REGION Network 27: STIRRER SPEED LINE 1 LIMITS CALCULATION ALARM
   RUNG wire#powerrail
      Add(in1 := #oPLC_Aux.o_rStirrerSpeedNominal_Line1, in2 := #"iHMI_Offsets Alarms and Warnings".StirrerSpeedNominalLine1_Max_Alarm, out => #oPLC_Aux.o_rHHlimitStirrerSpeedNominal_Line1)
      "FC21020_FEEDER_SCALING"(DINT_INPUT_VALUE := 0, REAL_INPUT_VALUE := #oPLC_Aux.o_rHHlimitStirrerSpeedNominal_Line1, DINT_TO_REAL := false, REAL_TRANSFORM_FOR_FEEDER := true, OUTPUT_VALUE_PLC => #Retval_Fill_R, OUTPUT_VALUE_FEEDER => #ioPowder_Feeder_Unit_In_Out.Outputs."PF Setpoints, Warnings and Alarms".o_rHHlimitStirrerSpeedNominal_Line1)
      Sub(in1 := #oPLC_Aux.o_rStirrerSpeedNominal_Line1, in2 := #"iHMI_Offsets Alarms and Warnings".StirrerSpeedNominalLine1_Min_Alarm, out => #oPLC_Aux.o_rLLlimitStirrerSpeedNominal_Line1)
      "FC21020_FEEDER_SCALING"(DINT_INPUT_VALUE := 0, REAL_INPUT_VALUE := #oPLC_Aux.o_rLLlimitStirrerSpeedNominal_Line1, DINT_TO_REAL := false, REAL_TRANSFORM_FOR_FEEDER := true, OUTPUT_VALUE_PLC => #Retval_Fill_R, OUTPUT_VALUE_FEEDER => #ioPowder_Feeder_Unit_In_Out.Outputs."PF Setpoints, Warnings and Alarms".o_rLLlimitStirrerSpeedNominal_Line1)
   END_RUNG
   // the same network as SCL:
   #oPLC_Aux.o_rHHlimitStirrerSpeedNominal_Line1 := #oPLC_Aux.o_rStirrerSpeedNominal_Line1 + #"iHMI_Offsets Alarms and Warnings".StirrerSpeedNominalLine1_Max_Alarm;
   "FC21020_FEEDER_SCALING"(DINT_INPUT_VALUE := 0,
                           REAL_INPUT_VALUE := #oPLC_Aux.o_rHHlimitStirrerSpeedNominal_Line1,
                           DINT_TO_REAL := false,
                           REAL_TRANSFORM_FOR_FEEDER := true,
                           OUTPUT_VALUE_PLC => #Retval_Fill_R,
                           OUTPUT_VALUE_FEEDER => #ioPowder_Feeder_Unit_In_Out.Outputs."PF Setpoints, Warnings and Alarms".o_rHHlimitStirrerSpeedNominal_Line1,
                           ENO => #_w1);
   IF #_w1 THEN
       #oPLC_Aux.o_rLLlimitStirrerSpeedNominal_Line1 := #oPLC_Aux.o_rStirrerSpeedNominal_Line1 - #"iHMI_Offsets Alarms and Warnings".StirrerSpeedNominalLine1_Min_Alarm;
       "FC21020_FEEDER_SCALING"(DINT_INPUT_VALUE := 0,
                               REAL_INPUT_VALUE := #oPLC_Aux.o_rLLlimitStirrerSpeedNominal_Line1,
                               DINT_TO_REAL := false,
                               REAL_TRANSFORM_FOR_FEEDER := true,
                               OUTPUT_VALUE_PLC => #Retval_Fill_R,
                               OUTPUT_VALUE_FEEDER => #ioPowder_Feeder_Unit_In_Out.Outputs."PF Setpoints, Warnings and Alarms".o_rLLlimitStirrerSpeedNominal_Line1);
   END_IF;
END_REGION

REGION Network 28: STIRRER SPEED LINE 2 LIMITS CALCULATION ALARM
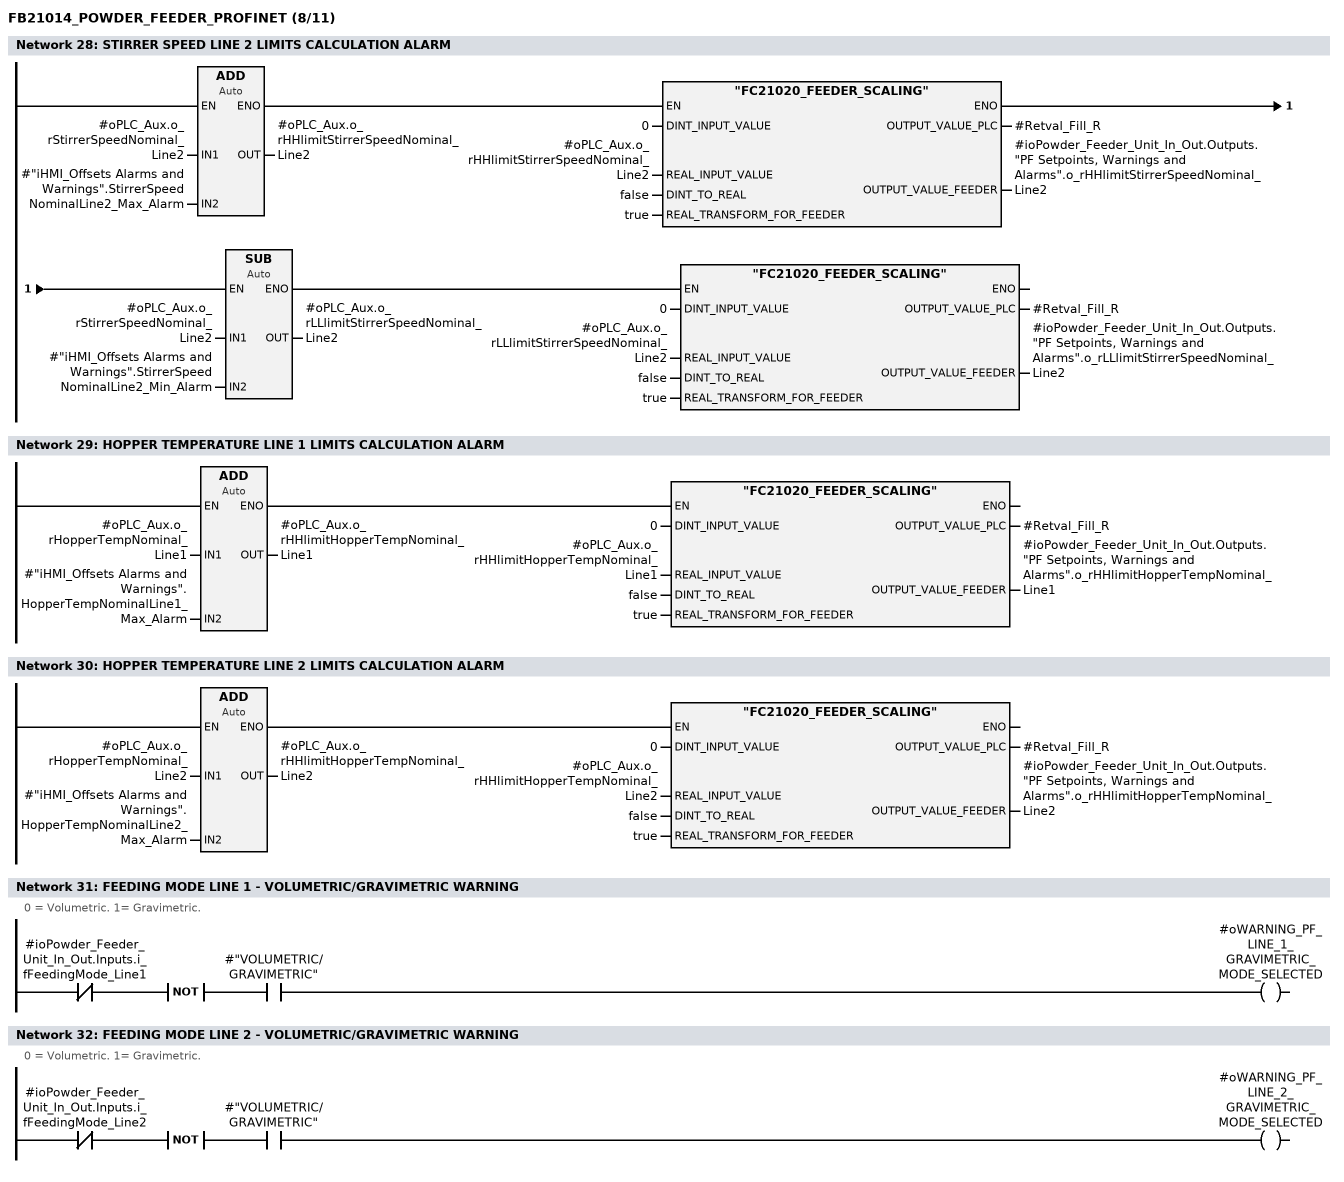
   RUNG wire#powerrail
      Add(in1 := #oPLC_Aux.o_rStirrerSpeedNominal_Line2, in2 := #"iHMI_Offsets Alarms and Warnings".StirrerSpeedNominalLine2_Max_Alarm, out => #oPLC_Aux.o_rHHlimitStirrerSpeedNominal_Line2)
      "FC21020_FEEDER_SCALING"(DINT_INPUT_VALUE := 0, REAL_INPUT_VALUE := #oPLC_Aux.o_rHHlimitStirrerSpeedNominal_Line2, DINT_TO_REAL := false, REAL_TRANSFORM_FOR_FEEDER := true, OUTPUT_VALUE_PLC => #Retval_Fill_R, OUTPUT_VALUE_FEEDER => #ioPowder_Feeder_Unit_In_Out.Outputs."PF Setpoints, Warnings and Alarms".o_rHHlimitStirrerSpeedNominal_Line2)
      Sub(in1 := #oPLC_Aux.o_rStirrerSpeedNominal_Line2, in2 := #"iHMI_Offsets Alarms and Warnings".StirrerSpeedNominalLine2_Min_Alarm, out => #oPLC_Aux.o_rLLlimitStirrerSpeedNominal_Line2)
      "FC21020_FEEDER_SCALING"(DINT_INPUT_VALUE := 0, REAL_INPUT_VALUE := #oPLC_Aux.o_rLLlimitStirrerSpeedNominal_Line2, DINT_TO_REAL := false, REAL_TRANSFORM_FOR_FEEDER := true, OUTPUT_VALUE_PLC => #Retval_Fill_R, OUTPUT_VALUE_FEEDER => #ioPowder_Feeder_Unit_In_Out.Outputs."PF Setpoints, Warnings and Alarms".o_rLLlimitStirrerSpeedNominal_Line2)
   END_RUNG
   // the same network as SCL:
   #oPLC_Aux.o_rHHlimitStirrerSpeedNominal_Line2 := #oPLC_Aux.o_rStirrerSpeedNominal_Line2 + #"iHMI_Offsets Alarms and Warnings".StirrerSpeedNominalLine2_Max_Alarm;
   "FC21020_FEEDER_SCALING"(DINT_INPUT_VALUE := 0,
                           REAL_INPUT_VALUE := #oPLC_Aux.o_rHHlimitStirrerSpeedNominal_Line2,
                           DINT_TO_REAL := false,
                           REAL_TRANSFORM_FOR_FEEDER := true,
                           OUTPUT_VALUE_PLC => #Retval_Fill_R,
                           OUTPUT_VALUE_FEEDER => #ioPowder_Feeder_Unit_In_Out.Outputs."PF Setpoints, Warnings and Alarms".o_rHHlimitStirrerSpeedNominal_Line2,
                           ENO => #_w1);
   IF #_w1 THEN
       #oPLC_Aux.o_rLLlimitStirrerSpeedNominal_Line2 := #oPLC_Aux.o_rStirrerSpeedNominal_Line2 - #"iHMI_Offsets Alarms and Warnings".StirrerSpeedNominalLine2_Min_Alarm;
       "FC21020_FEEDER_SCALING"(DINT_INPUT_VALUE := 0,
                               REAL_INPUT_VALUE := #oPLC_Aux.o_rLLlimitStirrerSpeedNominal_Line2,
                               DINT_TO_REAL := false,
                               REAL_TRANSFORM_FOR_FEEDER := true,
                               OUTPUT_VALUE_PLC => #Retval_Fill_R,
                               OUTPUT_VALUE_FEEDER => #ioPowder_Feeder_Unit_In_Out.Outputs."PF Setpoints, Warnings and Alarms".o_rLLlimitStirrerSpeedNominal_Line2);
   END_IF;
END_REGION

REGION Network 29: HOPPER TEMPERATURE LINE 1 LIMITS CALCULATION ALARM
   RUNG wire#powerrail
      Add(in1 := #oPLC_Aux.o_rHopperTempNominal_Line1, in2 := #"iHMI_Offsets Alarms and Warnings".HopperTempNominalLine1_Max_Alarm, out => #oPLC_Aux.o_rHHlimitHopperTempNominal_Line1)
      "FC21020_FEEDER_SCALING"(DINT_INPUT_VALUE := 0, REAL_INPUT_VALUE := #oPLC_Aux.o_rHHlimitHopperTempNominal_Line1, DINT_TO_REAL := false, REAL_TRANSFORM_FOR_FEEDER := true, OUTPUT_VALUE_PLC => #Retval_Fill_R, OUTPUT_VALUE_FEEDER => #ioPowder_Feeder_Unit_In_Out.Outputs."PF Setpoints, Warnings and Alarms".o_rHHlimitHopperTempNominal_Line1)
   END_RUNG
   // the same network as SCL:
   #oPLC_Aux.o_rHHlimitHopperTempNominal_Line1 := #oPLC_Aux.o_rHopperTempNominal_Line1 + #"iHMI_Offsets Alarms and Warnings".HopperTempNominalLine1_Max_Alarm;
   "FC21020_FEEDER_SCALING"(DINT_INPUT_VALUE := 0,
                           REAL_INPUT_VALUE := #oPLC_Aux.o_rHHlimitHopperTempNominal_Line1,
                           DINT_TO_REAL := false,
                           REAL_TRANSFORM_FOR_FEEDER := true,
                           OUTPUT_VALUE_PLC => #Retval_Fill_R,
                           OUTPUT_VALUE_FEEDER => #ioPowder_Feeder_Unit_In_Out.Outputs."PF Setpoints, Warnings and Alarms".o_rHHlimitHopperTempNominal_Line1);
END_REGION

REGION Network 30: HOPPER TEMPERATURE LINE 2 LIMITS CALCULATION ALARM
   RUNG wire#powerrail
      Add(in1 := #oPLC_Aux.o_rHopperTempNominal_Line2, in2 := #"iHMI_Offsets Alarms and Warnings".HopperTempNominalLine2_Max_Alarm, out => #oPLC_Aux.o_rHHlimitHopperTempNominal_Line2)
      "FC21020_FEEDER_SCALING"(DINT_INPUT_VALUE := 0, REAL_INPUT_VALUE := #oPLC_Aux.o_rHHlimitHopperTempNominal_Line2, DINT_TO_REAL := false, REAL_TRANSFORM_FOR_FEEDER := true, OUTPUT_VALUE_PLC => #Retval_Fill_R, OUTPUT_VALUE_FEEDER => #ioPowder_Feeder_Unit_In_Out.Outputs."PF Setpoints, Warnings and Alarms".o_rHHlimitHopperTempNominal_Line2)
   END_RUNG
   // the same network as SCL:
   #oPLC_Aux.o_rHHlimitHopperTempNominal_Line2 := #oPLC_Aux.o_rHopperTempNominal_Line2 + #"iHMI_Offsets Alarms and Warnings".HopperTempNominalLine2_Max_Alarm;
   "FC21020_FEEDER_SCALING"(DINT_INPUT_VALUE := 0,
                           REAL_INPUT_VALUE := #oPLC_Aux.o_rHHlimitHopperTempNominal_Line2,
                           DINT_TO_REAL := false,
                           REAL_TRANSFORM_FOR_FEEDER := true,
                           OUTPUT_VALUE_PLC => #Retval_Fill_R,
                           OUTPUT_VALUE_FEEDER => #ioPowder_Feeder_Unit_In_Out.Outputs."PF Setpoints, Warnings and Alarms".o_rHHlimitHopperTempNominal_Line2);
END_REGION

REGION Network 31: FEEDING MODE LINE 1 - VOLUMETRIC/GRAVIMETRIC WARNING
   // 0 = Volumetric. 1= Gravimetric.
   RUNG wire#powerrail
      I_Contact( #ioPowder_Feeder_Unit_In_Out.Inputs.i_fFeedingMode_Line1 )
      Not()
      Contact( #"VOLUMETRIC/GRAVIMETRIC" )
      Coil( #oWARNING_PF_LINE_1_GRAVIMETRIC_MODE_SELECTED )
   END_RUNG
   // the same network as SCL:
   #oWARNING_PF_LINE_1_GRAVIMETRIC_MODE_SELECTED := NOT (NOT #ioPowder_Feeder_Unit_In_Out.Inputs.i_fFeedingMode_Line1) AND #"VOLUMETRIC/GRAVIMETRIC";
END_REGION

REGION Network 32: FEEDING MODE LINE 2 - VOLUMETRIC/GRAVIMETRIC WARNING
   // 0 = Volumetric. 1= Gravimetric.
   RUNG wire#powerrail
      I_Contact( #ioPowder_Feeder_Unit_In_Out.Inputs.i_fFeedingMode_Line2 )
      Not()
      Contact( #"VOLUMETRIC/GRAVIMETRIC" )
      Coil( #oWARNING_PF_LINE_2_GRAVIMETRIC_MODE_SELECTED )
   END_RUNG
   // the same network as SCL:
   #oWARNING_PF_LINE_2_GRAVIMETRIC_MODE_SELECTED := NOT (NOT #ioPowder_Feeder_Unit_In_Out.Inputs.i_fFeedingMode_Line2) AND #"VOLUMETRIC/GRAVIMETRIC";
END_REGION

REGION Network 33: WARNING
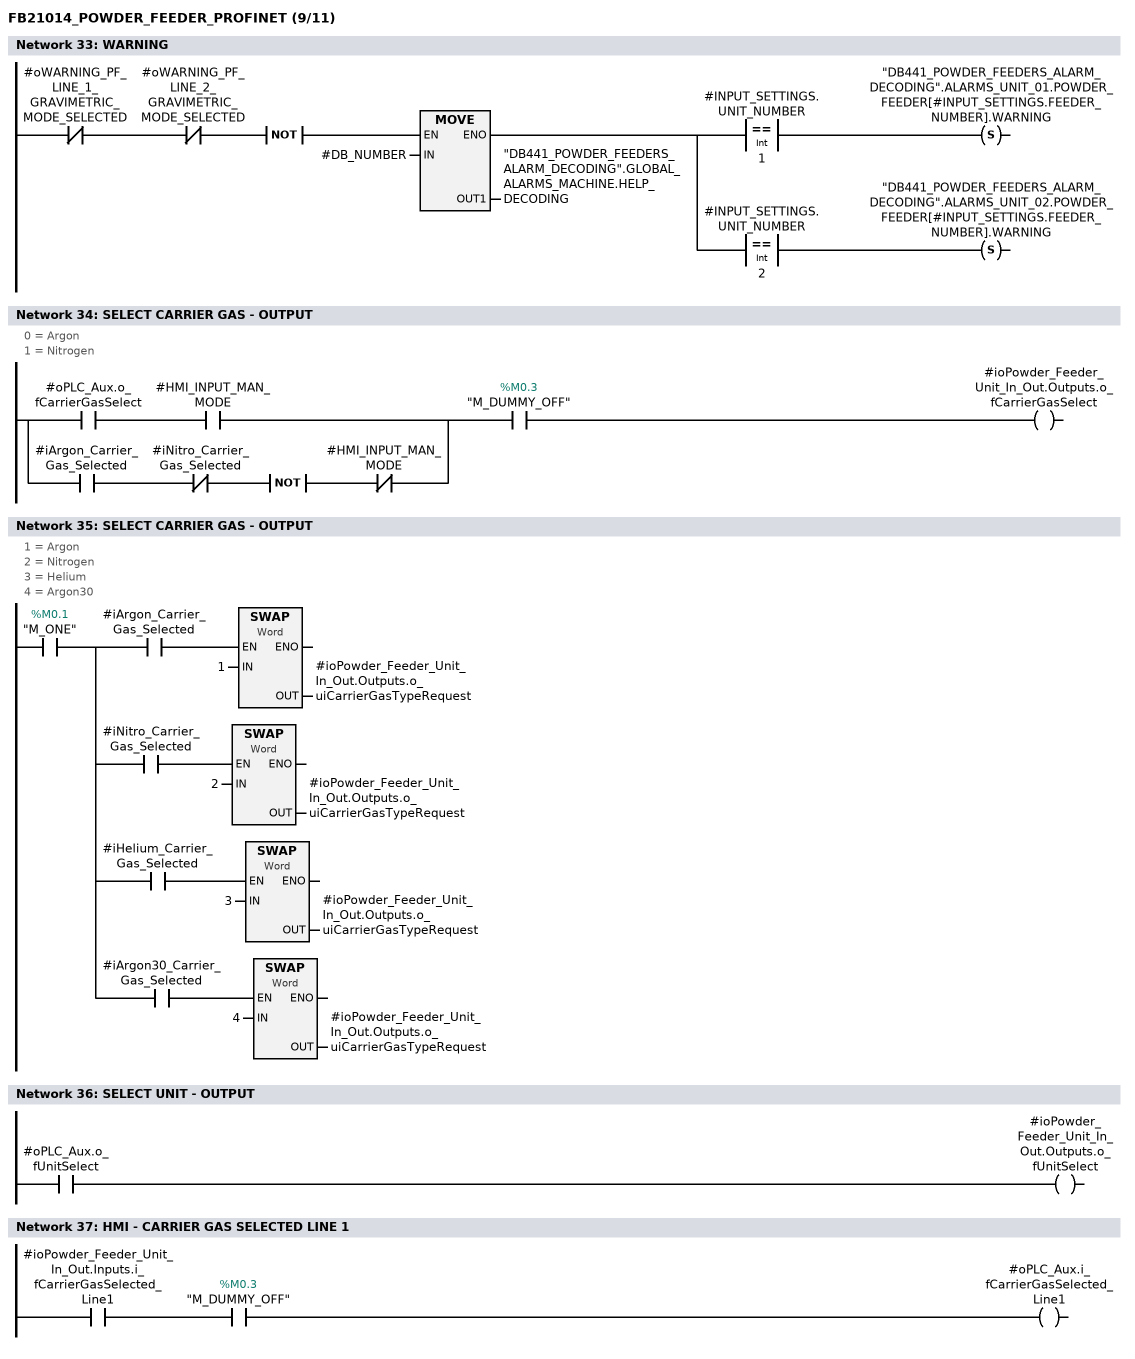
   RUNG wire#powerrail
      I_Contact( #oWARNING_PF_LINE_1_GRAVIMETRIC_MODE_SELECTED )
      I_Contact( #oWARNING_PF_LINE_2_GRAVIMETRIC_MODE_SELECTED )
      Not()
      Move(in := #DB_NUMBER, out1 => "DB441_POWDER_FEEDERS_ALARM_DECODING".GLOBAL_ALARMS_MACHINE.HELP_DECODING)
      wire#w1
      { S7_Templates := "SrcType := Int" } EQ_Contact(in1 := #INPUT_SETTINGS.UNIT_NUMBER, in2 := 1)
      S_Coil( "DB441_POWDER_FEEDERS_ALARM_DECODING".ALARMS_UNIT_01.POWDER_FEEDER[#INPUT_SETTINGS.FEEDER_NUMBER].WARNING )
   END_RUNG
   RUNG wire#w1
      { S7_Templates := "SrcType := Int" } EQ_Contact(in1 := #INPUT_SETTINGS.UNIT_NUMBER, in2 := 2)
      S_Coil( "DB441_POWDER_FEEDERS_ALARM_DECODING".ALARMS_UNIT_02.POWDER_FEEDER[#INPUT_SETTINGS.FEEDER_NUMBER].WARNING )
   END_RUNG
   // the same network as SCL:
   #_w1 := NOT (NOT #oWARNING_PF_LINE_1_GRAVIMETRIC_MODE_SELECTED AND NOT #oWARNING_PF_LINE_2_GRAVIMETRIC_MODE_SELECTED);
   IF #_w1 THEN
       "DB441_POWDER_FEEDERS_ALARM_DECODING".GLOBAL_ALARMS_MACHINE.HELP_DECODING := #DB_NUMBER;
   END_IF;
   IF #_w1 AND (#INPUT_SETTINGS.UNIT_NUMBER = 1) THEN
       "DB441_POWDER_FEEDERS_ALARM_DECODING".ALARMS_UNIT_01.POWDER_FEEDER[#INPUT_SETTINGS.FEEDER_NUMBER].WARNING := TRUE;
   END_IF;
   IF #_w1 AND (#INPUT_SETTINGS.UNIT_NUMBER = 2) THEN
       "DB441_POWDER_FEEDERS_ALARM_DECODING".ALARMS_UNIT_02.POWDER_FEEDER[#INPUT_SETTINGS.FEEDER_NUMBER].WARNING := TRUE;
   END_IF;
END_REGION

REGION Network 34: SELECT CARRIER GAS - OUTPUT
   // 0 = Argon
   // 1 = Nitrogen
   RUNG wire#powerrail
      Contact( #oPLC_Aux.o_fCarrierGasSelect )
      Contact( #HMI_INPUT_MAN_MODE )
      wire#w1
      Contact( "M_DUMMY_OFF" )
      Coil( #ioPowder_Feeder_Unit_In_Out.Outputs.o_fCarrierGasSelect )
   END_RUNG
   RUNG wire#powerrail
      Contact( #iArgon_Carrier_Gas_Selected )
      I_Contact( #iNitro_Carrier_Gas_Selected )
      Not()
      I_Contact( #HMI_INPUT_MAN_MODE )
   END_RUNG wire#w1
   // the same network as SCL:
   #ioPowder_Feeder_Unit_In_Out.Outputs.o_fCarrierGasSelect := ((#oPLC_Aux.o_fCarrierGasSelect AND #HMI_INPUT_MAN_MODE) OR (NOT (#iArgon_Carrier_Gas_Selected AND NOT #iNitro_Carrier_Gas_Selected) AND NOT #HMI_INPUT_MAN_MODE)) AND "M_DUMMY_OFF";
END_REGION

REGION Network 35: SELECT CARRIER GAS - OUTPUT
   // 1 = Argon
   // 2 = Nitrogen
   // 3 = Helium
   // 4 = Argon30
   IF "M_ONE" AND #iArgon_Carrier_Gas_Selected THEN
       #ioPowder_Feeder_Unit_In_Out.Outputs.o_uiCarrierGasTypeRequest := SWAP(1);
   END_IF;
   IF "M_ONE" AND #iNitro_Carrier_Gas_Selected THEN
       #ioPowder_Feeder_Unit_In_Out.Outputs.o_uiCarrierGasTypeRequest := SWAP(2);
   END_IF;
   IF "M_ONE" AND #iHelium_Carrier_Gas_Selected THEN
       #ioPowder_Feeder_Unit_In_Out.Outputs.o_uiCarrierGasTypeRequest := SWAP(3);
   END_IF;
   IF "M_ONE" AND #iArgon30_Carrier_Gas_Selected THEN
       #ioPowder_Feeder_Unit_In_Out.Outputs.o_uiCarrierGasTypeRequest := SWAP(4);
   END_IF;
END_REGION

REGION Network 36: SELECT UNIT - OUTPUT
   RUNG wire#powerrail
      Contact( #oPLC_Aux.o_fUnitSelect )
      Coil( #ioPowder_Feeder_Unit_In_Out.Outputs.o_fUnitSelect )
   END_RUNG
   // the same network as SCL:
   #ioPowder_Feeder_Unit_In_Out.Outputs.o_fUnitSelect := #oPLC_Aux.o_fUnitSelect;
END_REGION

REGION Network 37: HMI - CARRIER GAS SELECTED LINE 1
   RUNG wire#powerrail
      Contact( #ioPowder_Feeder_Unit_In_Out.Inputs.i_fCarrierGasSelected_Line1 )
      Contact( "M_DUMMY_OFF" )
      Coil( #oPLC_Aux.i_fCarrierGasSelected_Line1 )
   END_RUNG
   // the same network as SCL:
   #oPLC_Aux.i_fCarrierGasSelected_Line1 := #ioPowder_Feeder_Unit_In_Out.Inputs.i_fCarrierGasSelected_Line1 AND "M_DUMMY_OFF";
END_REGION

REGION Network 38: HMI - CARRIER GAS SELECTED LINE 2
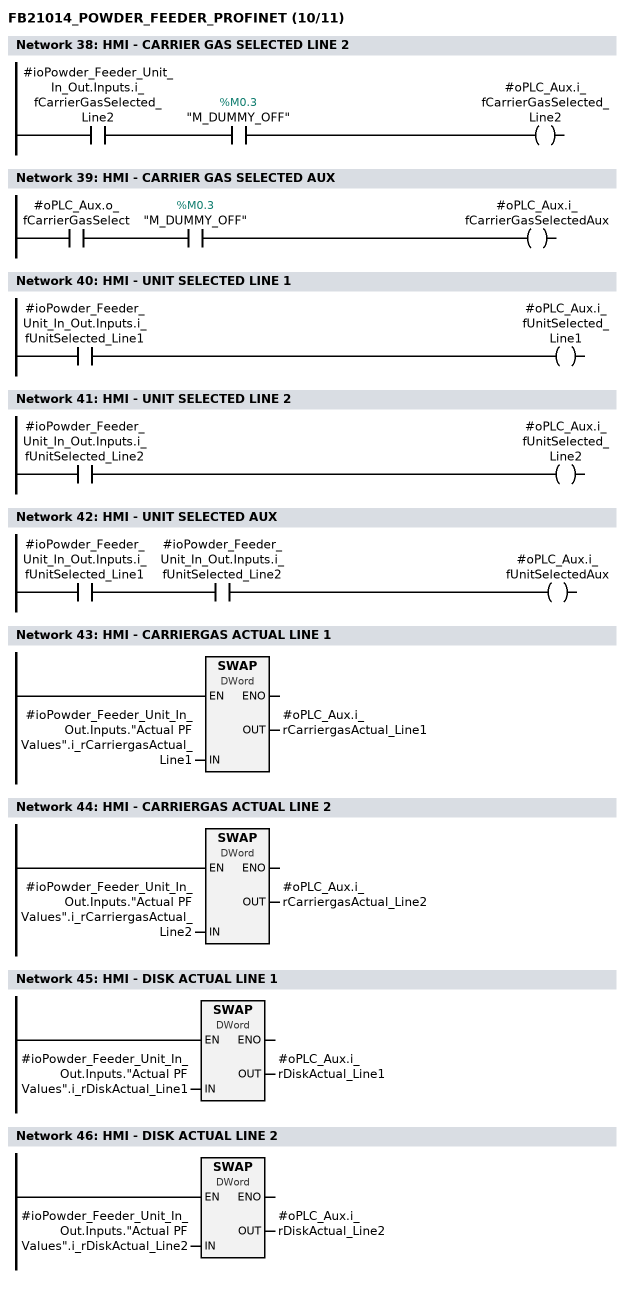
   RUNG wire#powerrail
      Contact( #ioPowder_Feeder_Unit_In_Out.Inputs.i_fCarrierGasSelected_Line2 )
      Contact( "M_DUMMY_OFF" )
      Coil( #oPLC_Aux.i_fCarrierGasSelected_Line2 )
   END_RUNG
   // the same network as SCL:
   #oPLC_Aux.i_fCarrierGasSelected_Line2 := #ioPowder_Feeder_Unit_In_Out.Inputs.i_fCarrierGasSelected_Line2 AND "M_DUMMY_OFF";
END_REGION

REGION Network 39: HMI - CARRIER GAS SELECTED AUX
   RUNG wire#powerrail
      Contact( #oPLC_Aux.o_fCarrierGasSelect )
      Contact( "M_DUMMY_OFF" )
      Coil( #oPLC_Aux.i_fCarrierGasSelectedAux )
   END_RUNG
   // the same network as SCL:
   #oPLC_Aux.i_fCarrierGasSelectedAux := #oPLC_Aux.o_fCarrierGasSelect AND "M_DUMMY_OFF";
END_REGION

REGION Network 40: HMI - UNIT SELECTED LINE 1
   RUNG wire#powerrail
      Contact( #ioPowder_Feeder_Unit_In_Out.Inputs.i_fUnitSelected_Line1 )
      Coil( #oPLC_Aux.i_fUnitSelected_Line1 )
   END_RUNG
   // the same network as SCL:
   #oPLC_Aux.i_fUnitSelected_Line1 := #ioPowder_Feeder_Unit_In_Out.Inputs.i_fUnitSelected_Line1;
END_REGION

REGION Network 41: HMI - UNIT SELECTED LINE 2
   RUNG wire#powerrail
      Contact( #ioPowder_Feeder_Unit_In_Out.Inputs.i_fUnitSelected_Line2 )
      Coil( #oPLC_Aux.i_fUnitSelected_Line2 )
   END_RUNG
   // the same network as SCL:
   #oPLC_Aux.i_fUnitSelected_Line2 := #ioPowder_Feeder_Unit_In_Out.Inputs.i_fUnitSelected_Line2;
END_REGION

REGION Network 42: HMI - UNIT SELECTED AUX
   RUNG wire#powerrail
      Contact( #ioPowder_Feeder_Unit_In_Out.Inputs.i_fUnitSelected_Line1 )
      Contact( #ioPowder_Feeder_Unit_In_Out.Inputs.i_fUnitSelected_Line2 )
      Coil( #oPLC_Aux.i_fUnitSelectedAux )
   END_RUNG
   // the same network as SCL:
   #oPLC_Aux.i_fUnitSelectedAux := #ioPowder_Feeder_Unit_In_Out.Inputs.i_fUnitSelected_Line1 AND #ioPowder_Feeder_Unit_In_Out.Inputs.i_fUnitSelected_Line2;
END_REGION

REGION Network 43: HMI - CARRIERGAS ACTUAL LINE 1
   #oPLC_Aux.i_rCarriergasActual_Line1 := SWAP(#ioPowder_Feeder_Unit_In_Out.Inputs."Actual PF Values".i_rCarriergasActual_Line1);
END_REGION

REGION Network 44: HMI - CARRIERGAS ACTUAL LINE 2
   #oPLC_Aux.i_rCarriergasActual_Line2 := SWAP(#ioPowder_Feeder_Unit_In_Out.Inputs."Actual PF Values".i_rCarriergasActual_Line2);
END_REGION

REGION Network 45: HMI - DISK ACTUAL LINE 1
   #oPLC_Aux.i_rDiskActual_Line1 := SWAP(#ioPowder_Feeder_Unit_In_Out.Inputs."Actual PF Values".i_rDiskActual_Line1);
END_REGION

REGION Network 46: HMI - DISK ACTUAL LINE 2
   #oPLC_Aux.i_rDiskActual_Line2 := SWAP(#ioPowder_Feeder_Unit_In_Out.Inputs."Actual PF Values".i_rDiskActual_Line2);
END_REGION

REGION Network 47: HMI - STIRRER ACTUAL LINE 1
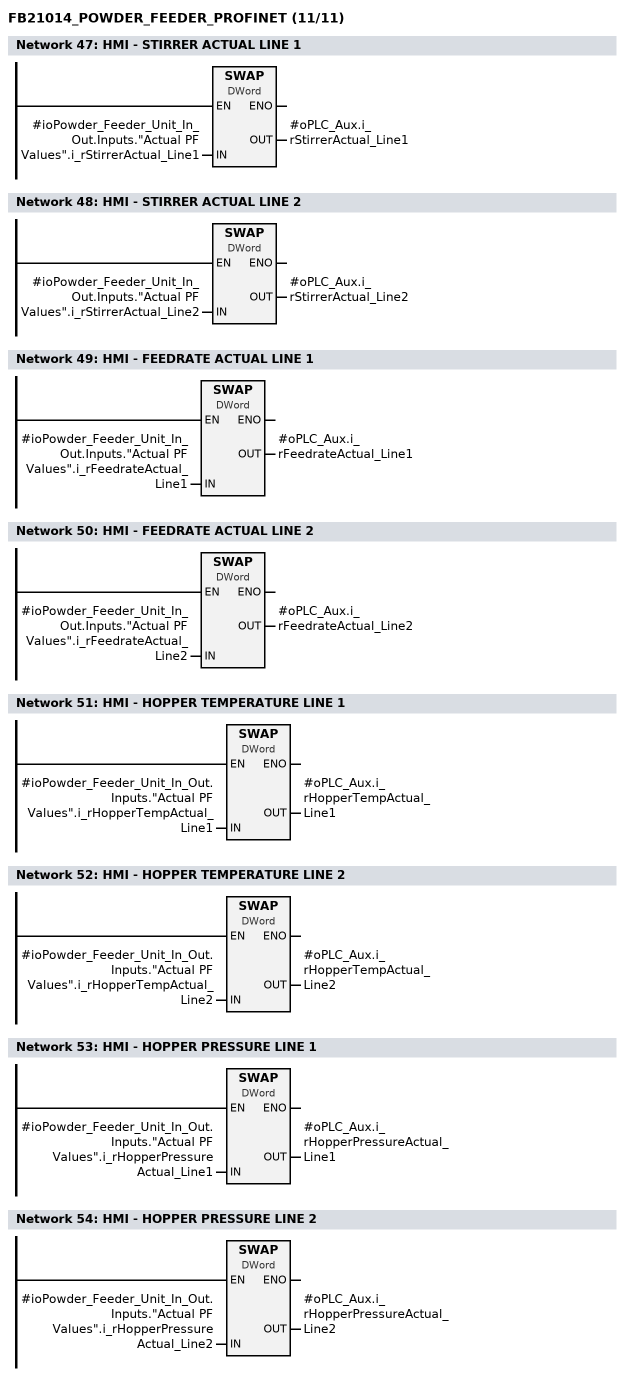
   #oPLC_Aux.i_rStirrerActual_Line1 := SWAP(#ioPowder_Feeder_Unit_In_Out.Inputs."Actual PF Values".i_rStirrerActual_Line1);
END_REGION

REGION Network 48: HMI - STIRRER ACTUAL LINE 2
   #oPLC_Aux.i_rStirrerActual_Line2 := SWAP(#ioPowder_Feeder_Unit_In_Out.Inputs."Actual PF Values".i_rStirrerActual_Line2);
END_REGION

REGION Network 49: HMI - FEEDRATE ACTUAL LINE 1
   #oPLC_Aux.i_rFeedrateActual_Line1 := SWAP(#ioPowder_Feeder_Unit_In_Out.Inputs."Actual PF Values".i_rFeedrateActual_Line1);
END_REGION

REGION Network 50: HMI - FEEDRATE ACTUAL LINE 2
   #oPLC_Aux.i_rFeedrateActual_Line2 := SWAP(#ioPowder_Feeder_Unit_In_Out.Inputs."Actual PF Values".i_rFeedrateActual_Line2);
END_REGION

REGION Network 51: HMI - HOPPER TEMPERATURE LINE 1
   #oPLC_Aux.i_rHopperTempActual_Line1 := SWAP(#ioPowder_Feeder_Unit_In_Out.Inputs."Actual PF Values".i_rHopperTempActual_Line1);
END_REGION

REGION Network 52: HMI - HOPPER TEMPERATURE LINE 2
   #oPLC_Aux.i_rHopperTempActual_Line2 := SWAP(#ioPowder_Feeder_Unit_In_Out.Inputs."Actual PF Values".i_rHopperTempActual_Line2);
END_REGION

REGION Network 53: HMI - HOPPER PRESSURE LINE 1
   #oPLC_Aux.i_rHopperPressureActual_Line1 := SWAP(#ioPowder_Feeder_Unit_In_Out.Inputs."Actual PF Values".i_rHopperPressureActual_Line1);
END_REGION

REGION Network 54: HMI - HOPPER PRESSURE LINE 2
   #oPLC_Aux.i_rHopperPressureActual_Line2 := SWAP(#ioPowder_Feeder_Unit_In_Out.Inputs."Actual PF Values".i_rHopperPressureActual_Line2);
END_REGION
END_FUNCTION_BLOCK

FUNCTION "FC21020_FEEDER_SCALING" : Void   // FC21020, LAD
TITLE = Robot-PLC Scaling
{ S7_Optimized_Access := 'TRUE' }
AUTHOR : Jbarturen
VERSION : 0.1
// stored: AutoNumber false, IsIECCheckEnabled false, SetENOAutomatically false, UDAEnableTagReadback false
   VAR_INPUT
      DINT_INPUT_VALUE : DInt;
      REAL_INPUT_VALUE : Real;
      DINT_TO_REAL : Bool;
      REAL_TRANSFORM_FOR_FEEDER : Bool;
   END_VAR
   VAR_OUTPUT
      OUTPUT_VALUE_PLC : Real;
      OUTPUT_VALUE_FEEDER : Real;
   END_VAR
   VAR_TEMP
      Value_Swapped : DInt;
      Value_Real : Real;
      Value_PLC : Real;
      Value_DWord : DWord;
      Value_DWord_Swapped : DWord;
   END_VAR
BEGIN

REGION Network 1: DATA TYPE CONVERTION / Robot-PLC
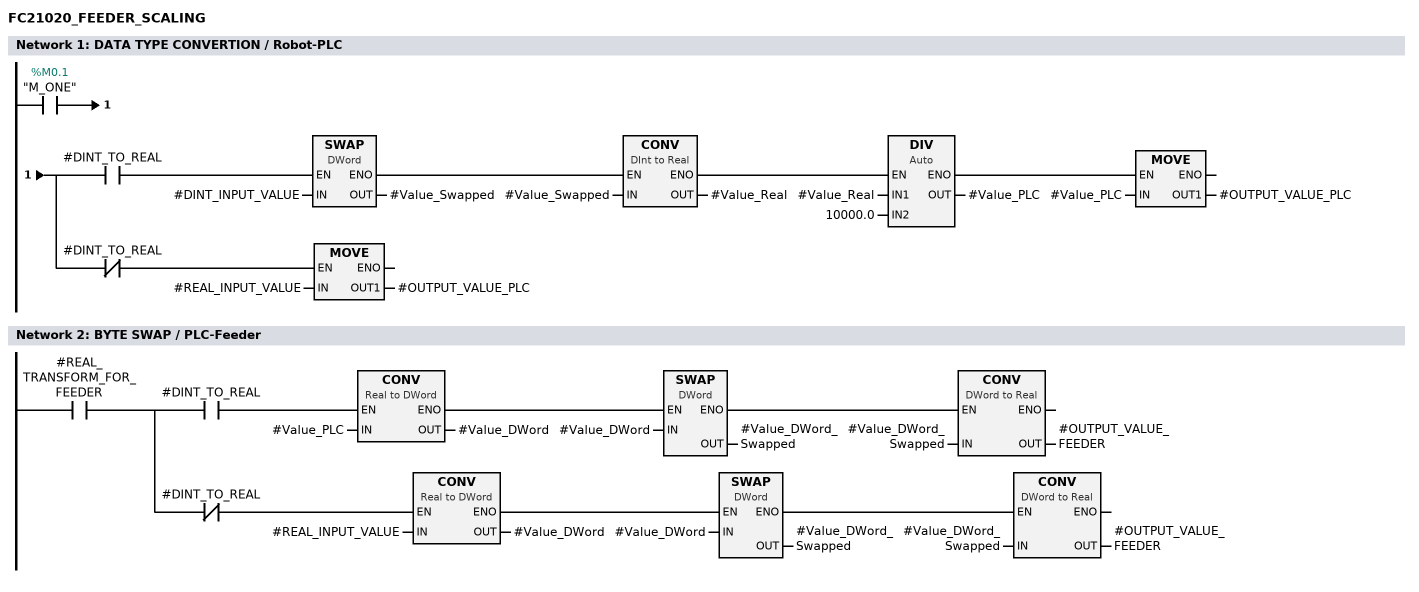
   IF "M_ONE" AND #DINT_TO_REAL THEN
       #Value_Swapped := SWAP(#DINT_INPUT_VALUE);
       #Value_Real := DINT_TO_REAL(#Value_Swapped);
       #Value_PLC := #Value_Real / 10000.0;
       #OUTPUT_VALUE_PLC := #Value_PLC;
   END_IF;
   IF "M_ONE" AND NOT #DINT_TO_REAL THEN #OUTPUT_VALUE_PLC := #REAL_INPUT_VALUE; END_IF;
END_REGION

REGION Network 2: BYTE SWAP / PLC-Feeder
   IF #REAL_TRANSFORM_FOR_FEEDER AND #DINT_TO_REAL THEN
       #Value_DWord := REAL_TO_DWORD(#Value_PLC);
       #Value_DWord_Swapped := SWAP(#Value_DWord);
       #OUTPUT_VALUE_FEEDER := DWORD_TO_REAL(#Value_DWord_Swapped);
   END_IF;
   IF #REAL_TRANSFORM_FOR_FEEDER AND NOT #DINT_TO_REAL THEN
       #Value_DWord := REAL_TO_DWORD(#REAL_INPUT_VALUE);
       #Value_DWord_Swapped := SWAP(#Value_DWord);
       #OUTPUT_VALUE_FEEDER := DWORD_TO_REAL(#Value_DWord_Swapped);
   END_IF;
END_REGION
END_FUNCTION

FUNCTION "FC21200_POWDER_FLOW_SENSOR_MEDICOAT" : Void   // FC21200, LAD
{ S7_Optimized_Access := 'TRUE' }
VERSION : 0.1
// stored: AutoNumber false, IsIECCheckEnabled false, SetENOAutomatically false, UDAEnableTagReadback false
BEGIN

REGION Network 1: /////_UNIT_01_/////
END_REGION

REGION Network 2: OERLIKON 1 LINE 1 OUTPUT MEDICOAT
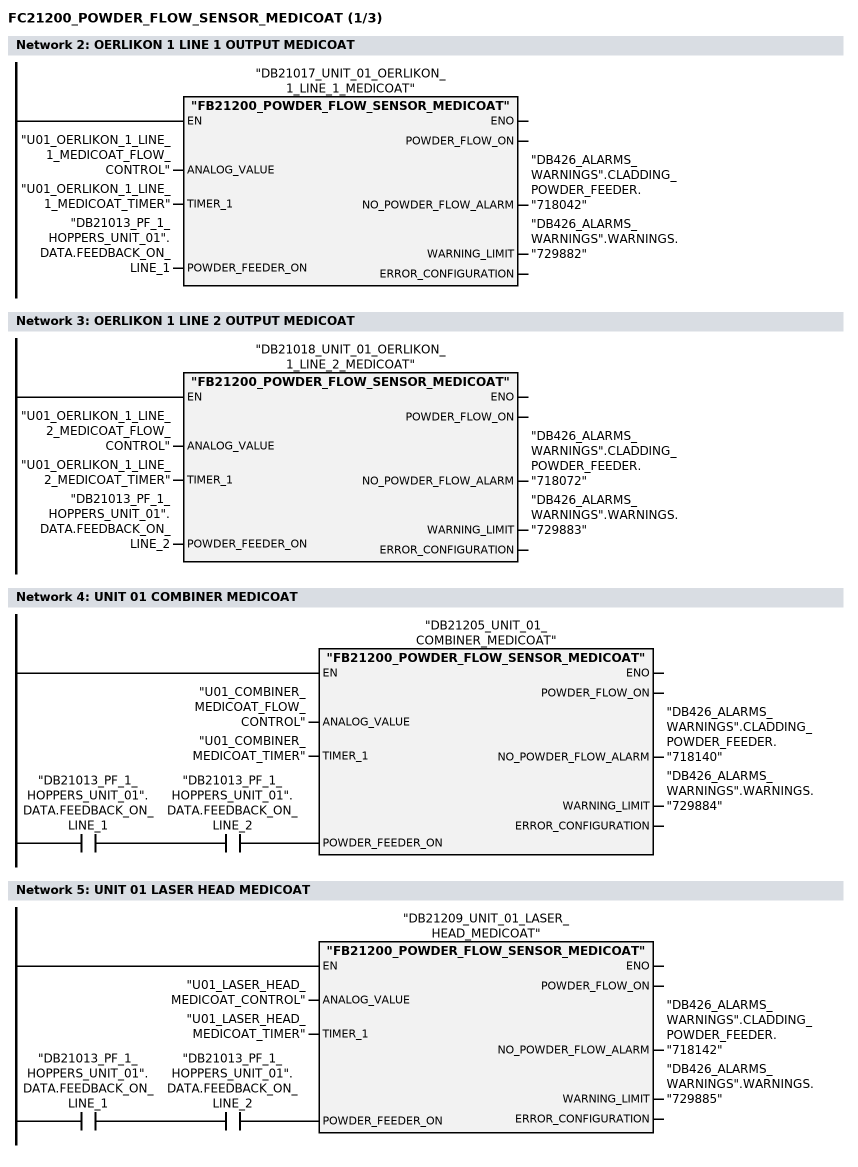
   RUNG wire#powerrail
      "DB21017_UNIT_01_OERLIKON_1_LINE_1_MEDICOAT"(ANALOG_VALUE := "U01_OERLIKON_1_LINE_1_MEDICOAT_FLOW_CONTROL", TIMER_1 := "U01_OERLIKON_1_LINE_1_MEDICOAT_TIMER", POWDER_FEEDER_ON := "DB21013_PF_1_HOPPERS_UNIT_01".DATA.FEEDBACK_ON_LINE_1, POWDER_FLOW_ON =>, NO_POWDER_FLOW_ALARM => "DB426_ALARMS_WARNINGS".CLADDING_POWDER_FEEDER."718042", WARNING_LIMIT => "DB426_ALARMS_WARNINGS".WARNINGS."729882", ERROR_CONFIGURATION =>)
   END_RUNG
   // the same network as SCL:
   "DB21017_UNIT_01_OERLIKON_1_LINE_1_MEDICOAT"(ANALOG_VALUE := "U01_OERLIKON_1_LINE_1_MEDICOAT_FLOW_CONTROL",   // "FB21200_POWDER_FLOW_SENSOR_MEDICOAT"
                           TIMER_1 := "U01_OERLIKON_1_LINE_1_MEDICOAT_TIMER",
                           POWDER_FEEDER_ON := "DB21013_PF_1_HOPPERS_UNIT_01".DATA.FEEDBACK_ON_LINE_1,
                           NO_POWDER_FLOW_ALARM => "DB426_ALARMS_WARNINGS".CLADDING_POWDER_FEEDER."718042",
                           WARNING_LIMIT => "DB426_ALARMS_WARNINGS".WARNINGS."729882");
END_REGION

REGION Network 3: OERLIKON 1 LINE 2 OUTPUT MEDICOAT
   RUNG wire#powerrail
      "DB21018_UNIT_01_OERLIKON_1_LINE_2_MEDICOAT"(ANALOG_VALUE := "U01_OERLIKON_1_LINE_2_MEDICOAT_FLOW_CONTROL", TIMER_1 := "U01_OERLIKON_1_LINE_2_MEDICOAT_TIMER", POWDER_FEEDER_ON := "DB21013_PF_1_HOPPERS_UNIT_01".DATA.FEEDBACK_ON_LINE_2, POWDER_FLOW_ON =>, NO_POWDER_FLOW_ALARM => "DB426_ALARMS_WARNINGS".CLADDING_POWDER_FEEDER."718072", WARNING_LIMIT => "DB426_ALARMS_WARNINGS".WARNINGS."729883", ERROR_CONFIGURATION =>)
   END_RUNG
   // the same network as SCL:
   "DB21018_UNIT_01_OERLIKON_1_LINE_2_MEDICOAT"(ANALOG_VALUE := "U01_OERLIKON_1_LINE_2_MEDICOAT_FLOW_CONTROL",   // "FB21200_POWDER_FLOW_SENSOR_MEDICOAT"
                           TIMER_1 := "U01_OERLIKON_1_LINE_2_MEDICOAT_TIMER",
                           POWDER_FEEDER_ON := "DB21013_PF_1_HOPPERS_UNIT_01".DATA.FEEDBACK_ON_LINE_2,
                           NO_POWDER_FLOW_ALARM => "DB426_ALARMS_WARNINGS".CLADDING_POWDER_FEEDER."718072",
                           WARNING_LIMIT => "DB426_ALARMS_WARNINGS".WARNINGS."729883");
END_REGION

REGION Network 4: UNIT 01 COMBINER MEDICOAT
   RUNG wire#powerrail
      "DB21205_UNIT_01_COMBINER_MEDICOAT"(POWDER_FEEDER_ON := wire#w1, ANALOG_VALUE := "U01_COMBINER_MEDICOAT_FLOW_CONTROL", TIMER_1 := "U01_COMBINER_MEDICOAT_TIMER", POWDER_FLOW_ON =>, NO_POWDER_FLOW_ALARM => "DB426_ALARMS_WARNINGS".CLADDING_POWDER_FEEDER."718140", WARNING_LIMIT => "DB426_ALARMS_WARNINGS".WARNINGS."729884", ERROR_CONFIGURATION =>)
   END_RUNG
   RUNG wire#powerrail
      Contact( "DB21013_PF_1_HOPPERS_UNIT_01".DATA.FEEDBACK_ON_LINE_1 )
      Contact( "DB21013_PF_1_HOPPERS_UNIT_01".DATA.FEEDBACK_ON_LINE_2 )
   END_RUNG wire#w1
   // the same network as SCL:
   "DB21205_UNIT_01_COMBINER_MEDICOAT"(ANALOG_VALUE := "U01_COMBINER_MEDICOAT_FLOW_CONTROL",   // "FB21200_POWDER_FLOW_SENSOR_MEDICOAT"
                           TIMER_1 := "U01_COMBINER_MEDICOAT_TIMER",
                           POWDER_FEEDER_ON := "DB21013_PF_1_HOPPERS_UNIT_01".DATA.FEEDBACK_ON_LINE_1 AND "DB21013_PF_1_HOPPERS_UNIT_01".DATA.FEEDBACK_ON_LINE_2,
                           NO_POWDER_FLOW_ALARM => "DB426_ALARMS_WARNINGS".CLADDING_POWDER_FEEDER."718140",
                           WARNING_LIMIT => "DB426_ALARMS_WARNINGS".WARNINGS."729884");
END_REGION

REGION Network 5: UNIT 01 LASER HEAD MEDICOAT
   RUNG wire#powerrail
      "DB21209_UNIT_01_LASER_HEAD_MEDICOAT"(POWDER_FEEDER_ON := wire#w1, ANALOG_VALUE := "U01_LASER_HEAD_MEDICOAT_CONTROL", TIMER_1 := "U01_LASER_HEAD_MEDICOAT_TIMER", POWDER_FLOW_ON =>, NO_POWDER_FLOW_ALARM => "DB426_ALARMS_WARNINGS".CLADDING_POWDER_FEEDER."718142", WARNING_LIMIT => "DB426_ALARMS_WARNINGS".WARNINGS."729885", ERROR_CONFIGURATION =>)
   END_RUNG
   RUNG wire#powerrail
      Contact( "DB21013_PF_1_HOPPERS_UNIT_01".DATA.FEEDBACK_ON_LINE_1 )
      Contact( "DB21013_PF_1_HOPPERS_UNIT_01".DATA.FEEDBACK_ON_LINE_2 )
   END_RUNG wire#w1
   // the same network as SCL:
   "DB21209_UNIT_01_LASER_HEAD_MEDICOAT"(ANALOG_VALUE := "U01_LASER_HEAD_MEDICOAT_CONTROL",   // "FB21200_POWDER_FLOW_SENSOR_MEDICOAT"
                           TIMER_1 := "U01_LASER_HEAD_MEDICOAT_TIMER",
                           POWDER_FEEDER_ON := "DB21013_PF_1_HOPPERS_UNIT_01".DATA.FEEDBACK_ON_LINE_1 AND "DB21013_PF_1_HOPPERS_UNIT_01".DATA.FEEDBACK_ON_LINE_2,
                           NO_POWDER_FLOW_ALARM => "DB426_ALARMS_WARNINGS".CLADDING_POWDER_FEEDER."718142",
                           WARNING_LIMIT => "DB426_ALARMS_WARNINGS".WARNINGS."729885");
END_REGION

REGION Network 6: /////_UNIT_02_/////
END_REGION

REGION Network 7: UNIT 02 OERLIKON 1 LINE 1 OUTPUT MEDICOAT
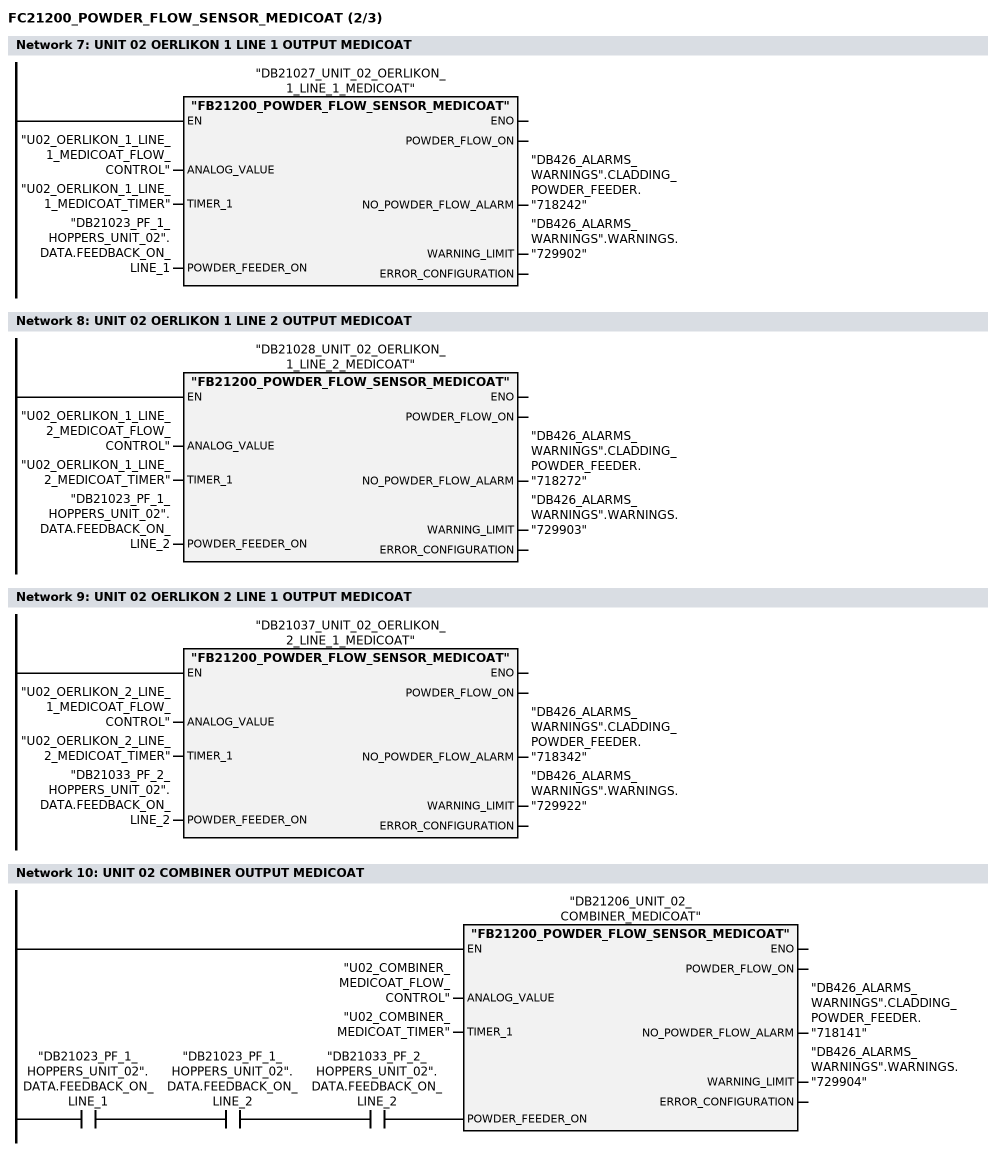
   RUNG wire#powerrail
      "DB21027_UNIT_02_OERLIKON_1_LINE_1_MEDICOAT"(ANALOG_VALUE := "U02_OERLIKON_1_LINE_1_MEDICOAT_FLOW_CONTROL", TIMER_1 := "U02_OERLIKON_1_LINE_1_MEDICOAT_TIMER", POWDER_FEEDER_ON := "DB21023_PF_1_HOPPERS_UNIT_02".DATA.FEEDBACK_ON_LINE_1, POWDER_FLOW_ON =>, NO_POWDER_FLOW_ALARM => "DB426_ALARMS_WARNINGS".CLADDING_POWDER_FEEDER."718242", WARNING_LIMIT => "DB426_ALARMS_WARNINGS".WARNINGS."729902", ERROR_CONFIGURATION =>)
   END_RUNG
   // the same network as SCL:
   "DB21027_UNIT_02_OERLIKON_1_LINE_1_MEDICOAT"(ANALOG_VALUE := "U02_OERLIKON_1_LINE_1_MEDICOAT_FLOW_CONTROL",   // "FB21200_POWDER_FLOW_SENSOR_MEDICOAT"
                           TIMER_1 := "U02_OERLIKON_1_LINE_1_MEDICOAT_TIMER",
                           POWDER_FEEDER_ON := "DB21023_PF_1_HOPPERS_UNIT_02".DATA.FEEDBACK_ON_LINE_1,
                           NO_POWDER_FLOW_ALARM => "DB426_ALARMS_WARNINGS".CLADDING_POWDER_FEEDER."718242",
                           WARNING_LIMIT => "DB426_ALARMS_WARNINGS".WARNINGS."729902");
END_REGION

REGION Network 8: UNIT 02 OERLIKON 1 LINE 2 OUTPUT MEDICOAT
   RUNG wire#powerrail
      "DB21028_UNIT_02_OERLIKON_1_LINE_2_MEDICOAT"(ANALOG_VALUE := "U02_OERLIKON_1_LINE_2_MEDICOAT_FLOW_CONTROL", TIMER_1 := "U02_OERLIKON_1_LINE_2_MEDICOAT_TIMER", POWDER_FEEDER_ON := "DB21023_PF_1_HOPPERS_UNIT_02".DATA.FEEDBACK_ON_LINE_2, POWDER_FLOW_ON =>, NO_POWDER_FLOW_ALARM => "DB426_ALARMS_WARNINGS".CLADDING_POWDER_FEEDER."718272", WARNING_LIMIT => "DB426_ALARMS_WARNINGS".WARNINGS."729903", ERROR_CONFIGURATION =>)
   END_RUNG
   // the same network as SCL:
   "DB21028_UNIT_02_OERLIKON_1_LINE_2_MEDICOAT"(ANALOG_VALUE := "U02_OERLIKON_1_LINE_2_MEDICOAT_FLOW_CONTROL",   // "FB21200_POWDER_FLOW_SENSOR_MEDICOAT"
                           TIMER_1 := "U02_OERLIKON_1_LINE_2_MEDICOAT_TIMER",
                           POWDER_FEEDER_ON := "DB21023_PF_1_HOPPERS_UNIT_02".DATA.FEEDBACK_ON_LINE_2,
                           NO_POWDER_FLOW_ALARM => "DB426_ALARMS_WARNINGS".CLADDING_POWDER_FEEDER."718272",
                           WARNING_LIMIT => "DB426_ALARMS_WARNINGS".WARNINGS."729903");
END_REGION

REGION Network 9: UNIT 02 OERLIKON 2 LINE 1 OUTPUT MEDICOAT
   RUNG wire#powerrail
      "DB21037_UNIT_02_OERLIKON_2_LINE_1_MEDICOAT"(ANALOG_VALUE := "U02_OERLIKON_2_LINE_1_MEDICOAT_FLOW_CONTROL", TIMER_1 := "U02_OERLIKON_2_LINE_2_MEDICOAT_TIMER", POWDER_FEEDER_ON := "DB21033_PF_2_HOPPERS_UNIT_02".DATA.FEEDBACK_ON_LINE_2, POWDER_FLOW_ON =>, NO_POWDER_FLOW_ALARM => "DB426_ALARMS_WARNINGS".CLADDING_POWDER_FEEDER."718342", WARNING_LIMIT => "DB426_ALARMS_WARNINGS".WARNINGS."729922", ERROR_CONFIGURATION =>)
   END_RUNG
   // the same network as SCL:
   "DB21037_UNIT_02_OERLIKON_2_LINE_1_MEDICOAT"(ANALOG_VALUE := "U02_OERLIKON_2_LINE_1_MEDICOAT_FLOW_CONTROL",   // "FB21200_POWDER_FLOW_SENSOR_MEDICOAT"
                           TIMER_1 := "U02_OERLIKON_2_LINE_2_MEDICOAT_TIMER",
                           POWDER_FEEDER_ON := "DB21033_PF_2_HOPPERS_UNIT_02".DATA.FEEDBACK_ON_LINE_2,
                           NO_POWDER_FLOW_ALARM => "DB426_ALARMS_WARNINGS".CLADDING_POWDER_FEEDER."718342",
                           WARNING_LIMIT => "DB426_ALARMS_WARNINGS".WARNINGS."729922");
END_REGION

REGION Network 10: UNIT 02 COMBINER OUTPUT MEDICOAT
   RUNG wire#powerrail
      "DB21206_UNIT_02_COMBINER_MEDICOAT"(POWDER_FEEDER_ON := wire#w1, ANALOG_VALUE := "U02_COMBINER_MEDICOAT_FLOW_CONTROL", TIMER_1 := "U02_COMBINER_MEDICOAT_TIMER", POWDER_FLOW_ON =>, NO_POWDER_FLOW_ALARM => "DB426_ALARMS_WARNINGS".CLADDING_POWDER_FEEDER."718141", WARNING_LIMIT => "DB426_ALARMS_WARNINGS".WARNINGS."729904", ERROR_CONFIGURATION =>)
   END_RUNG
   RUNG wire#powerrail
      Contact( "DB21023_PF_1_HOPPERS_UNIT_02".DATA.FEEDBACK_ON_LINE_1 )
      Contact( "DB21023_PF_1_HOPPERS_UNIT_02".DATA.FEEDBACK_ON_LINE_2 )
      Contact( "DB21033_PF_2_HOPPERS_UNIT_02".DATA.FEEDBACK_ON_LINE_2 )
   END_RUNG wire#w1
   // the same network as SCL:
   "DB21206_UNIT_02_COMBINER_MEDICOAT"(ANALOG_VALUE := "U02_COMBINER_MEDICOAT_FLOW_CONTROL",   // "FB21200_POWDER_FLOW_SENSOR_MEDICOAT"
                           TIMER_1 := "U02_COMBINER_MEDICOAT_TIMER",
                           POWDER_FEEDER_ON := "DB21023_PF_1_HOPPERS_UNIT_02".DATA.FEEDBACK_ON_LINE_1 AND "DB21023_PF_1_HOPPERS_UNIT_02".DATA.FEEDBACK_ON_LINE_2 AND "DB21033_PF_2_HOPPERS_UNIT_02".DATA.FEEDBACK_ON_LINE_2,
                           NO_POWDER_FLOW_ALARM => "DB426_ALARMS_WARNINGS".CLADDING_POWDER_FEEDER."718141",
                           WARNING_LIMIT => "DB426_ALARMS_WARNINGS".WARNINGS."729904");
END_REGION

REGION Network 11: UNIT 02 LASER HEAD OUTPUT MEDICOAT
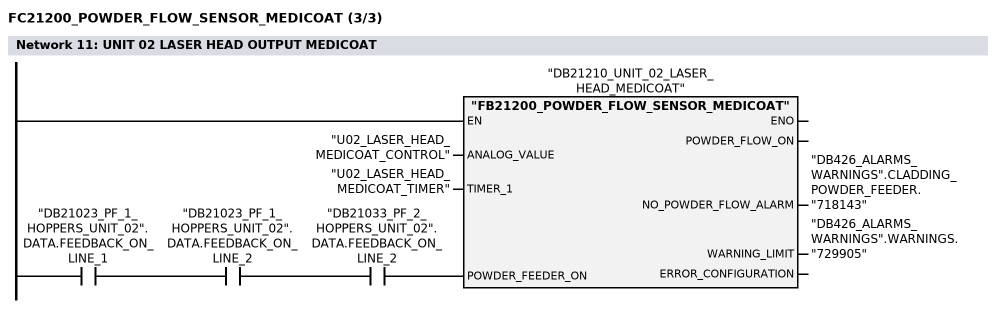
   RUNG wire#powerrail
      "DB21210_UNIT_02_LASER_HEAD_MEDICOAT"(POWDER_FEEDER_ON := wire#w1, ANALOG_VALUE := "U02_LASER_HEAD_MEDICOAT_CONTROL", TIMER_1 := "U02_LASER_HEAD_MEDICOAT_TIMER", POWDER_FLOW_ON =>, NO_POWDER_FLOW_ALARM => "DB426_ALARMS_WARNINGS".CLADDING_POWDER_FEEDER."718143", WARNING_LIMIT => "DB426_ALARMS_WARNINGS".WARNINGS."729905", ERROR_CONFIGURATION =>)
   END_RUNG
   RUNG wire#powerrail
      Contact( "DB21023_PF_1_HOPPERS_UNIT_02".DATA.FEEDBACK_ON_LINE_1 )
      Contact( "DB21023_PF_1_HOPPERS_UNIT_02".DATA.FEEDBACK_ON_LINE_2 )
      Contact( "DB21033_PF_2_HOPPERS_UNIT_02".DATA.FEEDBACK_ON_LINE_2 )
   END_RUNG wire#w1
   // the same network as SCL:
   "DB21210_UNIT_02_LASER_HEAD_MEDICOAT"(ANALOG_VALUE := "U02_LASER_HEAD_MEDICOAT_CONTROL",   // "FB21200_POWDER_FLOW_SENSOR_MEDICOAT"
                           TIMER_1 := "U02_LASER_HEAD_MEDICOAT_TIMER",
                           POWDER_FEEDER_ON := "DB21023_PF_1_HOPPERS_UNIT_02".DATA.FEEDBACK_ON_LINE_1 AND "DB21023_PF_1_HOPPERS_UNIT_02".DATA.FEEDBACK_ON_LINE_2 AND "DB21033_PF_2_HOPPERS_UNIT_02".DATA.FEEDBACK_ON_LINE_2,
                           NO_POWDER_FLOW_ALARM => "DB426_ALARMS_WARNINGS".CLADDING_POWDER_FEEDER."718143",
                           WARNING_LIMIT => "DB426_ALARMS_WARNINGS".WARNINGS."729905");
END_REGION
END_FUNCTION

FUNCTION_BLOCK "FB21200_POWDER_FLOW_SENSOR_MEDICOAT"   // FB21200, LAD
{ S7_Optimized_Access := 'FALSE' }
VERSION : 0.1
// stored: AutoNumber false, IsIECCheckEnabled false, SetENOAutomatically false, UDAEnableTagReadback false
   VAR_INPUT
      ANALOG_VALUE : Int;   // SENSOR VALUE INPUT
      TIMER_1 : Timer;   // TIMER FOR NOT FLOW ALARM
      POWDER_FEEDER_ON { ExternalVisible := 'False'; ExternalWritable := 'False'} : Bool;   // POWDER FEEDER SWITCHED ON
   END_VAR
   VAR_OUTPUT
      POWDER_FLOW_ON : Bool;   // POWDER FLOW OK
      NO_POWDER_FLOW_ALARM : Bool;   // NO POWDER FLOW ALARM
      WARNING_LIMIT : Bool;   // WARNING FLOW OUT OF LIMITS
      ERROR_CONFIGURATION : Bool;   // WRONG CONFIGURATION ERROR
   END_VAR
   VAR DB_SPECIFIC
      OUTPUT : Struct
         VALUE_REAL : Real;   // POWDER FLOW VALUE
         VALUE_INT : Int;
      END_STRUCT;
      INPUT_SETTINGS : Struct
         LOW_RANGE : Real;   // LOWER VALUE TO SCALE ANALOG SIGNAL
         HIGH_RANGE : Real;   // HIGHER VALUE TO SCALE ANALOG SIGNAL
         LOW_LIMIT_TO_POWDER_FLOW_ON : Real;   // MINIMUM VALUE TO POWDER FLOW OK
         UNIT_NUMBER : Int;
         FEEDER_NUMBER : Int;
      END_STRUCT;
      ALARMS_SETTINGS : Struct
         WARN_LIMIT_LOW : Real;   // LOWER LIMIT FOR WARNING
         WARN_LIMIT_HIGH : Real;   // HIGHER LIMIT FOR WARNING
      END_STRUCT;
      LOG : Struct
         DATE_MAX_MASS : Date_And_Time;
         VALUE_MAX_MASS : Real;
      END_STRUCT;
   END_VAR
   VAR_TEMP
      NORM_VALUE : Real;
      RETVAL : Word;
      DB_NUMBER : DInt;
   END_VAR
   VAR_TEMP   // added for the SCL form of the ladder/FBD networks
      _w1 : Bool;
      _s5time1 : S5Time;
   END_VAR
BEGIN

NETWORK
TITLE = READ INSTANCE DB NUMBER
      L     DINO;
      +     10#800000;
      T     #DB_NUMBER;

REGION Network 2: INPUTS
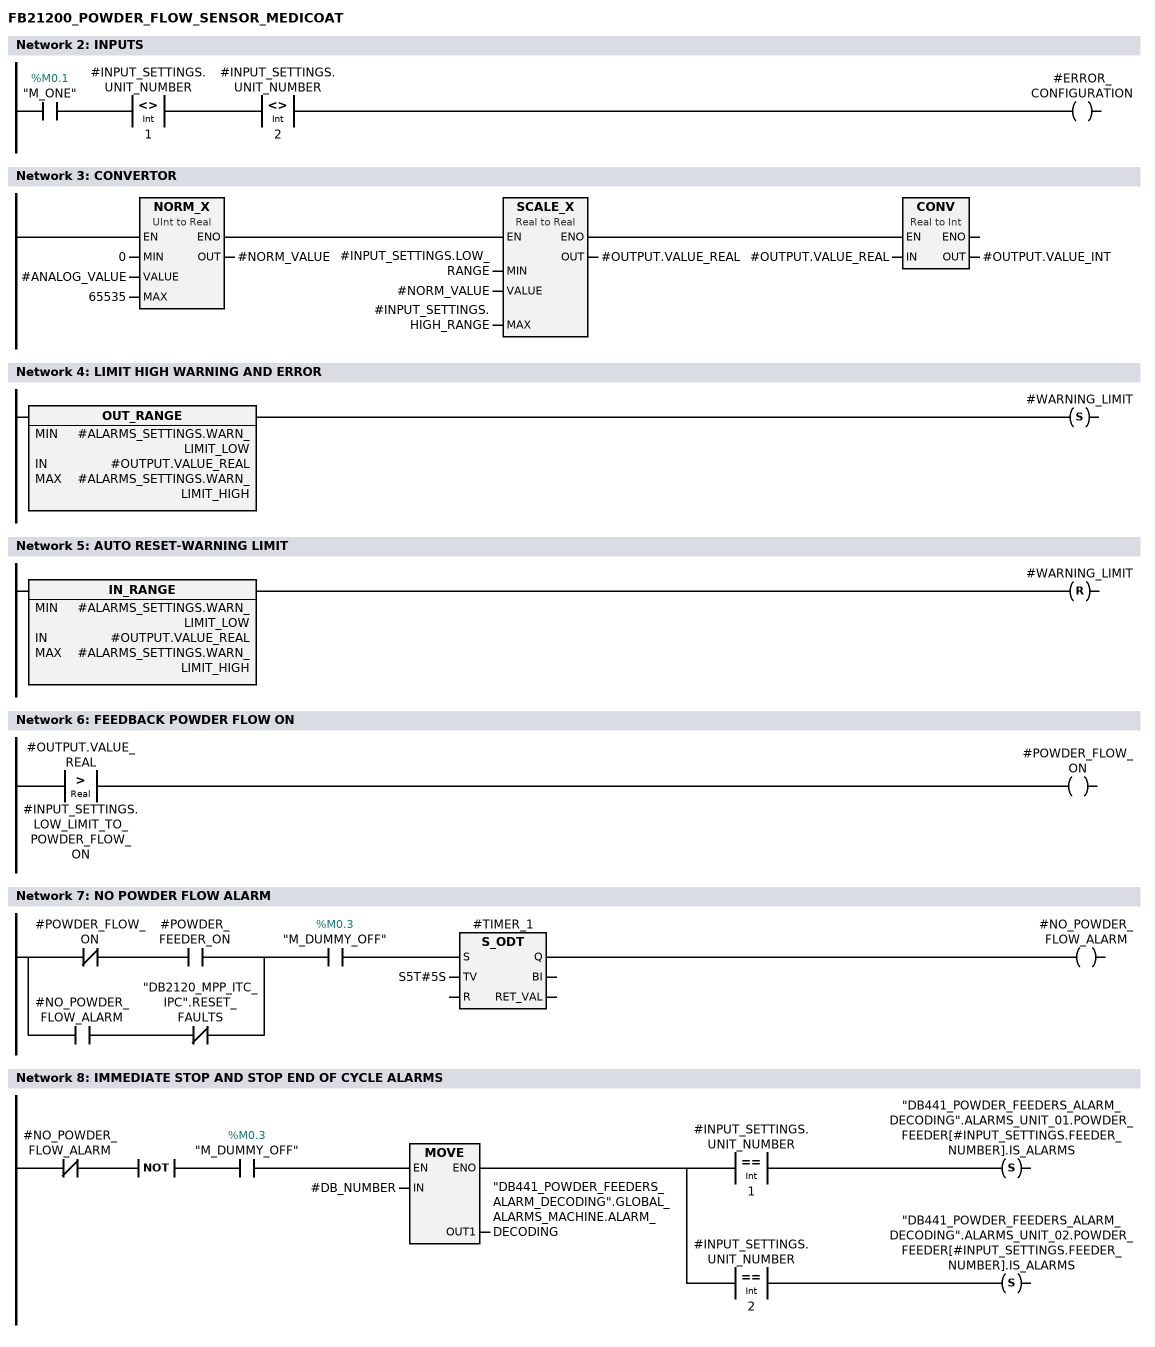
   RUNG wire#powerrail
      Contact( "M_ONE" )
      { S7_Templates := "SrcType := Int" } NE_Contact(in1 := #INPUT_SETTINGS.UNIT_NUMBER, in2 := 1)
      { S7_Templates := "SrcType := Int" } NE_Contact(in1 := #INPUT_SETTINGS.UNIT_NUMBER, in2 := 2)
      Coil( #ERROR_CONFIGURATION )
   END_RUNG
   // the same network as SCL:
   #ERROR_CONFIGURATION := "M_ONE" AND (#INPUT_SETTINGS.UNIT_NUMBER <> 1) AND (#INPUT_SETTINGS.UNIT_NUMBER <> 2);
END_REGION

REGION Network 3: CONVERTOR
   RUNG wire#powerrail
      { S7_Templates := "[SrcType := UInt, DestType := Real]" } Normalize(min := 0, value := #ANALOG_VALUE, max := 65535, out => #NORM_VALUE)
      { S7_Templates := "[SrcType := Real, DestType := Real]" } Scale(min := #INPUT_SETTINGS.LOW_RANGE, value := #NORM_VALUE, max := #INPUT_SETTINGS.HIGH_RANGE, out => #OUTPUT.VALUE_REAL)
      { S7_Templates := "[SrcType := Real, DestType := Int]" } Convert(in := #OUTPUT.VALUE_REAL, out => #OUTPUT.VALUE_INT)
   END_RUNG
   // the same network as SCL:
   #NORM_VALUE := NORM_X(MIN := 0, VALUE := #ANALOG_VALUE, MAX := 65535);
   #OUTPUT.VALUE_REAL := SCALE_X(MIN := #INPUT_SETTINGS.LOW_RANGE, VALUE := #NORM_VALUE, MAX := #INPUT_SETTINGS.HIGH_RANGE);
   #OUTPUT.VALUE_INT := REAL_TO_INT(#OUTPUT.VALUE_REAL);
END_REGION

REGION Network 4: LIMIT HIGH WARNING AND ERROR
   IF (#OUTPUT.VALUE_REAL < #ALARMS_SETTINGS.WARN_LIMIT_LOW) OR (#OUTPUT.VALUE_REAL > #ALARMS_SETTINGS.WARN_LIMIT_HIGH) THEN
       #WARNING_LIMIT := TRUE;
   END_IF;
END_REGION

REGION Network 5: AUTO RESET-WARNING LIMIT
   RUNG wire#powerrail
      { S7_Templates := "SrcType := Real" } InRange(min := #ALARMS_SETTINGS.WARN_LIMIT_LOW, in := #OUTPUT.VALUE_REAL, max := #ALARMS_SETTINGS.WARN_LIMIT_HIGH)
      R_Coil( #WARNING_LIMIT )
   END_RUNG
   // the same network as SCL:
   IF (#ALARMS_SETTINGS.WARN_LIMIT_LOW <= #OUTPUT.VALUE_REAL) AND (#OUTPUT.VALUE_REAL <= #ALARMS_SETTINGS.WARN_LIMIT_HIGH) THEN
       #WARNING_LIMIT := FALSE;
   END_IF;
END_REGION

REGION Network 6: FEEDBACK POWDER FLOW ON
   RUNG wire#powerrail
      { S7_Templates := "SrcType := Real" } GT_Contact(in1 := #OUTPUT.VALUE_REAL, in2 := #INPUT_SETTINGS.LOW_LIMIT_TO_POWDER_FLOW_ON)
      Coil( #POWDER_FLOW_ON )
   END_RUNG
   // the same network as SCL:
   #POWDER_FLOW_ON := #OUTPUT.VALUE_REAL > #INPUT_SETTINGS.LOW_LIMIT_TO_POWDER_FLOW_ON;
END_REGION

REGION Network 7: NO POWDER FLOW ALARM
   RUNG wire#powerrail
      I_Contact( #POWDER_FLOW_ON )
      Contact( #POWDER_FEEDER_ON )
      wire#w1
      Contact( "M_DUMMY_OFF" )
      S_ODT(T_NO := #TIMER_1, TV := S5T#5S, R :=, BI =>, RET_VAL =>)
      Coil( #NO_POWDER_FLOW_ALARM )
   END_RUNG
   RUNG wire#powerrail
      Contact( #NO_POWDER_FLOW_ALARM )
      I_Contact( "DB2120_MPP_ITC_IPC".RESET_FAULTS )
   END_RUNG wire#w1
   // the same network as SCL:
   #_s5time1 := S_ODT(T_NO := #TIMER_1,
                      S := ((NOT #POWDER_FLOW_ON AND #POWDER_FEEDER_ON) OR (#NO_POWDER_FLOW_ALARM AND NOT "DB2120_MPP_ITC_IPC".RESET_FAULTS)) AND "M_DUMMY_OFF",
                      TV := S5T#5S,
                      Q => #_w1);
   #NO_POWDER_FLOW_ALARM := #_w1;
END_REGION

REGION Network 8: IMMEDIATE STOP AND STOP END OF CYCLE ALARMS
   RUNG wire#powerrail
      I_Contact( #NO_POWDER_FLOW_ALARM )
      Not()
      Contact( "M_DUMMY_OFF" )
      Move(in := #DB_NUMBER, out1 => "DB441_POWDER_FEEDERS_ALARM_DECODING".GLOBAL_ALARMS_MACHINE.ALARM_DECODING)
      wire#w1
      { S7_Templates := "SrcType := Int" } EQ_Contact(in1 := #INPUT_SETTINGS.UNIT_NUMBER, in2 := 1)
      S_Coil( "DB441_POWDER_FEEDERS_ALARM_DECODING".ALARMS_UNIT_01.POWDER_FEEDER[#INPUT_SETTINGS.FEEDER_NUMBER].IS_ALARMS )
   END_RUNG
   RUNG wire#w1
      { S7_Templates := "SrcType := Int" } EQ_Contact(in1 := #INPUT_SETTINGS.UNIT_NUMBER, in2 := 2)
      S_Coil( "DB441_POWDER_FEEDERS_ALARM_DECODING".ALARMS_UNIT_02.POWDER_FEEDER[#INPUT_SETTINGS.FEEDER_NUMBER].IS_ALARMS )
   END_RUNG
   // the same network as SCL:
   #_w1 := NOT (NOT #NO_POWDER_FLOW_ALARM) AND "M_DUMMY_OFF";
   IF #_w1 THEN
       "DB441_POWDER_FEEDERS_ALARM_DECODING".GLOBAL_ALARMS_MACHINE.ALARM_DECODING := #DB_NUMBER;
   END_IF;
   IF #_w1 AND (#INPUT_SETTINGS.UNIT_NUMBER = 1) THEN
       "DB441_POWDER_FEEDERS_ALARM_DECODING".ALARMS_UNIT_01.POWDER_FEEDER[#INPUT_SETTINGS.FEEDER_NUMBER].IS_ALARMS := TRUE;
   END_IF;
   IF #_w1 AND (#INPUT_SETTINGS.UNIT_NUMBER = 2) THEN
       "DB441_POWDER_FEEDERS_ALARM_DECODING".ALARMS_UNIT_02.POWDER_FEEDER[#INPUT_SETTINGS.FEEDER_NUMBER].IS_ALARMS := TRUE;
   END_IF;
END_REGION
END_FUNCTION_BLOCK

FUNCTION_BLOCK "FB21222_POWDER_FILLING_START_STOP_BY_CURRENT"   // FB21222, LAD
{ S7_Optimized_Access := 'TRUE' }
VERSION : 0.1
// stored: AutoNumber false, IsIECCheckEnabled false, IsRetainMemResEnabled false, MemoryReserve 100, SetENOAutomatically false, UDAEnableTagReadback false
   VAR_INPUT
      SENSOR_VALUE : Int;   // SENSOR VALUE
      iFEEDER_STATE_LINE : Word;
      HMI_HIGH_CURRENT_LIMIT : Real;   // HMI HIGH CURRENT LIMIT
      HMI_LOW_CURRENT_LIMIT : Real;   // HMI LOW CURRENT LIMIT
   END_VAR
   VAR_OUTPUT
      POWDER_FILLING_STOP_BY_CURRENT : Bool;   // HMI POWDER FILLING STOP BY CURRENT
      POWDER_FILLING_START_BY_CURRENT : Bool;   // HMI POWDER FILLING START BY CURRENT
   END_VAR
   VAR
      CURRENT_AVG_BLCK_START : Real;   // CURRENT AVERAGE BLOCK START
      CURRENT_AVG_BLCK_STOP : Real;   // CURRENT AVERAGE BLOCK STOP
      CURRENT_AVG_BLCK_HMI_START : Real;   // CURRENT AVERAGE BLOCK HMI START
      CURRENT_AVG_BLCK_HMI_STOP : Real;   // CURRENT AVERAGE BLOCK HMI STOP
      PF_LINE_ON : Bool;   // POWDER FEEDER LINE ON
      NORMALIZED_VALUE : Real;   // NORMALIZED
      SCALED_VALUE : Real;   // SCALED
      DB_CURRENT_AVERAGE_START : "FB21990_LGF_FloatingAverage";
      DB_CURRENT_AVERAGE_STOP { S7_SetPoint := 'True'} : "FB21990_LGF_FloatingAverage";
      TON_TIME { S7_SetPoint := 'True'} : TON_TIME;
   END_VAR
   VAR_TEMP   // added for the SCL form of the ladder/FBD networks
      _w1 : Bool;
   END_VAR
BEGIN

REGION Network 1: SCALE - CURRENT VALUE
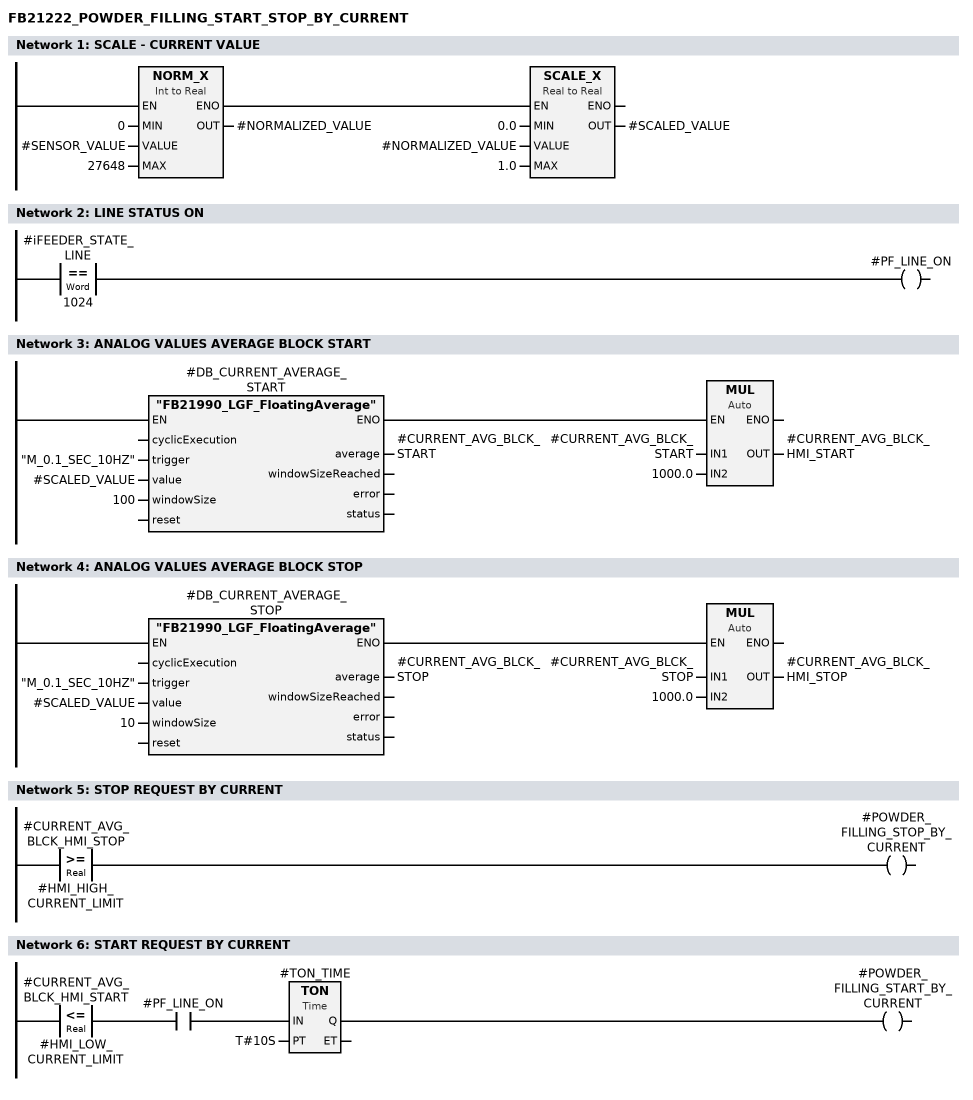
   RUNG wire#powerrail
      { S7_Templates := "[SrcType := Int, DestType := Real]"; S7_GenerateENO := "TRUE" } Normalize(min := 0, value := #SENSOR_VALUE, max := 27648, out => #NORMALIZED_VALUE)
      { S7_Templates := "[SrcType := Real, DestType := Real]"; S7_GenerateENO := "TRUE" } Scale(min := 0.0, value := #NORMALIZED_VALUE, max := 1.0, out => #SCALED_VALUE)
   END_RUNG
   // the same network as SCL:
   // ENO of a box is taken as its EN; it also drops when the box reports an error
   #NORMALIZED_VALUE := NORM_X(MIN := 0, VALUE := #SENSOR_VALUE, MAX := 27648);
   #SCALED_VALUE := SCALE_X(MIN := 0.0, VALUE := #NORMALIZED_VALUE, MAX := 1.0);
END_REGION

REGION Network 2: LINE STATUS ON
   RUNG wire#powerrail
      { S7_Templates := "SrcType := Word" } EQ_Contact(in1 := #iFEEDER_STATE_LINE, in2 := 1024)
      Coil( #PF_LINE_ON )
   END_RUNG
   // the same network as SCL:
   #PF_LINE_ON := #iFEEDER_STATE_LINE = 1024;
END_REGION

REGION Network 3: ANALOG VALUES AVERAGE BLOCK START
   RUNG wire#powerrail
      #DB_CURRENT_AVERAGE_START(cyclicExecution :=, trigger := "M_0.1_SEC_10HZ", value := #SCALED_VALUE, windowSize := 100, reset :=, average => #CURRENT_AVG_BLCK_START, windowSizeReached =>, error =>, status =>)
      { S7_GenerateENO := "TRUE" } Mul(in1 := #CURRENT_AVG_BLCK_START, in2 := 1000.0, out => #CURRENT_AVG_BLCK_HMI_START)
   END_RUNG
   // the same network as SCL:
   #DB_CURRENT_AVERAGE_START(trigger := "M_0.1_SEC_10HZ",   // "FB21990_LGF_FloatingAverage"
                           value := #SCALED_VALUE,
                           windowSize := 100,
                           average => #CURRENT_AVG_BLCK_START,
                           ENO => #_w1);
   IF #_w1 THEN #CURRENT_AVG_BLCK_HMI_START := #CURRENT_AVG_BLCK_START * 1000.0; END_IF;
END_REGION

REGION Network 4: ANALOG VALUES AVERAGE BLOCK STOP
   RUNG wire#powerrail
      #DB_CURRENT_AVERAGE_STOP(cyclicExecution :=, trigger := "M_0.1_SEC_10HZ", value := #SCALED_VALUE, windowSize := 10, reset :=, average => #CURRENT_AVG_BLCK_STOP, windowSizeReached =>, error =>, status =>)
      { S7_GenerateENO := "TRUE" } Mul(in1 := #CURRENT_AVG_BLCK_STOP, in2 := 1000.0, out => #CURRENT_AVG_BLCK_HMI_STOP)
   END_RUNG
   // the same network as SCL:
   #DB_CURRENT_AVERAGE_STOP(trigger := "M_0.1_SEC_10HZ",   // "FB21990_LGF_FloatingAverage"
                           value := #SCALED_VALUE,
                           windowSize := 10,
                           average => #CURRENT_AVG_BLCK_STOP,
                           ENO => #_w1);
   IF #_w1 THEN #CURRENT_AVG_BLCK_HMI_STOP := #CURRENT_AVG_BLCK_STOP * 1000.0; END_IF;
END_REGION

REGION Network 5: STOP REQUEST BY CURRENT
   RUNG wire#powerrail
      { S7_Templates := "SrcType := Real" } GE_Contact(in1 := #CURRENT_AVG_BLCK_HMI_STOP, in2 := #HMI_HIGH_CURRENT_LIMIT)
      Coil( #POWDER_FILLING_STOP_BY_CURRENT )
   END_RUNG
   // the same network as SCL:
   #POWDER_FILLING_STOP_BY_CURRENT := #CURRENT_AVG_BLCK_HMI_STOP >= #HMI_HIGH_CURRENT_LIMIT;
END_REGION

REGION Network 6: START REQUEST BY CURRENT
   RUNG wire#powerrail
      { S7_Templates := "SrcType := Real" } LE_Contact(in1 := #CURRENT_AVG_BLCK_HMI_START, in2 := #HMI_LOW_CURRENT_LIMIT)
      Contact( #PF_LINE_ON )
      { S7_Templates := "time_type := Time" } #TON_TIME.TON(pt := T#10S, et =>)
      Coil( #POWDER_FILLING_START_BY_CURRENT )
   END_RUNG
   // the same network as SCL:
   #TON_TIME(IN := (#CURRENT_AVG_BLCK_HMI_START <= #HMI_LOW_CURRENT_LIMIT) AND #PF_LINE_ON, PT := T#10S);   // TON
   #POWDER_FILLING_START_BY_CURRENT := #TON_TIME.Q;
END_REGION
END_FUNCTION_BLOCK

FUNCTION "FC22000_HOPPER_SYSTEM_MAIN" : Void   // FC22000, LAD
TITLE = FC22000 HOPPER SYSTEM MAIN
{ S7_Optimized_Access := 'TRUE' }
VERSION : 0.1
// stored: AutoNumber false, IsIECCheckEnabled false, SetENOAutomatically false, UDAEnableTagReadback false
BEGIN

REGION Network 1: FC22100_HOPPER_SYSTEM_SENSORS
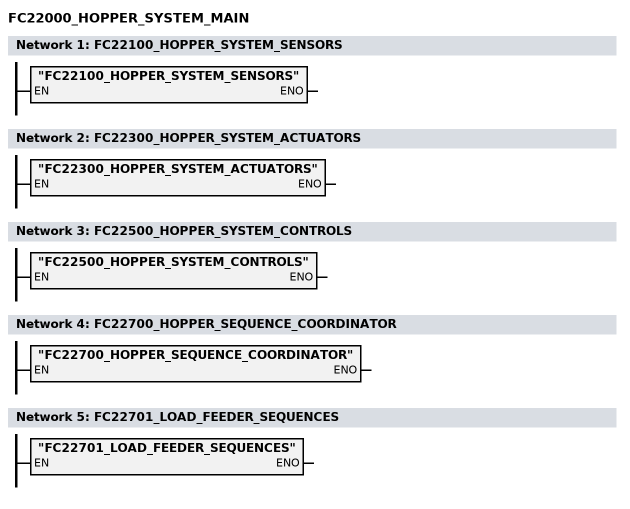
   RUNG wire#powerrail
      "FC22100_HOPPER_SYSTEM_SENSORS"()
   END_RUNG
   // the same network as SCL:
   "FC22100_HOPPER_SYSTEM_SENSORS"();
END_REGION

REGION Network 2: FC22300_HOPPER_SYSTEM_ACTUATORS
   RUNG wire#powerrail
      "FC22300_HOPPER_SYSTEM_ACTUATORS"()
   END_RUNG
   // the same network as SCL:
   "FC22300_HOPPER_SYSTEM_ACTUATORS"();
END_REGION

REGION Network 3: FC22500_HOPPER_SYSTEM_CONTROLS
   RUNG wire#powerrail
      "FC22500_HOPPER_SYSTEM_CONTROLS"()
   END_RUNG
   // the same network as SCL:
   "FC22500_HOPPER_SYSTEM_CONTROLS"();
END_REGION

REGION Network 4: FC22700_HOPPER_SEQUENCE_COORDINATOR
   RUNG wire#powerrail
      "FC22700_HOPPER_SEQUENCE_COORDINATOR"()
   END_RUNG
   // the same network as SCL:
   "FC22700_HOPPER_SEQUENCE_COORDINATOR"();
END_REGION

REGION Network 5: FC22701_LOAD_FEEDER_SEQUENCES
   RUNG wire#powerrail
      "FC22701_LOAD_FEEDER_SEQUENCES"()
   END_RUNG
   // the same network as SCL:
   "FC22701_LOAD_FEEDER_SEQUENCES"();
END_REGION
END_FUNCTION

FUNCTION "FC22100_HOPPER_SYSTEM_SENSORS" : Void   // FC22100, LAD
TITLE = FC22100 HOPPER SYSTEM SENSORS
{ S7_Optimized_Access := 'TRUE' }
VERSION : 0.1
// stored: AutoNumber false, IsIECCheckEnabled false, SetENOAutomatically false, UDAEnableTagReadback false
   VAR CONSTANT
      FC_NUMBER : UInt := 22100;
   END_VAR
   VAR_TEMP   // added for the SCL form of the ladder/FBD networks
      _w1 : Bool;
   END_VAR
BEGIN

REGION Network 1: /////_UNIT_01_SENSORS_/////
END_REGION

REGION Network 2: HOPPER 1 UNIT 01
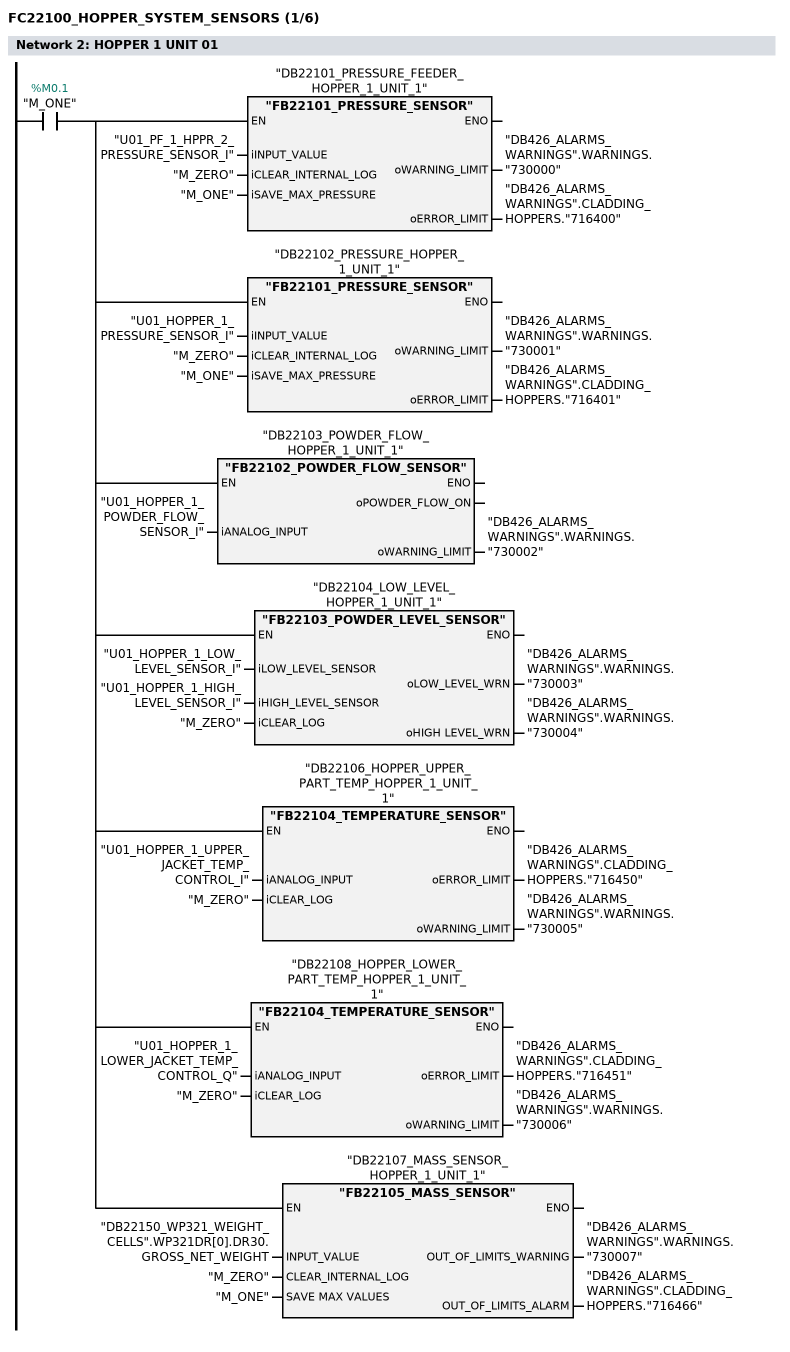
   RUNG wire#powerrail
      Contact( "M_ONE" )
      wire#w1
      "DB22101_PRESSURE_FEEDER_HOPPER_1_UNIT_1"(iINPUT_VALUE := "U01_PF_1_HPPR_2_PRESSURE_SENSOR_I", iCLEAR_INTERNAL_LOG := "M_ZERO", iSAVE_MAX_PRESSURE := "M_ONE", oWARNING_LIMIT => "DB426_ALARMS_WARNINGS".WARNINGS."730000", oERROR_LIMIT => "DB426_ALARMS_WARNINGS".CLADDING_HOPPERS."716400")
   END_RUNG
   RUNG wire#w1
      "DB22102_PRESSURE_HOPPER_1_UNIT_1"(iINPUT_VALUE := "U01_HOPPER_1_PRESSURE_SENSOR_I", iCLEAR_INTERNAL_LOG := "M_ZERO", iSAVE_MAX_PRESSURE := "M_ONE", oWARNING_LIMIT => "DB426_ALARMS_WARNINGS".WARNINGS."730001", oERROR_LIMIT => "DB426_ALARMS_WARNINGS".CLADDING_HOPPERS."716401")
   END_RUNG
   RUNG wire#w1
      "DB22103_POWDER_FLOW_HOPPER_1_UNIT_1"(iANALOG_INPUT := "U01_HOPPER_1_POWDER_FLOW_SENSOR_I", oPOWDER_FLOW_ON =>, oWARNING_LIMIT => "DB426_ALARMS_WARNINGS".WARNINGS."730002")
   END_RUNG
   RUNG wire#w1
      "DB22104_LOW_LEVEL_HOPPER_1_UNIT_1"(iLOW_LEVEL_SENSOR := "U01_HOPPER_1_LOW_LEVEL_SENSOR_I", iHIGH_LEVEL_SENSOR := "U01_HOPPER_1_HIGH_LEVEL_SENSOR_I", iCLEAR_LOG := "M_ZERO", oLOW_LEVEL_WRN => "DB426_ALARMS_WARNINGS".WARNINGS."730003", "oHIGH LEVEL_WRN" => "DB426_ALARMS_WARNINGS".WARNINGS."730004")
   END_RUNG
   RUNG wire#w1
      "DB22106_HOPPER_UPPER_PART_TEMP_HOPPER_1_UNIT_1"(iANALOG_INPUT := "U01_HOPPER_1_UPPER_JACKET_TEMP_CONTROL_I", iCLEAR_LOG := "M_ZERO", oERROR_LIMIT => "DB426_ALARMS_WARNINGS".CLADDING_HOPPERS."716450", oWARNING_LIMIT => "DB426_ALARMS_WARNINGS".WARNINGS."730005")
   END_RUNG
   RUNG wire#w1
      "DB22108_HOPPER_LOWER_PART_TEMP_HOPPER_1_UNIT_1"(iANALOG_INPUT := "U01_HOPPER_1_LOWER_JACKET_TEMP_CONTROL_Q", iCLEAR_LOG := "M_ZERO", oERROR_LIMIT => "DB426_ALARMS_WARNINGS".CLADDING_HOPPERS."716451", oWARNING_LIMIT => "DB426_ALARMS_WARNINGS".WARNINGS."730006")
   END_RUNG
   RUNG wire#w1
      "DB22107_MASS_SENSOR_HOPPER_1_UNIT_1"(INPUT_VALUE := "DB22150_WP321_WEIGHT_CELLS".WP321DR[0].DR30.GROSS_NET_WEIGHT, CLEAR_INTERNAL_LOG := "M_ZERO", "SAVE MAX VALUES" := "M_ONE", OUT_OF_LIMITS_WARNING => "DB426_ALARMS_WARNINGS".WARNINGS."730007", OUT_OF_LIMITS_ALARM => "DB426_ALARMS_WARNINGS".CLADDING_HOPPERS."716466")
   END_RUNG
   // the same network as SCL:
   #_w1 := "M_ONE";
   IF #_w1 THEN
       "DB22101_PRESSURE_FEEDER_HOPPER_1_UNIT_1"(iINPUT_VALUE := "U01_PF_1_HPPR_2_PRESSURE_SENSOR_I",   // "FB22101_PRESSURE_SENSOR"
                               iCLEAR_INTERNAL_LOG := "M_ZERO",
                               iSAVE_MAX_PRESSURE := "M_ONE",
                               oWARNING_LIMIT => "DB426_ALARMS_WARNINGS".WARNINGS."730000",
                               oERROR_LIMIT => "DB426_ALARMS_WARNINGS".CLADDING_HOPPERS."716400");
       "DB22102_PRESSURE_HOPPER_1_UNIT_1"(iINPUT_VALUE := "U01_HOPPER_1_PRESSURE_SENSOR_I",   // "FB22101_PRESSURE_SENSOR"
                               iCLEAR_INTERNAL_LOG := "M_ZERO",
                               iSAVE_MAX_PRESSURE := "M_ONE",
                               oWARNING_LIMIT => "DB426_ALARMS_WARNINGS".WARNINGS."730001",
                               oERROR_LIMIT => "DB426_ALARMS_WARNINGS".CLADDING_HOPPERS."716401");
       "DB22103_POWDER_FLOW_HOPPER_1_UNIT_1"(iANALOG_INPUT := "U01_HOPPER_1_POWDER_FLOW_SENSOR_I",   // "FB22102_POWDER_FLOW_SENSOR"
                               oWARNING_LIMIT => "DB426_ALARMS_WARNINGS".WARNINGS."730002");
       "DB22104_LOW_LEVEL_HOPPER_1_UNIT_1"(iLOW_LEVEL_SENSOR := "U01_HOPPER_1_LOW_LEVEL_SENSOR_I",   // "FB22103_POWDER_LEVEL_SENSOR"
                               iHIGH_LEVEL_SENSOR := "U01_HOPPER_1_HIGH_LEVEL_SENSOR_I",
                               iCLEAR_LOG := "M_ZERO",
                               oLOW_LEVEL_WRN => "DB426_ALARMS_WARNINGS".WARNINGS."730003",
                               "oHIGH LEVEL_WRN" => "DB426_ALARMS_WARNINGS".WARNINGS."730004");
       "DB22106_HOPPER_UPPER_PART_TEMP_HOPPER_1_UNIT_1"(iANALOG_INPUT := "U01_HOPPER_1_UPPER_JACKET_TEMP_CONTROL_I",   // "FB22104_TEMPERATURE_SENSOR"
                               iCLEAR_LOG := "M_ZERO",
                               oERROR_LIMIT => "DB426_ALARMS_WARNINGS".CLADDING_HOPPERS."716450",
                               oWARNING_LIMIT => "DB426_ALARMS_WARNINGS".WARNINGS."730005");
       "DB22108_HOPPER_LOWER_PART_TEMP_HOPPER_1_UNIT_1"(iANALOG_INPUT := "U01_HOPPER_1_LOWER_JACKET_TEMP_CONTROL_Q",   // "FB22104_TEMPERATURE_SENSOR"
                               iCLEAR_LOG := "M_ZERO",
                               oERROR_LIMIT => "DB426_ALARMS_WARNINGS".CLADDING_HOPPERS."716451",
                               oWARNING_LIMIT => "DB426_ALARMS_WARNINGS".WARNINGS."730006");
       "DB22107_MASS_SENSOR_HOPPER_1_UNIT_1"(INPUT_VALUE := "DB22150_WP321_WEIGHT_CELLS".WP321DR[0].DR30.GROSS_NET_WEIGHT,   // "FB22105_MASS_SENSOR"
                               CLEAR_INTERNAL_LOG := "M_ZERO",
                               "SAVE MAX VALUES" := "M_ONE",
                               OUT_OF_LIMITS_WARNING => "DB426_ALARMS_WARNINGS".WARNINGS."730007",
                               OUT_OF_LIMITS_ALARM => "DB426_ALARMS_WARNINGS".CLADDING_HOPPERS."716466");
   END_IF;
END_REGION

REGION Network 3: HOPPER 2 UNIT 01
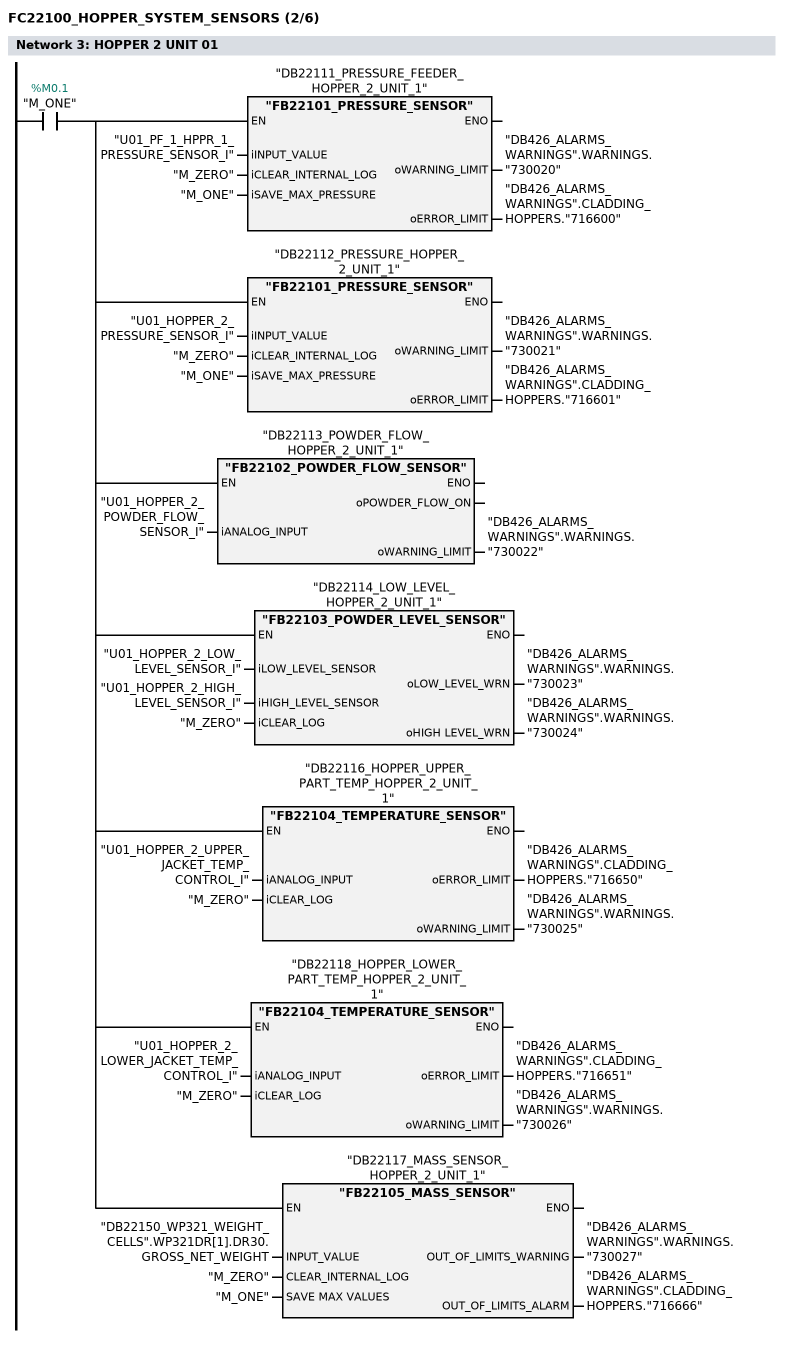
   RUNG wire#powerrail
      Contact( "M_ONE" )
      wire#w1
      "DB22111_PRESSURE_FEEDER_HOPPER_2_UNIT_1"(iINPUT_VALUE := "U01_PF_1_HPPR_1_PRESSURE_SENSOR_I", iCLEAR_INTERNAL_LOG := "M_ZERO", iSAVE_MAX_PRESSURE := "M_ONE", oWARNING_LIMIT => "DB426_ALARMS_WARNINGS".WARNINGS."730020", oERROR_LIMIT => "DB426_ALARMS_WARNINGS".CLADDING_HOPPERS."716600")
   END_RUNG
   RUNG wire#w1
      "DB22112_PRESSURE_HOPPER_2_UNIT_1"(iINPUT_VALUE := "U01_HOPPER_2_PRESSURE_SENSOR_I", iCLEAR_INTERNAL_LOG := "M_ZERO", iSAVE_MAX_PRESSURE := "M_ONE", oWARNING_LIMIT => "DB426_ALARMS_WARNINGS".WARNINGS."730021", oERROR_LIMIT => "DB426_ALARMS_WARNINGS".CLADDING_HOPPERS."716601")
   END_RUNG
   RUNG wire#w1
      "DB22113_POWDER_FLOW_HOPPER_2_UNIT_1"(iANALOG_INPUT := "U01_HOPPER_2_POWDER_FLOW_SENSOR_I", oPOWDER_FLOW_ON =>, oWARNING_LIMIT => "DB426_ALARMS_WARNINGS".WARNINGS."730022")
   END_RUNG
   RUNG wire#w1
      "DB22114_LOW_LEVEL_HOPPER_2_UNIT_1"(iLOW_LEVEL_SENSOR := "U01_HOPPER_2_LOW_LEVEL_SENSOR_I", iHIGH_LEVEL_SENSOR := "U01_HOPPER_2_HIGH_LEVEL_SENSOR_I", iCLEAR_LOG := "M_ZERO", oLOW_LEVEL_WRN => "DB426_ALARMS_WARNINGS".WARNINGS."730023", "oHIGH LEVEL_WRN" => "DB426_ALARMS_WARNINGS".WARNINGS."730024")
   END_RUNG
   RUNG wire#w1
      "DB22116_HOPPER_UPPER_PART_TEMP_HOPPER_2_UNIT_1"(iANALOG_INPUT := "U01_HOPPER_2_UPPER_JACKET_TEMP_CONTROL_I", iCLEAR_LOG := "M_ZERO", oERROR_LIMIT => "DB426_ALARMS_WARNINGS".CLADDING_HOPPERS."716650", oWARNING_LIMIT => "DB426_ALARMS_WARNINGS".WARNINGS."730025")
   END_RUNG
   RUNG wire#w1
      "DB22118_HOPPER_LOWER_PART_TEMP_HOPPER_2_UNIT_1"(iANALOG_INPUT := "U01_HOPPER_2_LOWER_JACKET_TEMP_CONTROL_I", iCLEAR_LOG := "M_ZERO", oERROR_LIMIT => "DB426_ALARMS_WARNINGS".CLADDING_HOPPERS."716651", oWARNING_LIMIT => "DB426_ALARMS_WARNINGS".WARNINGS."730026")
   END_RUNG
   RUNG wire#w1
      "DB22117_MASS_SENSOR_HOPPER_2_UNIT_1"(INPUT_VALUE := "DB22150_WP321_WEIGHT_CELLS".WP321DR[1].DR30.GROSS_NET_WEIGHT, CLEAR_INTERNAL_LOG := "M_ZERO", "SAVE MAX VALUES" := "M_ONE", OUT_OF_LIMITS_WARNING => "DB426_ALARMS_WARNINGS".WARNINGS."730027", OUT_OF_LIMITS_ALARM => "DB426_ALARMS_WARNINGS".CLADDING_HOPPERS."716666")
   END_RUNG
   // the same network as SCL:
   #_w1 := "M_ONE";
   IF #_w1 THEN
       "DB22111_PRESSURE_FEEDER_HOPPER_2_UNIT_1"(iINPUT_VALUE := "U01_PF_1_HPPR_1_PRESSURE_SENSOR_I",   // "FB22101_PRESSURE_SENSOR"
                               iCLEAR_INTERNAL_LOG := "M_ZERO",
                               iSAVE_MAX_PRESSURE := "M_ONE",
                               oWARNING_LIMIT => "DB426_ALARMS_WARNINGS".WARNINGS."730020",
                               oERROR_LIMIT => "DB426_ALARMS_WARNINGS".CLADDING_HOPPERS."716600");
       "DB22112_PRESSURE_HOPPER_2_UNIT_1"(iINPUT_VALUE := "U01_HOPPER_2_PRESSURE_SENSOR_I",   // "FB22101_PRESSURE_SENSOR"
                               iCLEAR_INTERNAL_LOG := "M_ZERO",
                               iSAVE_MAX_PRESSURE := "M_ONE",
                               oWARNING_LIMIT => "DB426_ALARMS_WARNINGS".WARNINGS."730021",
                               oERROR_LIMIT => "DB426_ALARMS_WARNINGS".CLADDING_HOPPERS."716601");
       "DB22113_POWDER_FLOW_HOPPER_2_UNIT_1"(iANALOG_INPUT := "U01_HOPPER_2_POWDER_FLOW_SENSOR_I",   // "FB22102_POWDER_FLOW_SENSOR"
                               oWARNING_LIMIT => "DB426_ALARMS_WARNINGS".WARNINGS."730022");
       "DB22114_LOW_LEVEL_HOPPER_2_UNIT_1"(iLOW_LEVEL_SENSOR := "U01_HOPPER_2_LOW_LEVEL_SENSOR_I",   // "FB22103_POWDER_LEVEL_SENSOR"
                               iHIGH_LEVEL_SENSOR := "U01_HOPPER_2_HIGH_LEVEL_SENSOR_I",
                               iCLEAR_LOG := "M_ZERO",
                               oLOW_LEVEL_WRN => "DB426_ALARMS_WARNINGS".WARNINGS."730023",
                               "oHIGH LEVEL_WRN" => "DB426_ALARMS_WARNINGS".WARNINGS."730024");
       "DB22116_HOPPER_UPPER_PART_TEMP_HOPPER_2_UNIT_1"(iANALOG_INPUT := "U01_HOPPER_2_UPPER_JACKET_TEMP_CONTROL_I",   // "FB22104_TEMPERATURE_SENSOR"
                               iCLEAR_LOG := "M_ZERO",
                               oERROR_LIMIT => "DB426_ALARMS_WARNINGS".CLADDING_HOPPERS."716650",
                               oWARNING_LIMIT => "DB426_ALARMS_WARNINGS".WARNINGS."730025");
       "DB22118_HOPPER_LOWER_PART_TEMP_HOPPER_2_UNIT_1"(iANALOG_INPUT := "U01_HOPPER_2_LOWER_JACKET_TEMP_CONTROL_I",   // "FB22104_TEMPERATURE_SENSOR"
                               iCLEAR_LOG := "M_ZERO",
                               oERROR_LIMIT => "DB426_ALARMS_WARNINGS".CLADDING_HOPPERS."716651",
                               oWARNING_LIMIT => "DB426_ALARMS_WARNINGS".WARNINGS."730026");
       "DB22117_MASS_SENSOR_HOPPER_2_UNIT_1"(INPUT_VALUE := "DB22150_WP321_WEIGHT_CELLS".WP321DR[1].DR30.GROSS_NET_WEIGHT,   // "FB22105_MASS_SENSOR"
                               CLEAR_INTERNAL_LOG := "M_ZERO",
                               "SAVE MAX VALUES" := "M_ONE",
                               OUT_OF_LIMITS_WARNING => "DB426_ALARMS_WARNINGS".WARNINGS."730027",
                               OUT_OF_LIMITS_ALARM => "DB426_ALARMS_WARNINGS".CLADDING_HOPPERS."716666");
   END_IF;
END_REGION

REGION Network 4: /////_UNIT_02_SENSORS_/////
END_REGION

REGION Network 5: HOPPER 1 UNIT 02
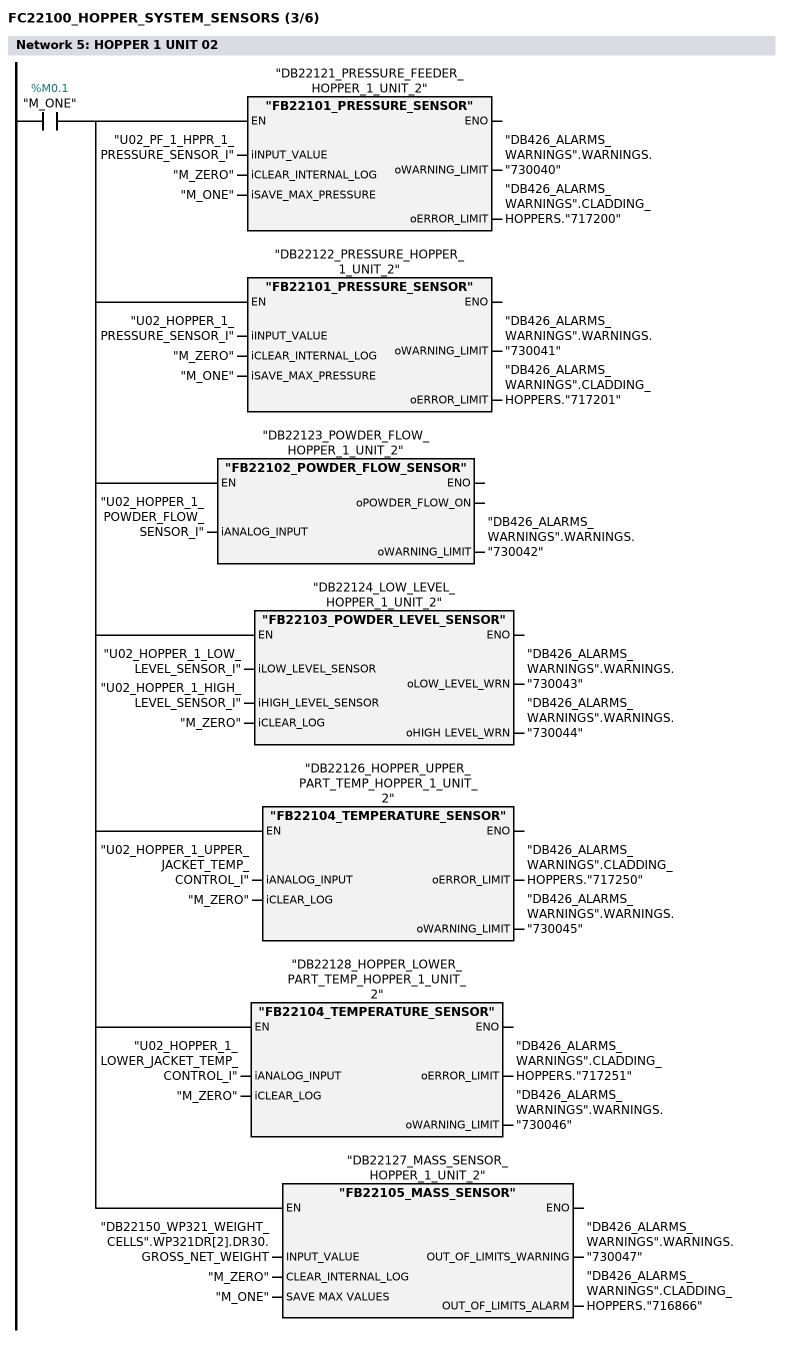
   RUNG wire#powerrail
      Contact( "M_ONE" )
      wire#w1
      "DB22121_PRESSURE_FEEDER_HOPPER_1_UNIT_2"(iINPUT_VALUE := "U02_PF_1_HPPR_1_PRESSURE_SENSOR_I", iCLEAR_INTERNAL_LOG := "M_ZERO", iSAVE_MAX_PRESSURE := "M_ONE", oWARNING_LIMIT => "DB426_ALARMS_WARNINGS".WARNINGS."730040", oERROR_LIMIT => "DB426_ALARMS_WARNINGS".CLADDING_HOPPERS."717200")
   END_RUNG
   RUNG wire#w1
      "DB22122_PRESSURE_HOPPER_1_UNIT_2"(iINPUT_VALUE := "U02_HOPPER_1_PRESSURE_SENSOR_I", iCLEAR_INTERNAL_LOG := "M_ZERO", iSAVE_MAX_PRESSURE := "M_ONE", oWARNING_LIMIT => "DB426_ALARMS_WARNINGS".WARNINGS."730041", oERROR_LIMIT => "DB426_ALARMS_WARNINGS".CLADDING_HOPPERS."717201")
   END_RUNG
   RUNG wire#w1
      "DB22123_POWDER_FLOW_HOPPER_1_UNIT_2"(iANALOG_INPUT := "U02_HOPPER_1_POWDER_FLOW_SENSOR_I", oPOWDER_FLOW_ON =>, oWARNING_LIMIT => "DB426_ALARMS_WARNINGS".WARNINGS."730042")
   END_RUNG
   RUNG wire#w1
      "DB22124_LOW_LEVEL_HOPPER_1_UNIT_2"(iLOW_LEVEL_SENSOR := "U02_HOPPER_1_LOW_LEVEL_SENSOR_I", iHIGH_LEVEL_SENSOR := "U02_HOPPER_1_HIGH_LEVEL_SENSOR_I", iCLEAR_LOG := "M_ZERO", oLOW_LEVEL_WRN => "DB426_ALARMS_WARNINGS".WARNINGS."730043", "oHIGH LEVEL_WRN" => "DB426_ALARMS_WARNINGS".WARNINGS."730044")
   END_RUNG
   RUNG wire#w1
      "DB22126_HOPPER_UPPER_PART_TEMP_HOPPER_1_UNIT_2"(iANALOG_INPUT := "U02_HOPPER_1_UPPER_JACKET_TEMP_CONTROL_I", iCLEAR_LOG := "M_ZERO", oERROR_LIMIT => "DB426_ALARMS_WARNINGS".CLADDING_HOPPERS."717250", oWARNING_LIMIT => "DB426_ALARMS_WARNINGS".WARNINGS."730045")
   END_RUNG
   RUNG wire#w1
      "DB22128_HOPPER_LOWER_PART_TEMP_HOPPER_1_UNIT_2"(iANALOG_INPUT := "U02_HOPPER_1_LOWER_JACKET_TEMP_CONTROL_I", iCLEAR_LOG := "M_ZERO", oERROR_LIMIT => "DB426_ALARMS_WARNINGS".CLADDING_HOPPERS."717251", oWARNING_LIMIT => "DB426_ALARMS_WARNINGS".WARNINGS."730046")
   END_RUNG
   RUNG wire#w1
      "DB22127_MASS_SENSOR_HOPPER_1_UNIT_2"(INPUT_VALUE := "DB22150_WP321_WEIGHT_CELLS".WP321DR[2].DR30.GROSS_NET_WEIGHT, CLEAR_INTERNAL_LOG := "M_ZERO", "SAVE MAX VALUES" := "M_ONE", OUT_OF_LIMITS_WARNING => "DB426_ALARMS_WARNINGS".WARNINGS."730047", OUT_OF_LIMITS_ALARM => "DB426_ALARMS_WARNINGS".CLADDING_HOPPERS."716866")
   END_RUNG
   // the same network as SCL:
   #_w1 := "M_ONE";
   IF #_w1 THEN
       "DB22121_PRESSURE_FEEDER_HOPPER_1_UNIT_2"(iINPUT_VALUE := "U02_PF_1_HPPR_1_PRESSURE_SENSOR_I",   // "FB22101_PRESSURE_SENSOR"
                               iCLEAR_INTERNAL_LOG := "M_ZERO",
                               iSAVE_MAX_PRESSURE := "M_ONE",
                               oWARNING_LIMIT => "DB426_ALARMS_WARNINGS".WARNINGS."730040",
                               oERROR_LIMIT => "DB426_ALARMS_WARNINGS".CLADDING_HOPPERS."717200");
       "DB22122_PRESSURE_HOPPER_1_UNIT_2"(iINPUT_VALUE := "U02_HOPPER_1_PRESSURE_SENSOR_I",   // "FB22101_PRESSURE_SENSOR"
                               iCLEAR_INTERNAL_LOG := "M_ZERO",
                               iSAVE_MAX_PRESSURE := "M_ONE",
                               oWARNING_LIMIT => "DB426_ALARMS_WARNINGS".WARNINGS."730041",
                               oERROR_LIMIT => "DB426_ALARMS_WARNINGS".CLADDING_HOPPERS."717201");
       "DB22123_POWDER_FLOW_HOPPER_1_UNIT_2"(iANALOG_INPUT := "U02_HOPPER_1_POWDER_FLOW_SENSOR_I",   // "FB22102_POWDER_FLOW_SENSOR"
                               oWARNING_LIMIT => "DB426_ALARMS_WARNINGS".WARNINGS."730042");
       "DB22124_LOW_LEVEL_HOPPER_1_UNIT_2"(iLOW_LEVEL_SENSOR := "U02_HOPPER_1_LOW_LEVEL_SENSOR_I",   // "FB22103_POWDER_LEVEL_SENSOR"
                               iHIGH_LEVEL_SENSOR := "U02_HOPPER_1_HIGH_LEVEL_SENSOR_I",
                               iCLEAR_LOG := "M_ZERO",
                               oLOW_LEVEL_WRN => "DB426_ALARMS_WARNINGS".WARNINGS."730043",
                               "oHIGH LEVEL_WRN" => "DB426_ALARMS_WARNINGS".WARNINGS."730044");
       "DB22126_HOPPER_UPPER_PART_TEMP_HOPPER_1_UNIT_2"(iANALOG_INPUT := "U02_HOPPER_1_UPPER_JACKET_TEMP_CONTROL_I",   // "FB22104_TEMPERATURE_SENSOR"
                               iCLEAR_LOG := "M_ZERO",
                               oERROR_LIMIT => "DB426_ALARMS_WARNINGS".CLADDING_HOPPERS."717250",
                               oWARNING_LIMIT => "DB426_ALARMS_WARNINGS".WARNINGS."730045");
       "DB22128_HOPPER_LOWER_PART_TEMP_HOPPER_1_UNIT_2"(iANALOG_INPUT := "U02_HOPPER_1_LOWER_JACKET_TEMP_CONTROL_I",   // "FB22104_TEMPERATURE_SENSOR"
                               iCLEAR_LOG := "M_ZERO",
                               oERROR_LIMIT => "DB426_ALARMS_WARNINGS".CLADDING_HOPPERS."717251",
                               oWARNING_LIMIT => "DB426_ALARMS_WARNINGS".WARNINGS."730046");
       "DB22127_MASS_SENSOR_HOPPER_1_UNIT_2"(INPUT_VALUE := "DB22150_WP321_WEIGHT_CELLS".WP321DR[2].DR30.GROSS_NET_WEIGHT,   // "FB22105_MASS_SENSOR"
                               CLEAR_INTERNAL_LOG := "M_ZERO",
                               "SAVE MAX VALUES" := "M_ONE",
                               OUT_OF_LIMITS_WARNING => "DB426_ALARMS_WARNINGS".WARNINGS."730047",
                               OUT_OF_LIMITS_ALARM => "DB426_ALARMS_WARNINGS".CLADDING_HOPPERS."716866");
   END_IF;
END_REGION

REGION Network 6: HOPPER 2 UNIT 02
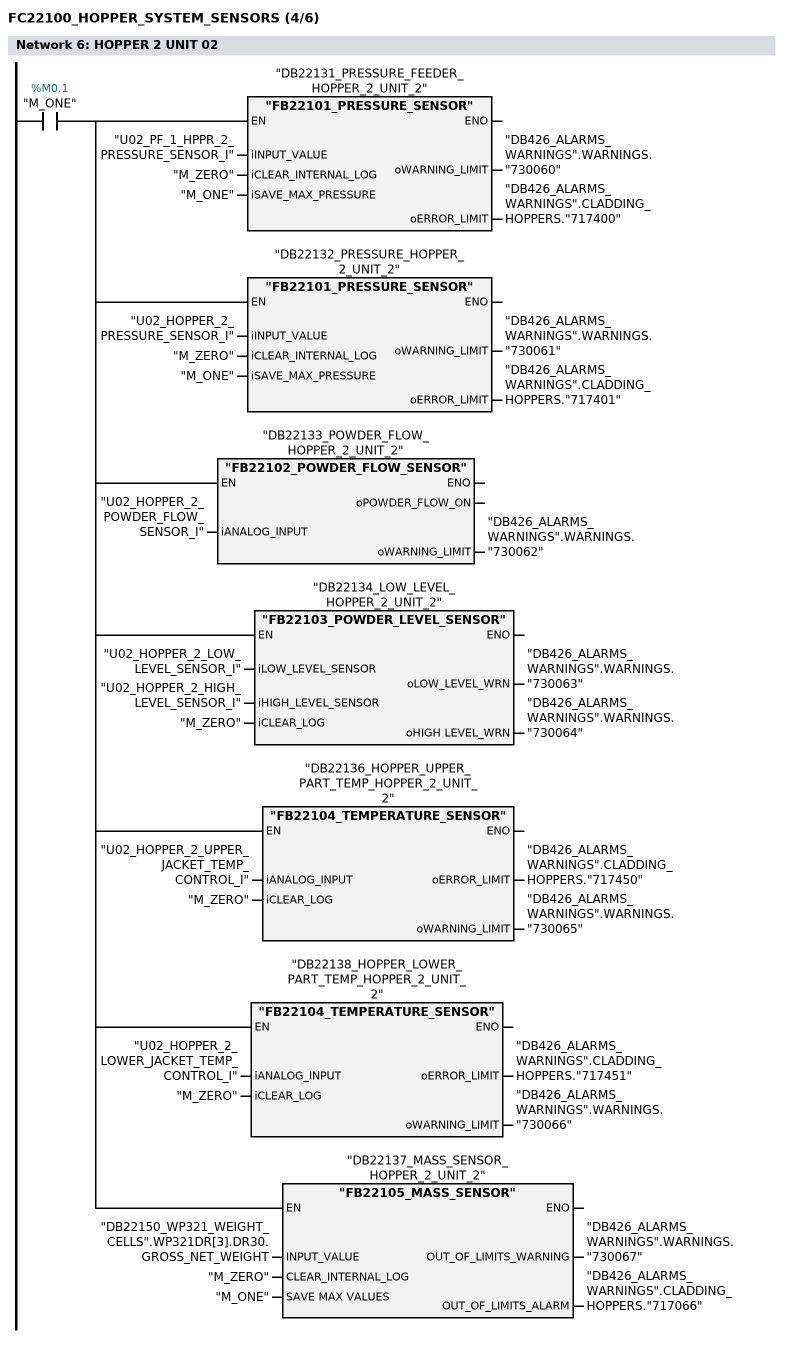
   RUNG wire#powerrail
      Contact( "M_ONE" )
      wire#w1
      "DB22131_PRESSURE_FEEDER_HOPPER_2_UNIT_2"(iINPUT_VALUE := "U02_PF_1_HPPR_2_PRESSURE_SENSOR_I", iCLEAR_INTERNAL_LOG := "M_ZERO", iSAVE_MAX_PRESSURE := "M_ONE", oWARNING_LIMIT => "DB426_ALARMS_WARNINGS".WARNINGS."730060", oERROR_LIMIT => "DB426_ALARMS_WARNINGS".CLADDING_HOPPERS."717400")
   END_RUNG
   RUNG wire#w1
      "DB22132_PRESSURE_HOPPER_2_UNIT_2"(iINPUT_VALUE := "U02_HOPPER_2_PRESSURE_SENSOR_I", iCLEAR_INTERNAL_LOG := "M_ZERO", iSAVE_MAX_PRESSURE := "M_ONE", oWARNING_LIMIT => "DB426_ALARMS_WARNINGS".WARNINGS."730061", oERROR_LIMIT => "DB426_ALARMS_WARNINGS".CLADDING_HOPPERS."717401")
   END_RUNG
   RUNG wire#w1
      "DB22133_POWDER_FLOW_HOPPER_2_UNIT_2"(iANALOG_INPUT := "U02_HOPPER_2_POWDER_FLOW_SENSOR_I", oPOWDER_FLOW_ON =>, oWARNING_LIMIT => "DB426_ALARMS_WARNINGS".WARNINGS."730062")
   END_RUNG
   RUNG wire#w1
      "DB22134_LOW_LEVEL_HOPPER_2_UNIT_2"(iLOW_LEVEL_SENSOR := "U02_HOPPER_2_LOW_LEVEL_SENSOR_I", iHIGH_LEVEL_SENSOR := "U02_HOPPER_2_HIGH_LEVEL_SENSOR_I", iCLEAR_LOG := "M_ZERO", oLOW_LEVEL_WRN => "DB426_ALARMS_WARNINGS".WARNINGS."730063", "oHIGH LEVEL_WRN" => "DB426_ALARMS_WARNINGS".WARNINGS."730064")
   END_RUNG
   RUNG wire#w1
      "DB22136_HOPPER_UPPER_PART_TEMP_HOPPER_2_UNIT_2"(iANALOG_INPUT := "U02_HOPPER_2_UPPER_JACKET_TEMP_CONTROL_I", iCLEAR_LOG := "M_ZERO", oERROR_LIMIT => "DB426_ALARMS_WARNINGS".CLADDING_HOPPERS."717450", oWARNING_LIMIT => "DB426_ALARMS_WARNINGS".WARNINGS."730065")
   END_RUNG
   RUNG wire#w1
      "DB22138_HOPPER_LOWER_PART_TEMP_HOPPER_2_UNIT_2"(iANALOG_INPUT := "U02_HOPPER_2_LOWER_JACKET_TEMP_CONTROL_I", iCLEAR_LOG := "M_ZERO", oERROR_LIMIT => "DB426_ALARMS_WARNINGS".CLADDING_HOPPERS."717451", oWARNING_LIMIT => "DB426_ALARMS_WARNINGS".WARNINGS."730066")
   END_RUNG
   RUNG wire#w1
      "DB22137_MASS_SENSOR_HOPPER_2_UNIT_2"(INPUT_VALUE := "DB22150_WP321_WEIGHT_CELLS".WP321DR[3].DR30.GROSS_NET_WEIGHT, CLEAR_INTERNAL_LOG := "M_ZERO", "SAVE MAX VALUES" := "M_ONE", OUT_OF_LIMITS_WARNING => "DB426_ALARMS_WARNINGS".WARNINGS."730067", OUT_OF_LIMITS_ALARM => "DB426_ALARMS_WARNINGS".CLADDING_HOPPERS."717066")
   END_RUNG
   // the same network as SCL:
   #_w1 := "M_ONE";
   IF #_w1 THEN
       "DB22131_PRESSURE_FEEDER_HOPPER_2_UNIT_2"(iINPUT_VALUE := "U02_PF_1_HPPR_2_PRESSURE_SENSOR_I",   // "FB22101_PRESSURE_SENSOR"
                               iCLEAR_INTERNAL_LOG := "M_ZERO",
                               iSAVE_MAX_PRESSURE := "M_ONE",
                               oWARNING_LIMIT => "DB426_ALARMS_WARNINGS".WARNINGS."730060",
                               oERROR_LIMIT => "DB426_ALARMS_WARNINGS".CLADDING_HOPPERS."717400");
       "DB22132_PRESSURE_HOPPER_2_UNIT_2"(iINPUT_VALUE := "U02_HOPPER_2_PRESSURE_SENSOR_I",   // "FB22101_PRESSURE_SENSOR"
                               iCLEAR_INTERNAL_LOG := "M_ZERO",
                               iSAVE_MAX_PRESSURE := "M_ONE",
                               oWARNING_LIMIT => "DB426_ALARMS_WARNINGS".WARNINGS."730061",
                               oERROR_LIMIT => "DB426_ALARMS_WARNINGS".CLADDING_HOPPERS."717401");
       "DB22133_POWDER_FLOW_HOPPER_2_UNIT_2"(iANALOG_INPUT := "U02_HOPPER_2_POWDER_FLOW_SENSOR_I",   // "FB22102_POWDER_FLOW_SENSOR"
                               oWARNING_LIMIT => "DB426_ALARMS_WARNINGS".WARNINGS."730062");
       "DB22134_LOW_LEVEL_HOPPER_2_UNIT_2"(iLOW_LEVEL_SENSOR := "U02_HOPPER_2_LOW_LEVEL_SENSOR_I",   // "FB22103_POWDER_LEVEL_SENSOR"
                               iHIGH_LEVEL_SENSOR := "U02_HOPPER_2_HIGH_LEVEL_SENSOR_I",
                               iCLEAR_LOG := "M_ZERO",
                               oLOW_LEVEL_WRN => "DB426_ALARMS_WARNINGS".WARNINGS."730063",
                               "oHIGH LEVEL_WRN" => "DB426_ALARMS_WARNINGS".WARNINGS."730064");
       "DB22136_HOPPER_UPPER_PART_TEMP_HOPPER_2_UNIT_2"(iANALOG_INPUT := "U02_HOPPER_2_UPPER_JACKET_TEMP_CONTROL_I",   // "FB22104_TEMPERATURE_SENSOR"
                               iCLEAR_LOG := "M_ZERO",
                               oERROR_LIMIT => "DB426_ALARMS_WARNINGS".CLADDING_HOPPERS."717450",
                               oWARNING_LIMIT => "DB426_ALARMS_WARNINGS".WARNINGS."730065");
       "DB22138_HOPPER_LOWER_PART_TEMP_HOPPER_2_UNIT_2"(iANALOG_INPUT := "U02_HOPPER_2_LOWER_JACKET_TEMP_CONTROL_I",   // "FB22104_TEMPERATURE_SENSOR"
                               iCLEAR_LOG := "M_ZERO",
                               oERROR_LIMIT => "DB426_ALARMS_WARNINGS".CLADDING_HOPPERS."717451",
                               oWARNING_LIMIT => "DB426_ALARMS_WARNINGS".WARNINGS."730066");
       "DB22137_MASS_SENSOR_HOPPER_2_UNIT_2"(INPUT_VALUE := "DB22150_WP321_WEIGHT_CELLS".WP321DR[3].DR30.GROSS_NET_WEIGHT,   // "FB22105_MASS_SENSOR"
                               CLEAR_INTERNAL_LOG := "M_ZERO",
                               "SAVE MAX VALUES" := "M_ONE",
                               OUT_OF_LIMITS_WARNING => "DB426_ALARMS_WARNINGS".WARNINGS."730067",
                               OUT_OF_LIMITS_ALARM => "DB426_ALARMS_WARNINGS".CLADDING_HOPPERS."717066");
   END_IF;
END_REGION

REGION Network 7: HOPPER 3 UNIT 02
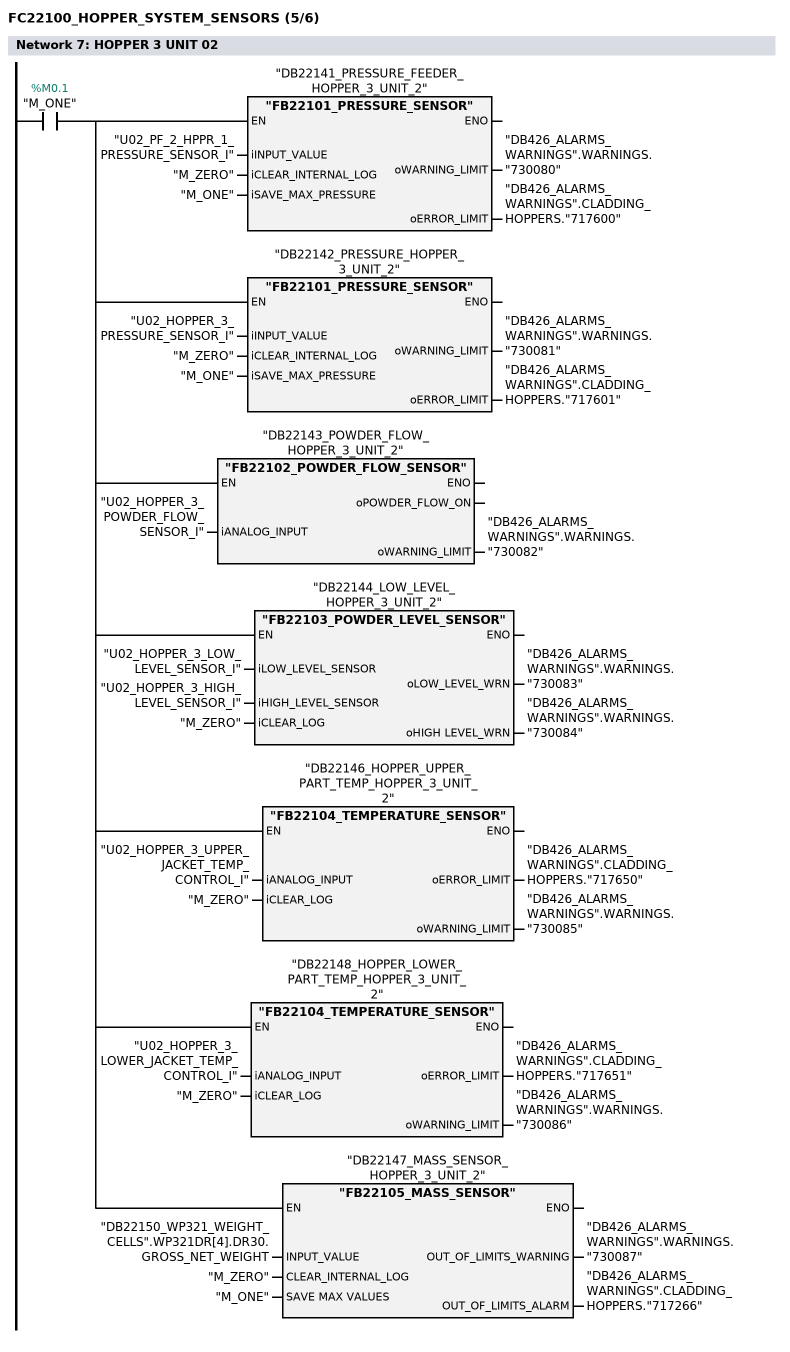
   RUNG wire#powerrail
      Contact( "M_ONE" )
      wire#w1
      "DB22141_PRESSURE_FEEDER_HOPPER_3_UNIT_2"(iINPUT_VALUE := "U02_PF_2_HPPR_1_PRESSURE_SENSOR_I", iCLEAR_INTERNAL_LOG := "M_ZERO", iSAVE_MAX_PRESSURE := "M_ONE", oWARNING_LIMIT => "DB426_ALARMS_WARNINGS".WARNINGS."730080", oERROR_LIMIT => "DB426_ALARMS_WARNINGS".CLADDING_HOPPERS."717600")
   END_RUNG
   RUNG wire#w1
      "DB22142_PRESSURE_HOPPER_3_UNIT_2"(iINPUT_VALUE := "U02_HOPPER_3_PRESSURE_SENSOR_I", iCLEAR_INTERNAL_LOG := "M_ZERO", iSAVE_MAX_PRESSURE := "M_ONE", oWARNING_LIMIT => "DB426_ALARMS_WARNINGS".WARNINGS."730081", oERROR_LIMIT => "DB426_ALARMS_WARNINGS".CLADDING_HOPPERS."717601")
   END_RUNG
   RUNG wire#w1
      "DB22143_POWDER_FLOW_HOPPER_3_UNIT_2"(iANALOG_INPUT := "U02_HOPPER_3_POWDER_FLOW_SENSOR_I", oPOWDER_FLOW_ON =>, oWARNING_LIMIT => "DB426_ALARMS_WARNINGS".WARNINGS."730082")
   END_RUNG
   RUNG wire#w1
      "DB22144_LOW_LEVEL_HOPPER_3_UNIT_2"(iLOW_LEVEL_SENSOR := "U02_HOPPER_3_LOW_LEVEL_SENSOR_I", iHIGH_LEVEL_SENSOR := "U02_HOPPER_3_HIGH_LEVEL_SENSOR_I", iCLEAR_LOG := "M_ZERO", oLOW_LEVEL_WRN => "DB426_ALARMS_WARNINGS".WARNINGS."730083", "oHIGH LEVEL_WRN" => "DB426_ALARMS_WARNINGS".WARNINGS."730084")
   END_RUNG
   RUNG wire#w1
      "DB22146_HOPPER_UPPER_PART_TEMP_HOPPER_3_UNIT_2"(iANALOG_INPUT := "U02_HOPPER_3_UPPER_JACKET_TEMP_CONTROL_I", iCLEAR_LOG := "M_ZERO", oERROR_LIMIT => "DB426_ALARMS_WARNINGS".CLADDING_HOPPERS."717650", oWARNING_LIMIT => "DB426_ALARMS_WARNINGS".WARNINGS."730085")
   END_RUNG
   RUNG wire#w1
      "DB22148_HOPPER_LOWER_PART_TEMP_HOPPER_3_UNIT_2"(iANALOG_INPUT := "U02_HOPPER_3_LOWER_JACKET_TEMP_CONTROL_I", iCLEAR_LOG := "M_ZERO", oERROR_LIMIT => "DB426_ALARMS_WARNINGS".CLADDING_HOPPERS."717651", oWARNING_LIMIT => "DB426_ALARMS_WARNINGS".WARNINGS."730086")
   END_RUNG
   RUNG wire#w1
      "DB22147_MASS_SENSOR_HOPPER_3_UNIT_2"(INPUT_VALUE := "DB22150_WP321_WEIGHT_CELLS".WP321DR[4].DR30.GROSS_NET_WEIGHT, CLEAR_INTERNAL_LOG := "M_ZERO", "SAVE MAX VALUES" := "M_ONE", OUT_OF_LIMITS_WARNING => "DB426_ALARMS_WARNINGS".WARNINGS."730087", OUT_OF_LIMITS_ALARM => "DB426_ALARMS_WARNINGS".CLADDING_HOPPERS."717266")
   END_RUNG
   // the same network as SCL:
   #_w1 := "M_ONE";
   IF #_w1 THEN
       "DB22141_PRESSURE_FEEDER_HOPPER_3_UNIT_2"(iINPUT_VALUE := "U02_PF_2_HPPR_1_PRESSURE_SENSOR_I",   // "FB22101_PRESSURE_SENSOR"
                               iCLEAR_INTERNAL_LOG := "M_ZERO",
                               iSAVE_MAX_PRESSURE := "M_ONE",
                               oWARNING_LIMIT => "DB426_ALARMS_WARNINGS".WARNINGS."730080",
                               oERROR_LIMIT => "DB426_ALARMS_WARNINGS".CLADDING_HOPPERS."717600");
       "DB22142_PRESSURE_HOPPER_3_UNIT_2"(iINPUT_VALUE := "U02_HOPPER_3_PRESSURE_SENSOR_I",   // "FB22101_PRESSURE_SENSOR"
                               iCLEAR_INTERNAL_LOG := "M_ZERO",
                               iSAVE_MAX_PRESSURE := "M_ONE",
                               oWARNING_LIMIT => "DB426_ALARMS_WARNINGS".WARNINGS."730081",
                               oERROR_LIMIT => "DB426_ALARMS_WARNINGS".CLADDING_HOPPERS."717601");
       "DB22143_POWDER_FLOW_HOPPER_3_UNIT_2"(iANALOG_INPUT := "U02_HOPPER_3_POWDER_FLOW_SENSOR_I",   // "FB22102_POWDER_FLOW_SENSOR"
                               oWARNING_LIMIT => "DB426_ALARMS_WARNINGS".WARNINGS."730082");
       "DB22144_LOW_LEVEL_HOPPER_3_UNIT_2"(iLOW_LEVEL_SENSOR := "U02_HOPPER_3_LOW_LEVEL_SENSOR_I",   // "FB22103_POWDER_LEVEL_SENSOR"
                               iHIGH_LEVEL_SENSOR := "U02_HOPPER_3_HIGH_LEVEL_SENSOR_I",
                               iCLEAR_LOG := "M_ZERO",
                               oLOW_LEVEL_WRN => "DB426_ALARMS_WARNINGS".WARNINGS."730083",
                               "oHIGH LEVEL_WRN" => "DB426_ALARMS_WARNINGS".WARNINGS."730084");
       "DB22146_HOPPER_UPPER_PART_TEMP_HOPPER_3_UNIT_2"(iANALOG_INPUT := "U02_HOPPER_3_UPPER_JACKET_TEMP_CONTROL_I",   // "FB22104_TEMPERATURE_SENSOR"
                               iCLEAR_LOG := "M_ZERO",
                               oERROR_LIMIT => "DB426_ALARMS_WARNINGS".CLADDING_HOPPERS."717650",
                               oWARNING_LIMIT => "DB426_ALARMS_WARNINGS".WARNINGS."730085");
       "DB22148_HOPPER_LOWER_PART_TEMP_HOPPER_3_UNIT_2"(iANALOG_INPUT := "U02_HOPPER_3_LOWER_JACKET_TEMP_CONTROL_I",   // "FB22104_TEMPERATURE_SENSOR"
                               iCLEAR_LOG := "M_ZERO",
                               oERROR_LIMIT => "DB426_ALARMS_WARNINGS".CLADDING_HOPPERS."717651",
                               oWARNING_LIMIT => "DB426_ALARMS_WARNINGS".WARNINGS."730086");
       "DB22147_MASS_SENSOR_HOPPER_3_UNIT_2"(INPUT_VALUE := "DB22150_WP321_WEIGHT_CELLS".WP321DR[4].DR30.GROSS_NET_WEIGHT,   // "FB22105_MASS_SENSOR"
                               CLEAR_INTERNAL_LOG := "M_ZERO",
                               "SAVE MAX VALUES" := "M_ONE",
                               OUT_OF_LIMITS_WARNING => "DB426_ALARMS_WARNINGS".WARNINGS."730087",
                               OUT_OF_LIMITS_ALARM => "DB426_ALARMS_WARNINGS".CLADDING_HOPPERS."717266");
   END_IF;
END_REGION

REGION Network 8: CALL FB22108 WP321_MUL_CALL
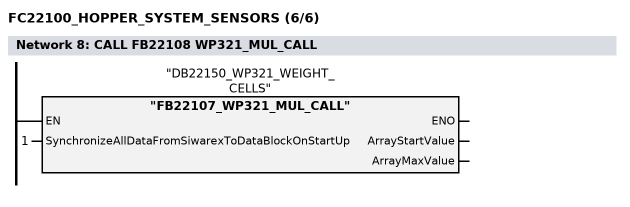
   RUNG wire#powerrail
      "DB22150_WP321_WEIGHT_CELLS"(SynchronizeAllDataFromSiwarexToDataBlockOnStartUp := 1, ArrayStartValue =>, ArrayMaxValue =>)
   END_RUNG
   // the same network as SCL:
   "DB22150_WP321_WEIGHT_CELLS"(SynchronizeAllDataFromSiwarexToDataBlockOnStartUp := 1);   // "FB22107_WP321_MUL_CALL"
END_REGION
END_FUNCTION

FUNCTION "FC22300_HOPPER_SYSTEM_ACTUATORS" : Void   // FC22300, LAD
TITLE = FC22300 HOPPER SYSTEM ACTUATORS
{ S7_Optimized_Access := 'TRUE' }
VERSION : 0.1
// stored: AutoNumber false, IsIECCheckEnabled false, SetENOAutomatically false, UDAEnableTagReadback false
BEGIN

REGION Network 1: //////////ACTUATORS HOPPERS UNIT 01//////////
END_REGION

REGION Network 2: CALL FB22301 TRANSFER POWDER VALVE HOPPER 1 UNIT 01
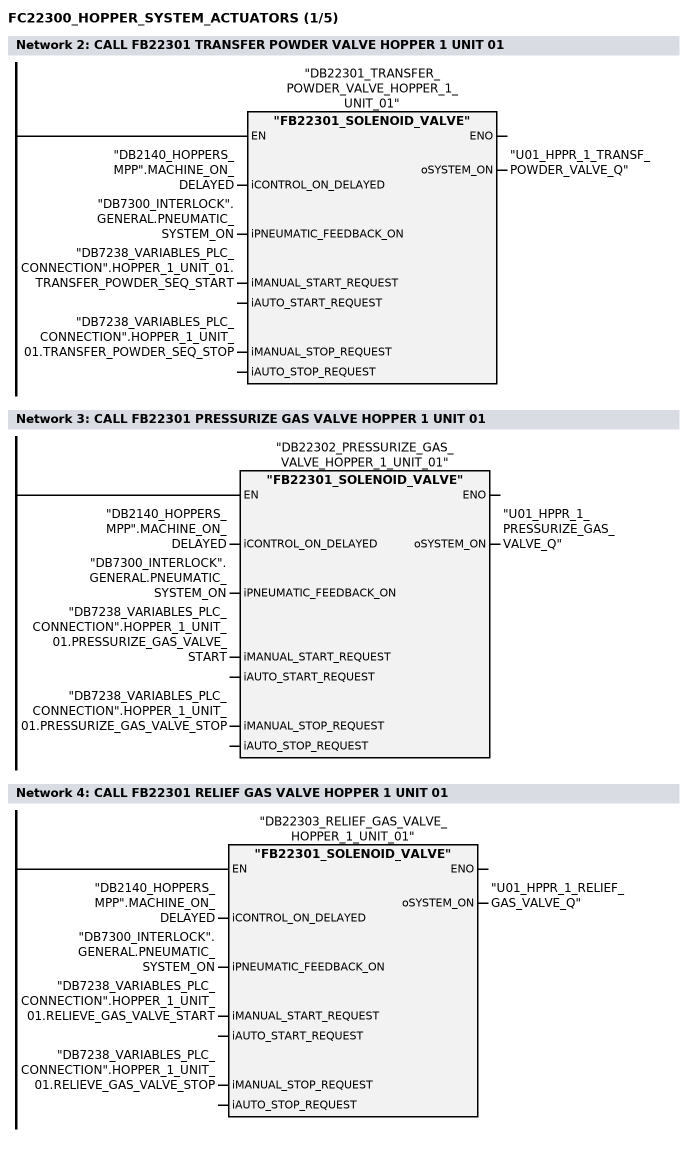
   RUNG wire#powerrail
      "DB22301_TRANSFER_POWDER_VALVE_HOPPER_1_UNIT_01"(iCONTROL_ON_DELAYED := "DB2140_HOPPERS_MPP".MACHINE_ON_DELAYED, iPNEUMATIC_FEEDBACK_ON := "DB7300_INTERLOCK".GENERAL.PNEUMATIC_SYSTEM_ON, iMANUAL_START_REQUEST := "DB7238_VARIABLES_PLC_CONNECTION".HOPPER_1_UNIT_01.TRANSFER_POWDER_SEQ_START, iAUTO_START_REQUEST :=, iMANUAL_STOP_REQUEST := "DB7238_VARIABLES_PLC_CONNECTION".HOPPER_1_UNIT_01.TRANSFER_POWDER_SEQ_STOP, iAUTO_STOP_REQUEST :=, oSYSTEM_ON => "U01_HPPR_1_TRANSF_POWDER_VALVE_Q")
   END_RUNG
   // the same network as SCL:
   "DB22301_TRANSFER_POWDER_VALVE_HOPPER_1_UNIT_01"(iCONTROL_ON_DELAYED := "DB2140_HOPPERS_MPP".MACHINE_ON_DELAYED,   // "FB22301_SOLENOID_VALVE"
                           iPNEUMATIC_FEEDBACK_ON := "DB7300_INTERLOCK".GENERAL.PNEUMATIC_SYSTEM_ON,
                           iMANUAL_START_REQUEST := "DB7238_VARIABLES_PLC_CONNECTION".HOPPER_1_UNIT_01.TRANSFER_POWDER_SEQ_START,
                           iMANUAL_STOP_REQUEST := "DB7238_VARIABLES_PLC_CONNECTION".HOPPER_1_UNIT_01.TRANSFER_POWDER_SEQ_STOP,
                           oSYSTEM_ON => "U01_HPPR_1_TRANSF_POWDER_VALVE_Q");
END_REGION

REGION Network 3: CALL FB22301 PRESSURIZE GAS VALVE HOPPER 1 UNIT 01
   RUNG wire#powerrail
      "DB22302_PRESSURIZE_GAS_VALVE_HOPPER_1_UNIT_01"(iCONTROL_ON_DELAYED := "DB2140_HOPPERS_MPP".MACHINE_ON_DELAYED, iPNEUMATIC_FEEDBACK_ON := "DB7300_INTERLOCK".GENERAL.PNEUMATIC_SYSTEM_ON, iMANUAL_START_REQUEST := "DB7238_VARIABLES_PLC_CONNECTION".HOPPER_1_UNIT_01.PRESSURIZE_GAS_VALVE_START, iAUTO_START_REQUEST :=, iMANUAL_STOP_REQUEST := "DB7238_VARIABLES_PLC_CONNECTION".HOPPER_1_UNIT_01.PRESSURIZE_GAS_VALVE_STOP, iAUTO_STOP_REQUEST :=, oSYSTEM_ON => "U01_HPPR_1_PRESSURIZE_GAS_VALVE_Q")
   END_RUNG
   // the same network as SCL:
   "DB22302_PRESSURIZE_GAS_VALVE_HOPPER_1_UNIT_01"(iCONTROL_ON_DELAYED := "DB2140_HOPPERS_MPP".MACHINE_ON_DELAYED,   // "FB22301_SOLENOID_VALVE"
                           iPNEUMATIC_FEEDBACK_ON := "DB7300_INTERLOCK".GENERAL.PNEUMATIC_SYSTEM_ON,
                           iMANUAL_START_REQUEST := "DB7238_VARIABLES_PLC_CONNECTION".HOPPER_1_UNIT_01.PRESSURIZE_GAS_VALVE_START,
                           iMANUAL_STOP_REQUEST := "DB7238_VARIABLES_PLC_CONNECTION".HOPPER_1_UNIT_01.PRESSURIZE_GAS_VALVE_STOP,
                           oSYSTEM_ON => "U01_HPPR_1_PRESSURIZE_GAS_VALVE_Q");
END_REGION

REGION Network 4: CALL FB22301 RELIEF GAS VALVE HOPPER 1 UNIT 01
   RUNG wire#powerrail
      "DB22303_RELIEF_GAS_VALVE_HOPPER_1_UNIT_01"(iCONTROL_ON_DELAYED := "DB2140_HOPPERS_MPP".MACHINE_ON_DELAYED, iPNEUMATIC_FEEDBACK_ON := "DB7300_INTERLOCK".GENERAL.PNEUMATIC_SYSTEM_ON, iMANUAL_START_REQUEST := "DB7238_VARIABLES_PLC_CONNECTION".HOPPER_1_UNIT_01.RELIEVE_GAS_VALVE_START, iAUTO_START_REQUEST :=, iMANUAL_STOP_REQUEST := "DB7238_VARIABLES_PLC_CONNECTION".HOPPER_1_UNIT_01.RELIEVE_GAS_VALVE_STOP, iAUTO_STOP_REQUEST :=, oSYSTEM_ON => "U01_HPPR_1_RELIEF_GAS_VALVE_Q")
   END_RUNG
   // the same network as SCL:
   "DB22303_RELIEF_GAS_VALVE_HOPPER_1_UNIT_01"(iCONTROL_ON_DELAYED := "DB2140_HOPPERS_MPP".MACHINE_ON_DELAYED,   // "FB22301_SOLENOID_VALVE"
                           iPNEUMATIC_FEEDBACK_ON := "DB7300_INTERLOCK".GENERAL.PNEUMATIC_SYSTEM_ON,
                           iMANUAL_START_REQUEST := "DB7238_VARIABLES_PLC_CONNECTION".HOPPER_1_UNIT_01.RELIEVE_GAS_VALVE_START,
                           iMANUAL_STOP_REQUEST := "DB7238_VARIABLES_PLC_CONNECTION".HOPPER_1_UNIT_01.RELIEVE_GAS_VALVE_STOP,
                           oSYSTEM_ON => "U01_HPPR_1_RELIEF_GAS_VALVE_Q");
END_REGION

REGION Network 5: CALL FB22301 TRANSFER POWDER VALVE HOPPER 2 UNIT 01
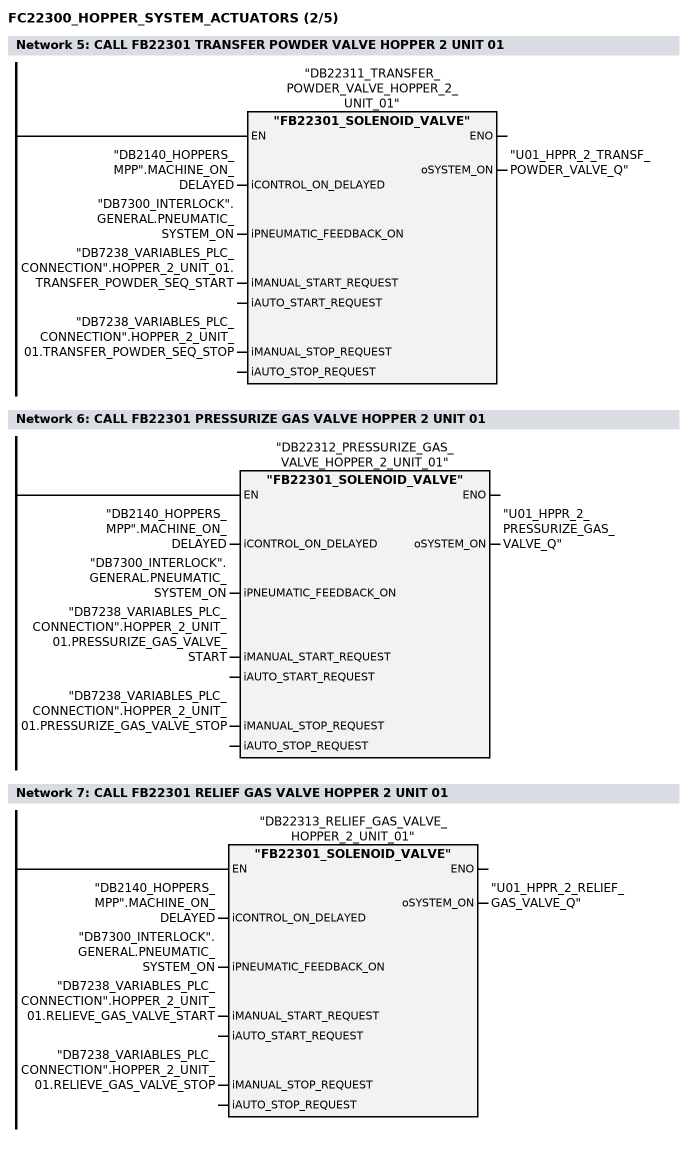
   RUNG wire#powerrail
      "DB22311_TRANSFER_POWDER_VALVE_HOPPER_2_UNIT_01"(iCONTROL_ON_DELAYED := "DB2140_HOPPERS_MPP".MACHINE_ON_DELAYED, iPNEUMATIC_FEEDBACK_ON := "DB7300_INTERLOCK".GENERAL.PNEUMATIC_SYSTEM_ON, iMANUAL_START_REQUEST := "DB7238_VARIABLES_PLC_CONNECTION".HOPPER_2_UNIT_01.TRANSFER_POWDER_SEQ_START, iAUTO_START_REQUEST :=, iMANUAL_STOP_REQUEST := "DB7238_VARIABLES_PLC_CONNECTION".HOPPER_2_UNIT_01.TRANSFER_POWDER_SEQ_STOP, iAUTO_STOP_REQUEST :=, oSYSTEM_ON => "U01_HPPR_2_TRANSF_POWDER_VALVE_Q")
   END_RUNG
   // the same network as SCL:
   "DB22311_TRANSFER_POWDER_VALVE_HOPPER_2_UNIT_01"(iCONTROL_ON_DELAYED := "DB2140_HOPPERS_MPP".MACHINE_ON_DELAYED,   // "FB22301_SOLENOID_VALVE"
                           iPNEUMATIC_FEEDBACK_ON := "DB7300_INTERLOCK".GENERAL.PNEUMATIC_SYSTEM_ON,
                           iMANUAL_START_REQUEST := "DB7238_VARIABLES_PLC_CONNECTION".HOPPER_2_UNIT_01.TRANSFER_POWDER_SEQ_START,
                           iMANUAL_STOP_REQUEST := "DB7238_VARIABLES_PLC_CONNECTION".HOPPER_2_UNIT_01.TRANSFER_POWDER_SEQ_STOP,
                           oSYSTEM_ON => "U01_HPPR_2_TRANSF_POWDER_VALVE_Q");
END_REGION

REGION Network 6: CALL FB22301 PRESSURIZE GAS VALVE HOPPER 2 UNIT 01
   RUNG wire#powerrail
      "DB22312_PRESSURIZE_GAS_VALVE_HOPPER_2_UNIT_01"(iCONTROL_ON_DELAYED := "DB2140_HOPPERS_MPP".MACHINE_ON_DELAYED, iPNEUMATIC_FEEDBACK_ON := "DB7300_INTERLOCK".GENERAL.PNEUMATIC_SYSTEM_ON, iMANUAL_START_REQUEST := "DB7238_VARIABLES_PLC_CONNECTION".HOPPER_2_UNIT_01.PRESSURIZE_GAS_VALVE_START, iAUTO_START_REQUEST :=, iMANUAL_STOP_REQUEST := "DB7238_VARIABLES_PLC_CONNECTION".HOPPER_2_UNIT_01.PRESSURIZE_GAS_VALVE_STOP, iAUTO_STOP_REQUEST :=, oSYSTEM_ON => "U01_HPPR_2_PRESSURIZE_GAS_VALVE_Q")
   END_RUNG
   // the same network as SCL:
   "DB22312_PRESSURIZE_GAS_VALVE_HOPPER_2_UNIT_01"(iCONTROL_ON_DELAYED := "DB2140_HOPPERS_MPP".MACHINE_ON_DELAYED,   // "FB22301_SOLENOID_VALVE"
                           iPNEUMATIC_FEEDBACK_ON := "DB7300_INTERLOCK".GENERAL.PNEUMATIC_SYSTEM_ON,
                           iMANUAL_START_REQUEST := "DB7238_VARIABLES_PLC_CONNECTION".HOPPER_2_UNIT_01.PRESSURIZE_GAS_VALVE_START,
                           iMANUAL_STOP_REQUEST := "DB7238_VARIABLES_PLC_CONNECTION".HOPPER_2_UNIT_01.PRESSURIZE_GAS_VALVE_STOP,
                           oSYSTEM_ON => "U01_HPPR_2_PRESSURIZE_GAS_VALVE_Q");
END_REGION

REGION Network 7: CALL FB22301 RELIEF GAS VALVE HOPPER 2 UNIT 01
   RUNG wire#powerrail
      "DB22313_RELIEF_GAS_VALVE_HOPPER_2_UNIT_01"(iCONTROL_ON_DELAYED := "DB2140_HOPPERS_MPP".MACHINE_ON_DELAYED, iPNEUMATIC_FEEDBACK_ON := "DB7300_INTERLOCK".GENERAL.PNEUMATIC_SYSTEM_ON, iMANUAL_START_REQUEST := "DB7238_VARIABLES_PLC_CONNECTION".HOPPER_2_UNIT_01.RELIEVE_GAS_VALVE_START, iAUTO_START_REQUEST :=, iMANUAL_STOP_REQUEST := "DB7238_VARIABLES_PLC_CONNECTION".HOPPER_2_UNIT_01.RELIEVE_GAS_VALVE_STOP, iAUTO_STOP_REQUEST :=, oSYSTEM_ON => "U01_HPPR_2_RELIEF_GAS_VALVE_Q")
   END_RUNG
   // the same network as SCL:
   "DB22313_RELIEF_GAS_VALVE_HOPPER_2_UNIT_01"(iCONTROL_ON_DELAYED := "DB2140_HOPPERS_MPP".MACHINE_ON_DELAYED,   // "FB22301_SOLENOID_VALVE"
                           iPNEUMATIC_FEEDBACK_ON := "DB7300_INTERLOCK".GENERAL.PNEUMATIC_SYSTEM_ON,
                           iMANUAL_START_REQUEST := "DB7238_VARIABLES_PLC_CONNECTION".HOPPER_2_UNIT_01.RELIEVE_GAS_VALVE_START,
                           iMANUAL_STOP_REQUEST := "DB7238_VARIABLES_PLC_CONNECTION".HOPPER_2_UNIT_01.RELIEVE_GAS_VALVE_STOP,
                           oSYSTEM_ON => "U01_HPPR_2_RELIEF_GAS_VALVE_Q");
END_REGION

REGION Network 8: //////////ACTUATORS HOPPERS UNIT 02//////////
END_REGION

REGION Network 9: CALL FB22301 TRANSFER POWDER VALVE HOPPER 1 UNIT 02
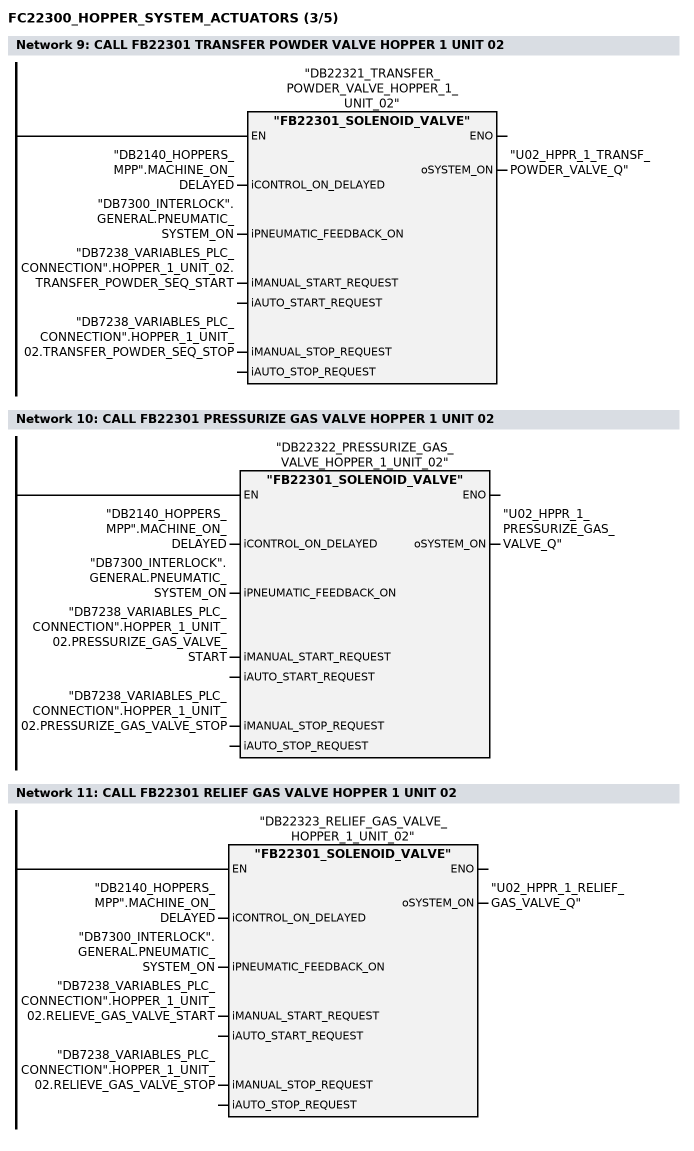
   RUNG wire#powerrail
      "DB22321_TRANSFER_POWDER_VALVE_HOPPER_1_UNIT_02"(iCONTROL_ON_DELAYED := "DB2140_HOPPERS_MPP".MACHINE_ON_DELAYED, iPNEUMATIC_FEEDBACK_ON := "DB7300_INTERLOCK".GENERAL.PNEUMATIC_SYSTEM_ON, iMANUAL_START_REQUEST := "DB7238_VARIABLES_PLC_CONNECTION".HOPPER_1_UNIT_02.TRANSFER_POWDER_SEQ_START, iAUTO_START_REQUEST :=, iMANUAL_STOP_REQUEST := "DB7238_VARIABLES_PLC_CONNECTION".HOPPER_1_UNIT_02.TRANSFER_POWDER_SEQ_STOP, iAUTO_STOP_REQUEST :=, oSYSTEM_ON => "U02_HPPR_1_TRANSF_POWDER_VALVE_Q")
   END_RUNG
   // the same network as SCL:
   "DB22321_TRANSFER_POWDER_VALVE_HOPPER_1_UNIT_02"(iCONTROL_ON_DELAYED := "DB2140_HOPPERS_MPP".MACHINE_ON_DELAYED,   // "FB22301_SOLENOID_VALVE"
                           iPNEUMATIC_FEEDBACK_ON := "DB7300_INTERLOCK".GENERAL.PNEUMATIC_SYSTEM_ON,
                           iMANUAL_START_REQUEST := "DB7238_VARIABLES_PLC_CONNECTION".HOPPER_1_UNIT_02.TRANSFER_POWDER_SEQ_START,
                           iMANUAL_STOP_REQUEST := "DB7238_VARIABLES_PLC_CONNECTION".HOPPER_1_UNIT_02.TRANSFER_POWDER_SEQ_STOP,
                           oSYSTEM_ON => "U02_HPPR_1_TRANSF_POWDER_VALVE_Q");
END_REGION

REGION Network 10: CALL FB22301 PRESSURIZE GAS VALVE HOPPER 1 UNIT 02
   RUNG wire#powerrail
      "DB22322_PRESSURIZE_GAS_VALVE_HOPPER_1_UNIT_02"(iCONTROL_ON_DELAYED := "DB2140_HOPPERS_MPP".MACHINE_ON_DELAYED, iPNEUMATIC_FEEDBACK_ON := "DB7300_INTERLOCK".GENERAL.PNEUMATIC_SYSTEM_ON, iMANUAL_START_REQUEST := "DB7238_VARIABLES_PLC_CONNECTION".HOPPER_1_UNIT_02.PRESSURIZE_GAS_VALVE_START, iAUTO_START_REQUEST :=, iMANUAL_STOP_REQUEST := "DB7238_VARIABLES_PLC_CONNECTION".HOPPER_1_UNIT_02.PRESSURIZE_GAS_VALVE_STOP, iAUTO_STOP_REQUEST :=, oSYSTEM_ON => "U02_HPPR_1_PRESSURIZE_GAS_VALVE_Q")
   END_RUNG
   // the same network as SCL:
   "DB22322_PRESSURIZE_GAS_VALVE_HOPPER_1_UNIT_02"(iCONTROL_ON_DELAYED := "DB2140_HOPPERS_MPP".MACHINE_ON_DELAYED,   // "FB22301_SOLENOID_VALVE"
                           iPNEUMATIC_FEEDBACK_ON := "DB7300_INTERLOCK".GENERAL.PNEUMATIC_SYSTEM_ON,
                           iMANUAL_START_REQUEST := "DB7238_VARIABLES_PLC_CONNECTION".HOPPER_1_UNIT_02.PRESSURIZE_GAS_VALVE_START,
                           iMANUAL_STOP_REQUEST := "DB7238_VARIABLES_PLC_CONNECTION".HOPPER_1_UNIT_02.PRESSURIZE_GAS_VALVE_STOP,
                           oSYSTEM_ON => "U02_HPPR_1_PRESSURIZE_GAS_VALVE_Q");
END_REGION

REGION Network 11: CALL FB22301 RELIEF GAS VALVE HOPPER 1 UNIT 02
   RUNG wire#powerrail
      "DB22323_RELIEF_GAS_VALVE_HOPPER_1_UNIT_02"(iCONTROL_ON_DELAYED := "DB2140_HOPPERS_MPP".MACHINE_ON_DELAYED, iPNEUMATIC_FEEDBACK_ON := "DB7300_INTERLOCK".GENERAL.PNEUMATIC_SYSTEM_ON, iMANUAL_START_REQUEST := "DB7238_VARIABLES_PLC_CONNECTION".HOPPER_1_UNIT_02.RELIEVE_GAS_VALVE_START, iAUTO_START_REQUEST :=, iMANUAL_STOP_REQUEST := "DB7238_VARIABLES_PLC_CONNECTION".HOPPER_1_UNIT_02.RELIEVE_GAS_VALVE_STOP, iAUTO_STOP_REQUEST :=, oSYSTEM_ON => "U02_HPPR_1_RELIEF_GAS_VALVE_Q")
   END_RUNG
   // the same network as SCL:
   "DB22323_RELIEF_GAS_VALVE_HOPPER_1_UNIT_02"(iCONTROL_ON_DELAYED := "DB2140_HOPPERS_MPP".MACHINE_ON_DELAYED,   // "FB22301_SOLENOID_VALVE"
                           iPNEUMATIC_FEEDBACK_ON := "DB7300_INTERLOCK".GENERAL.PNEUMATIC_SYSTEM_ON,
                           iMANUAL_START_REQUEST := "DB7238_VARIABLES_PLC_CONNECTION".HOPPER_1_UNIT_02.RELIEVE_GAS_VALVE_START,
                           iMANUAL_STOP_REQUEST := "DB7238_VARIABLES_PLC_CONNECTION".HOPPER_1_UNIT_02.RELIEVE_GAS_VALVE_STOP,
                           oSYSTEM_ON => "U02_HPPR_1_RELIEF_GAS_VALVE_Q");
END_REGION

REGION Network 12: CALL FB22301 TRANSFER POWDER VALVE HOPPER 2 UNIT 02
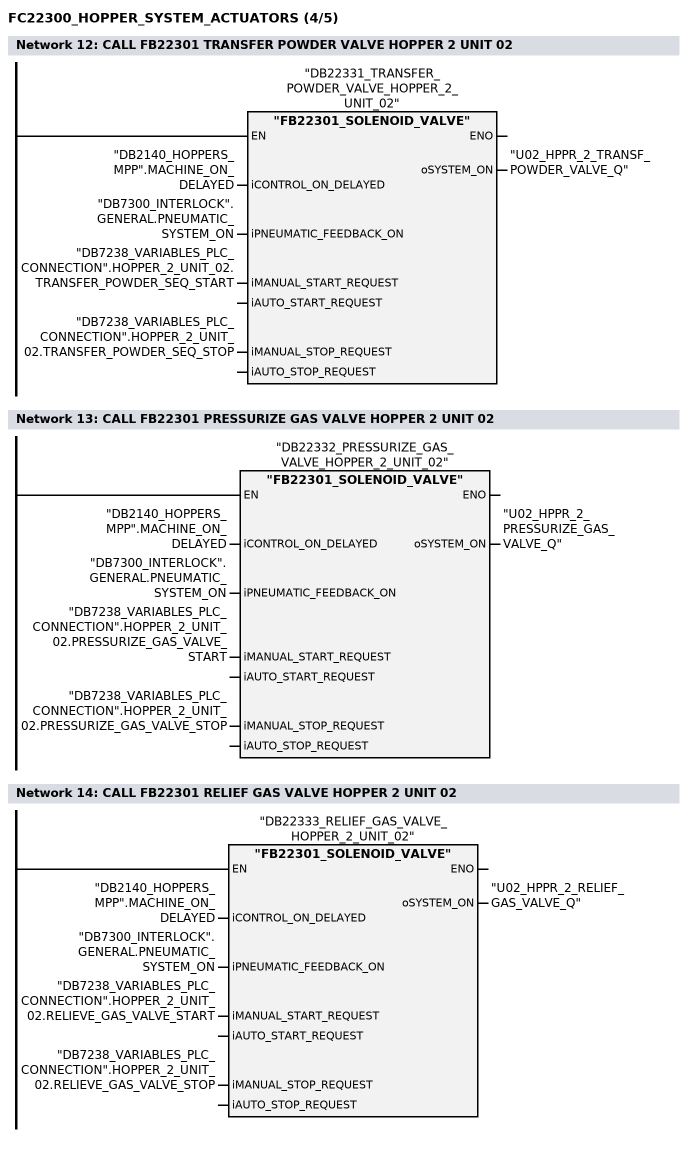
   RUNG wire#powerrail
      "DB22331_TRANSFER_POWDER_VALVE_HOPPER_2_UNIT_02"(iCONTROL_ON_DELAYED := "DB2140_HOPPERS_MPP".MACHINE_ON_DELAYED, iPNEUMATIC_FEEDBACK_ON := "DB7300_INTERLOCK".GENERAL.PNEUMATIC_SYSTEM_ON, iMANUAL_START_REQUEST := "DB7238_VARIABLES_PLC_CONNECTION".HOPPER_2_UNIT_02.TRANSFER_POWDER_SEQ_START, iAUTO_START_REQUEST :=, iMANUAL_STOP_REQUEST := "DB7238_VARIABLES_PLC_CONNECTION".HOPPER_2_UNIT_02.TRANSFER_POWDER_SEQ_STOP, iAUTO_STOP_REQUEST :=, oSYSTEM_ON => "U02_HPPR_2_TRANSF_POWDER_VALVE_Q")
   END_RUNG
   // the same network as SCL:
   "DB22331_TRANSFER_POWDER_VALVE_HOPPER_2_UNIT_02"(iCONTROL_ON_DELAYED := "DB2140_HOPPERS_MPP".MACHINE_ON_DELAYED,   // "FB22301_SOLENOID_VALVE"
                           iPNEUMATIC_FEEDBACK_ON := "DB7300_INTERLOCK".GENERAL.PNEUMATIC_SYSTEM_ON,
                           iMANUAL_START_REQUEST := "DB7238_VARIABLES_PLC_CONNECTION".HOPPER_2_UNIT_02.TRANSFER_POWDER_SEQ_START,
                           iMANUAL_STOP_REQUEST := "DB7238_VARIABLES_PLC_CONNECTION".HOPPER_2_UNIT_02.TRANSFER_POWDER_SEQ_STOP,
                           oSYSTEM_ON => "U02_HPPR_2_TRANSF_POWDER_VALVE_Q");
END_REGION

REGION Network 13: CALL FB22301 PRESSURIZE GAS VALVE HOPPER 2 UNIT 02
   RUNG wire#powerrail
      "DB22332_PRESSURIZE_GAS_VALVE_HOPPER_2_UNIT_02"(iCONTROL_ON_DELAYED := "DB2140_HOPPERS_MPP".MACHINE_ON_DELAYED, iPNEUMATIC_FEEDBACK_ON := "DB7300_INTERLOCK".GENERAL.PNEUMATIC_SYSTEM_ON, iMANUAL_START_REQUEST := "DB7238_VARIABLES_PLC_CONNECTION".HOPPER_2_UNIT_02.PRESSURIZE_GAS_VALVE_START, iAUTO_START_REQUEST :=, iMANUAL_STOP_REQUEST := "DB7238_VARIABLES_PLC_CONNECTION".HOPPER_2_UNIT_02.PRESSURIZE_GAS_VALVE_STOP, iAUTO_STOP_REQUEST :=, oSYSTEM_ON => "U02_HPPR_2_PRESSURIZE_GAS_VALVE_Q")
   END_RUNG
   // the same network as SCL:
   "DB22332_PRESSURIZE_GAS_VALVE_HOPPER_2_UNIT_02"(iCONTROL_ON_DELAYED := "DB2140_HOPPERS_MPP".MACHINE_ON_DELAYED,   // "FB22301_SOLENOID_VALVE"
                           iPNEUMATIC_FEEDBACK_ON := "DB7300_INTERLOCK".GENERAL.PNEUMATIC_SYSTEM_ON,
                           iMANUAL_START_REQUEST := "DB7238_VARIABLES_PLC_CONNECTION".HOPPER_2_UNIT_02.PRESSURIZE_GAS_VALVE_START,
                           iMANUAL_STOP_REQUEST := "DB7238_VARIABLES_PLC_CONNECTION".HOPPER_2_UNIT_02.PRESSURIZE_GAS_VALVE_STOP,
                           oSYSTEM_ON => "U02_HPPR_2_PRESSURIZE_GAS_VALVE_Q");
END_REGION

REGION Network 14: CALL FB22301 RELIEF GAS VALVE HOPPER 2 UNIT 02
   RUNG wire#powerrail
      "DB22333_RELIEF_GAS_VALVE_HOPPER_2_UNIT_02"(iCONTROL_ON_DELAYED := "DB2140_HOPPERS_MPP".MACHINE_ON_DELAYED, iPNEUMATIC_FEEDBACK_ON := "DB7300_INTERLOCK".GENERAL.PNEUMATIC_SYSTEM_ON, iMANUAL_START_REQUEST := "DB7238_VARIABLES_PLC_CONNECTION".HOPPER_2_UNIT_02.RELIEVE_GAS_VALVE_START, iAUTO_START_REQUEST :=, iMANUAL_STOP_REQUEST := "DB7238_VARIABLES_PLC_CONNECTION".HOPPER_2_UNIT_02.RELIEVE_GAS_VALVE_STOP, iAUTO_STOP_REQUEST :=, oSYSTEM_ON => "U02_HPPR_2_RELIEF_GAS_VALVE_Q")
   END_RUNG
   // the same network as SCL:
   "DB22333_RELIEF_GAS_VALVE_HOPPER_2_UNIT_02"(iCONTROL_ON_DELAYED := "DB2140_HOPPERS_MPP".MACHINE_ON_DELAYED,   // "FB22301_SOLENOID_VALVE"
                           iPNEUMATIC_FEEDBACK_ON := "DB7300_INTERLOCK".GENERAL.PNEUMATIC_SYSTEM_ON,
                           iMANUAL_START_REQUEST := "DB7238_VARIABLES_PLC_CONNECTION".HOPPER_2_UNIT_02.RELIEVE_GAS_VALVE_START,
                           iMANUAL_STOP_REQUEST := "DB7238_VARIABLES_PLC_CONNECTION".HOPPER_2_UNIT_02.RELIEVE_GAS_VALVE_STOP,
                           oSYSTEM_ON => "U02_HPPR_2_RELIEF_GAS_VALVE_Q");
END_REGION

REGION Network 15: CALL FB22301 TRANSFER POWDER VALVE HOPPER 3 UNIT 02
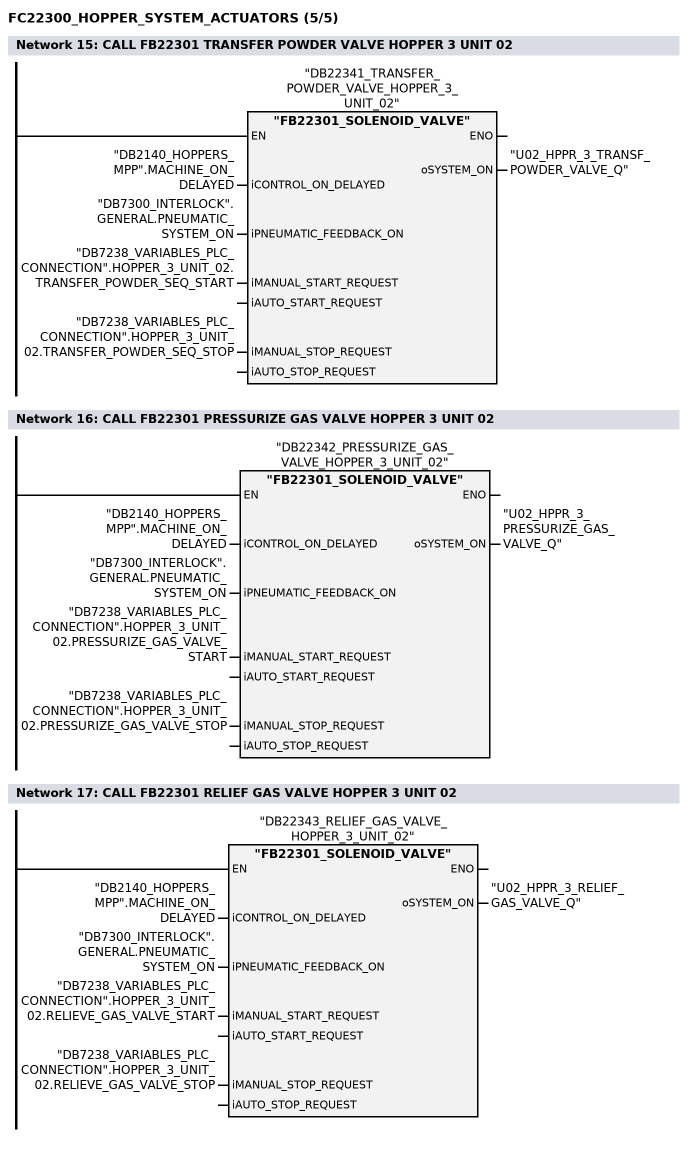
   RUNG wire#powerrail
      "DB22341_TRANSFER_POWDER_VALVE_HOPPER_3_UNIT_02"(iCONTROL_ON_DELAYED := "DB2140_HOPPERS_MPP".MACHINE_ON_DELAYED, iPNEUMATIC_FEEDBACK_ON := "DB7300_INTERLOCK".GENERAL.PNEUMATIC_SYSTEM_ON, iMANUAL_START_REQUEST := "DB7238_VARIABLES_PLC_CONNECTION".HOPPER_3_UNIT_02.TRANSFER_POWDER_SEQ_START, iAUTO_START_REQUEST :=, iMANUAL_STOP_REQUEST := "DB7238_VARIABLES_PLC_CONNECTION".HOPPER_3_UNIT_02.TRANSFER_POWDER_SEQ_STOP, iAUTO_STOP_REQUEST :=, oSYSTEM_ON => "U02_HPPR_3_TRANSF_POWDER_VALVE_Q")
   END_RUNG
   // the same network as SCL:
   "DB22341_TRANSFER_POWDER_VALVE_HOPPER_3_UNIT_02"(iCONTROL_ON_DELAYED := "DB2140_HOPPERS_MPP".MACHINE_ON_DELAYED,   // "FB22301_SOLENOID_VALVE"
                           iPNEUMATIC_FEEDBACK_ON := "DB7300_INTERLOCK".GENERAL.PNEUMATIC_SYSTEM_ON,
                           iMANUAL_START_REQUEST := "DB7238_VARIABLES_PLC_CONNECTION".HOPPER_3_UNIT_02.TRANSFER_POWDER_SEQ_START,
                           iMANUAL_STOP_REQUEST := "DB7238_VARIABLES_PLC_CONNECTION".HOPPER_3_UNIT_02.TRANSFER_POWDER_SEQ_STOP,
                           oSYSTEM_ON => "U02_HPPR_3_TRANSF_POWDER_VALVE_Q");
END_REGION

REGION Network 16: CALL FB22301 PRESSURIZE GAS VALVE HOPPER 3 UNIT 02
   RUNG wire#powerrail
      "DB22342_PRESSURIZE_GAS_VALVE_HOPPER_3_UNIT_02"(iCONTROL_ON_DELAYED := "DB2140_HOPPERS_MPP".MACHINE_ON_DELAYED, iPNEUMATIC_FEEDBACK_ON := "DB7300_INTERLOCK".GENERAL.PNEUMATIC_SYSTEM_ON, iMANUAL_START_REQUEST := "DB7238_VARIABLES_PLC_CONNECTION".HOPPER_3_UNIT_02.PRESSURIZE_GAS_VALVE_START, iAUTO_START_REQUEST :=, iMANUAL_STOP_REQUEST := "DB7238_VARIABLES_PLC_CONNECTION".HOPPER_3_UNIT_02.PRESSURIZE_GAS_VALVE_STOP, iAUTO_STOP_REQUEST :=, oSYSTEM_ON => "U02_HPPR_3_PRESSURIZE_GAS_VALVE_Q")
   END_RUNG
   // the same network as SCL:
   "DB22342_PRESSURIZE_GAS_VALVE_HOPPER_3_UNIT_02"(iCONTROL_ON_DELAYED := "DB2140_HOPPERS_MPP".MACHINE_ON_DELAYED,   // "FB22301_SOLENOID_VALVE"
                           iPNEUMATIC_FEEDBACK_ON := "DB7300_INTERLOCK".GENERAL.PNEUMATIC_SYSTEM_ON,
                           iMANUAL_START_REQUEST := "DB7238_VARIABLES_PLC_CONNECTION".HOPPER_3_UNIT_02.PRESSURIZE_GAS_VALVE_START,
                           iMANUAL_STOP_REQUEST := "DB7238_VARIABLES_PLC_CONNECTION".HOPPER_3_UNIT_02.PRESSURIZE_GAS_VALVE_STOP,
                           oSYSTEM_ON => "U02_HPPR_3_PRESSURIZE_GAS_VALVE_Q");
END_REGION

REGION Network 17: CALL FB22301 RELIEF GAS VALVE HOPPER 3 UNIT 02
   RUNG wire#powerrail
      "DB22343_RELIEF_GAS_VALVE_HOPPER_3_UNIT_02"(iCONTROL_ON_DELAYED := "DB2140_HOPPERS_MPP".MACHINE_ON_DELAYED, iPNEUMATIC_FEEDBACK_ON := "DB7300_INTERLOCK".GENERAL.PNEUMATIC_SYSTEM_ON, iMANUAL_START_REQUEST := "DB7238_VARIABLES_PLC_CONNECTION".HOPPER_3_UNIT_02.RELIEVE_GAS_VALVE_START, iAUTO_START_REQUEST :=, iMANUAL_STOP_REQUEST := "DB7238_VARIABLES_PLC_CONNECTION".HOPPER_3_UNIT_02.RELIEVE_GAS_VALVE_STOP, iAUTO_STOP_REQUEST :=, oSYSTEM_ON => "U02_HPPR_3_RELIEF_GAS_VALVE_Q")
   END_RUNG
   // the same network as SCL:
   "DB22343_RELIEF_GAS_VALVE_HOPPER_3_UNIT_02"(iCONTROL_ON_DELAYED := "DB2140_HOPPERS_MPP".MACHINE_ON_DELAYED,   // "FB22301_SOLENOID_VALVE"
                           iPNEUMATIC_FEEDBACK_ON := "DB7300_INTERLOCK".GENERAL.PNEUMATIC_SYSTEM_ON,
                           iMANUAL_START_REQUEST := "DB7238_VARIABLES_PLC_CONNECTION".HOPPER_3_UNIT_02.RELIEVE_GAS_VALVE_START,
                           iMANUAL_STOP_REQUEST := "DB7238_VARIABLES_PLC_CONNECTION".HOPPER_3_UNIT_02.RELIEVE_GAS_VALVE_STOP,
                           oSYSTEM_ON => "U02_HPPR_3_RELIEF_GAS_VALVE_Q");
END_REGION
END_FUNCTION

FUNCTION "FC22500_HOPPER_SYSTEM_CONTROLS" : Void   // FC22500, LAD
TITLE = FC22500 HOPPER SYSTEM CONTROLS
{ S7_Optimized_Access := 'TRUE' }
VERSION : 0.1
// stored: AutoNumber false, IsIECCheckEnabled false, SetENOAutomatically false, UDAEnableTagReadback false
   VAR_TEMP
      RPM_INT_AUX : Word;
      RPM_REAL_AUX : Real;
   END_VAR
BEGIN

REGION Network 1: //////////UNIT 01 HOPERS CONTROLS//////////
END_REGION

REGION Network 2: CALL FB22501 TEMPERATURE JKT CONTROL UPPER HOPPER 1 UNIT 01
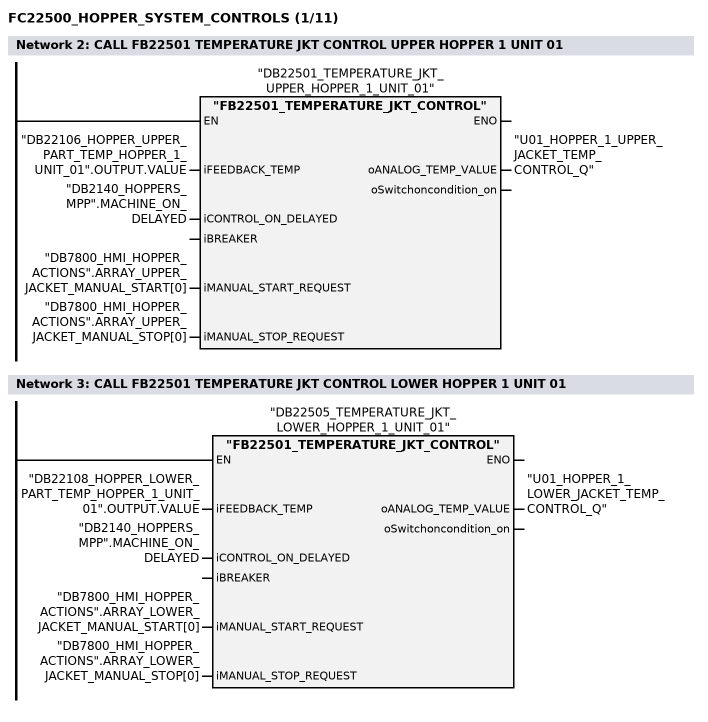
   RUNG wire#powerrail
      "DB22501_TEMPERATURE_JKT_UPPER_HOPPER_1_UNIT_01"(iFEEDBACK_TEMP := "DB22106_HOPPER_UPPER_PART_TEMP_HOPPER_1_UNIT_01".OUTPUT.VALUE, iCONTROL_ON_DELAYED := "DB2140_HOPPERS_MPP".MACHINE_ON_DELAYED, iBREAKER :=, iMANUAL_START_REQUEST := "DB7800_HMI_HOPPER_ACTIONS".ARRAY_UPPER_JACKET_MANUAL_START[0], iMANUAL_STOP_REQUEST := "DB7800_HMI_HOPPER_ACTIONS".ARRAY_UPPER_JACKET_MANUAL_STOP[0], oANALOG_TEMP_VALUE => "U01_HOPPER_1_UPPER_JACKET_TEMP_CONTROL_Q", oSwitchoncondition_on =>)
   END_RUNG
   // the same network as SCL:
   "DB22501_TEMPERATURE_JKT_UPPER_HOPPER_1_UNIT_01"(iFEEDBACK_TEMP := "DB22106_HOPPER_UPPER_PART_TEMP_HOPPER_1_UNIT_01".OUTPUT.VALUE,   // "FB22501_TEMPERATURE_JKT_CONTROL"
                           iCONTROL_ON_DELAYED := "DB2140_HOPPERS_MPP".MACHINE_ON_DELAYED,
                           iMANUAL_START_REQUEST := "DB7800_HMI_HOPPER_ACTIONS".ARRAY_UPPER_JACKET_MANUAL_START[0],
                           iMANUAL_STOP_REQUEST := "DB7800_HMI_HOPPER_ACTIONS".ARRAY_UPPER_JACKET_MANUAL_STOP[0],
                           oANALOG_TEMP_VALUE => "U01_HOPPER_1_UPPER_JACKET_TEMP_CONTROL_Q");
END_REGION

REGION Network 3: CALL FB22501 TEMPERATURE JKT CONTROL LOWER HOPPER 1 UNIT 01
   RUNG wire#powerrail
      "DB22505_TEMPERATURE_JKT_LOWER_HOPPER_1_UNIT_01"(iFEEDBACK_TEMP := "DB22108_HOPPER_LOWER_PART_TEMP_HOPPER_1_UNIT_01".OUTPUT.VALUE, iCONTROL_ON_DELAYED := "DB2140_HOPPERS_MPP".MACHINE_ON_DELAYED, iBREAKER :=, iMANUAL_START_REQUEST := "DB7800_HMI_HOPPER_ACTIONS".ARRAY_LOWER_JACKET_MANUAL_START[0], iMANUAL_STOP_REQUEST := "DB7800_HMI_HOPPER_ACTIONS".ARRAY_LOWER_JACKET_MANUAL_STOP[0], oANALOG_TEMP_VALUE => "U01_HOPPER_1_LOWER_JACKET_TEMP_CONTROL_Q", oSwitchoncondition_on =>)
   END_RUNG
   // the same network as SCL:
   "DB22505_TEMPERATURE_JKT_LOWER_HOPPER_1_UNIT_01"(iFEEDBACK_TEMP := "DB22108_HOPPER_LOWER_PART_TEMP_HOPPER_1_UNIT_01".OUTPUT.VALUE,   // "FB22501_TEMPERATURE_JKT_CONTROL"
                           iCONTROL_ON_DELAYED := "DB2140_HOPPERS_MPP".MACHINE_ON_DELAYED,
                           iMANUAL_START_REQUEST := "DB7800_HMI_HOPPER_ACTIONS".ARRAY_LOWER_JACKET_MANUAL_START[0],
                           iMANUAL_STOP_REQUEST := "DB7800_HMI_HOPPER_ACTIONS".ARRAY_LOWER_JACKET_MANUAL_STOP[0],
                           oANALOG_TEMP_VALUE => "U01_HOPPER_1_LOWER_JACKET_TEMP_CONTROL_Q");
END_REGION

REGION Network 4: CALL FB22502 MOTOR STIRRER CONTROL HOPPER 1 UNIT 01
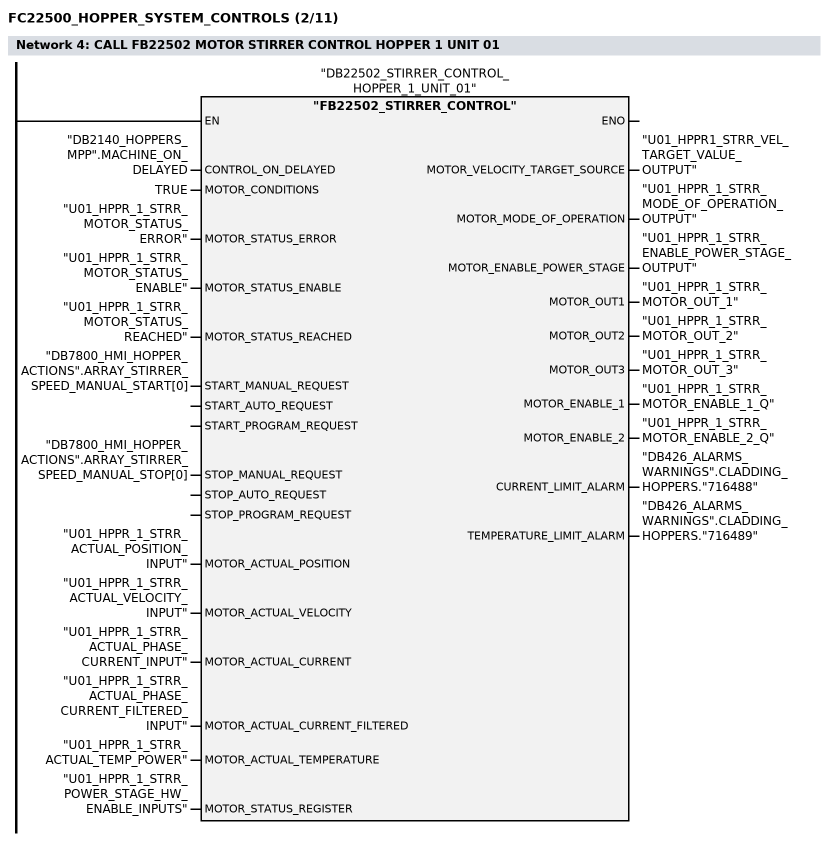
   RUNG wire#powerrail
      "DB22502_STIRRER_CONTROL_HOPPER_1_UNIT_01"(CONTROL_ON_DELAYED := "DB2140_HOPPERS_MPP".MACHINE_ON_DELAYED, MOTOR_CONDITIONS := TRUE, MOTOR_STATUS_ERROR := "U01_HPPR_1_STRR_MOTOR_STATUS_ERROR", MOTOR_STATUS_ENABLE := "U01_HPPR_1_STRR_MOTOR_STATUS_ENABLE", MOTOR_STATUS_REACHED := "U01_HPPR_1_STRR_MOTOR_STATUS_REACHED", START_MANUAL_REQUEST := "DB7800_HMI_HOPPER_ACTIONS".ARRAY_STIRRER_SPEED_MANUAL_START[0], START_AUTO_REQUEST :=, START_PROGRAM_REQUEST :=, STOP_MANUAL_REQUEST := "DB7800_HMI_HOPPER_ACTIONS".ARRAY_STIRRER_SPEED_MANUAL_STOP[0], STOP_AUTO_REQUEST :=, STOP_PROGRAM_REQUEST :=, MOTOR_ACTUAL_POSITION := "U01_HPPR_1_STRR_ACTUAL_POSITION_INPUT", MOTOR_ACTUAL_VELOCITY := "U01_HPPR_1_STRR_ACTUAL_VELOCITY_INPUT", MOTOR_ACTUAL_CURRENT := "U01_HPPR_1_STRR_ACTUAL_PHASE_CURRENT_INPUT", MOTOR_ACTUAL_CURRENT_FILTERED := "U01_HPPR_1_STRR_ACTUAL_PHASE_CURRENT_FILTERED_INPUT", MOTOR_ACTUAL_TEMPERATURE := "U01_HPPR_1_STRR_ACTUAL_TEMP_POWER", MOTOR_STATUS_REGISTER := "U01_HPPR_1_STRR_POWER_STAGE_HW_ENABLE_INPUTS", MOTOR_VELOCITY_TARGET_SOURCE => "U01_HPPR1_STRR_VEL_TARGET_VALUE_OUTPUT", MOTOR_MODE_OF_OPERATION => "U01_HPPR_1_STRR_MODE_OF_OPERATION_OUTPUT", MOTOR_ENABLE_POWER_STAGE => "U01_HPPR_1_STRR_ENABLE_POWER_STAGE_OUTPUT", MOTOR_OUT1 => "U01_HPPR_1_STRR_MOTOR_OUT_1", MOTOR_OUT2 => "U01_HPPR_1_STRR_MOTOR_OUT_2", MOTOR_OUT3 => "U01_HPPR_1_STRR_MOTOR_OUT_3", MOTOR_ENABLE_1 => "U01_HPPR_1_STRR_MOTOR_ENABLE_1_Q", MOTOR_ENABLE_2 => "U01_HPPR_1_STRR_MOTOR_ENABLE_2_Q", CURRENT_LIMIT_ALARM => "DB426_ALARMS_WARNINGS".CLADDING_HOPPERS."716488", TEMPERATURE_LIMIT_ALARM => "DB426_ALARMS_WARNINGS".CLADDING_HOPPERS."716489")
   END_RUNG
   // the same network as SCL:
   "DB22502_STIRRER_CONTROL_HOPPER_1_UNIT_01"(CONTROL_ON_DELAYED := "DB2140_HOPPERS_MPP".MACHINE_ON_DELAYED,   // "FB22502_STIRRER_CONTROL"
                           MOTOR_CONDITIONS := TRUE,
                           MOTOR_STATUS_ERROR := "U01_HPPR_1_STRR_MOTOR_STATUS_ERROR",
                           MOTOR_STATUS_ENABLE := "U01_HPPR_1_STRR_MOTOR_STATUS_ENABLE",
                           MOTOR_STATUS_REACHED := "U01_HPPR_1_STRR_MOTOR_STATUS_REACHED",
                           START_MANUAL_REQUEST := "DB7800_HMI_HOPPER_ACTIONS".ARRAY_STIRRER_SPEED_MANUAL_START[0],
                           STOP_MANUAL_REQUEST := "DB7800_HMI_HOPPER_ACTIONS".ARRAY_STIRRER_SPEED_MANUAL_STOP[0],
                           MOTOR_ACTUAL_POSITION := "U01_HPPR_1_STRR_ACTUAL_POSITION_INPUT",
                           MOTOR_ACTUAL_VELOCITY := "U01_HPPR_1_STRR_ACTUAL_VELOCITY_INPUT",
                           MOTOR_ACTUAL_CURRENT := "U01_HPPR_1_STRR_ACTUAL_PHASE_CURRENT_INPUT",
                           MOTOR_ACTUAL_CURRENT_FILTERED := "U01_HPPR_1_STRR_ACTUAL_PHASE_CURRENT_FILTERED_INPUT",
                           MOTOR_ACTUAL_TEMPERATURE := "U01_HPPR_1_STRR_ACTUAL_TEMP_POWER",
                           MOTOR_STATUS_REGISTER := "U01_HPPR_1_STRR_POWER_STAGE_HW_ENABLE_INPUTS",
                           MOTOR_VELOCITY_TARGET_SOURCE => "U01_HPPR1_STRR_VEL_TARGET_VALUE_OUTPUT",
                           MOTOR_MODE_OF_OPERATION => "U01_HPPR_1_STRR_MODE_OF_OPERATION_OUTPUT",
                           MOTOR_ENABLE_POWER_STAGE => "U01_HPPR_1_STRR_ENABLE_POWER_STAGE_OUTPUT",
                           MOTOR_OUT1 => "U01_HPPR_1_STRR_MOTOR_OUT_1",
                           MOTOR_OUT2 => "U01_HPPR_1_STRR_MOTOR_OUT_2",
                           MOTOR_OUT3 => "U01_HPPR_1_STRR_MOTOR_OUT_3",
                           MOTOR_ENABLE_1 => "U01_HPPR_1_STRR_MOTOR_ENABLE_1_Q",
                           MOTOR_ENABLE_2 => "U01_HPPR_1_STRR_MOTOR_ENABLE_2_Q",
                           CURRENT_LIMIT_ALARM => "DB426_ALARMS_WARNINGS".CLADDING_HOPPERS."716488",
                           TEMPERATURE_LIMIT_ALARM => "DB426_ALARMS_WARNINGS".CLADDING_HOPPERS."716489");
END_REGION

REGION Network 5: CALL FB22503 HOPPER COVER PRESSURE CONTROL HOPPER 1 UNIT 01
